// TIA Portal project "Project3" (V14)

(* hardware
DEVICE "S7-1200 station_1"  S7-1200 Station
   slot 0: "Rack_0"  S7-1200 Rack  Rack  V1.0
   slot 1: "PLC_1"  CPU 1215C DC/DC/DC  6ES7 215-1AG40-0XB0  V4.2
   slot 2: "DI 16/DQ 16x24VDC_1"  6ES7 223-1BL32-0XB0  V2.0
   slot 3: "DI 16/DQ 16x24VDC_2"  6ES7 223-1BL32-0XB0  V2.0
   slot 4: "AI 4x13BIT_1"  6ES7 231-4HD32-0XB0  V2.0
   slot 5: "AI 4xRTD_1"  SM 1231 AI4 x RTD  6ES7 231-5PD32-0XB0  V2.0
DEVICE "S7-1200 station_2"  S7-1200 Station
   slot 0: "Rack_0"  S7-1200 Rack  Rack  V1.0
   slot 1: "PLC_2"  CPU 1214C DC/DC/DC  6ES7 214-1AG40-0XB0  V4.2
   slot 2: "DI 16/DQ 16x24VDC_1"  6ES7 223-1BL32-0XB0  V2.0
   slot 3: "AQ 4x14BIT_1"  6ES7 232-4HD32-0XB0  V2.0
*)

// ===== PLC "PLC_1"  CPU 1215C DC/DC/DC =====

VAR_GLOBAL   // PLC tag table "Default tag table"
   "Rabota_M1.1" AT %I8.0 : Bool;
   "Rabota_X_M2" AT %I8.1 : Bool;
   "SL12.5.1" AT %I1.2 : Bool;
   "Gotovnost_M3" AT %I300.0 : Bool;
   "Rabota_M4" AT %I8.2 : Bool;
   "Rabota_M5" AT %I8.3 : Bool;
   "Gotovnost_X_M6.1" AT %I300.1 : Bool;
   "SL17.1" AT %I8.5 : Bool;
   "SL17.2" AT %I8.6 : Bool;
   "Gotovnost_M7.1" AT %I300.2 : Bool;
   "Gotovnost_M7" AT %I1.0 : Bool;
   "Rabota_X_12.1" AT %I300.5 : Bool;
   "Rabota_X_M6.1" AT %I300.6 : Bool;
   "Rabota_M8.3" AT %I300.7 : Bool;
   "Rabota_M9" AT %I301.0 : Bool;
   "Gotovnost_M10.1" AT %I300.3 : Bool;
   "Avaria_M10" AT %I1.4 : Bool;
   "Rabota_M11" AT %I301.1 : Bool;
   "Gotovnost_M12.1" AT %I300.4 : Bool;
   "Gotovnost_M12" AT %I1.1 : Bool;
   "Rabota_M13" AT %I301.2 : Bool;
   "Rabota_M14" AT %I301.3 : Bool;
   "Rabota_M15" AT %I301.4 : Bool;
   "Rabota_M16" AT %I301.5 : Bool;
   "Rabota_Vent" AT %I8.7 : Bool;
   "SB_Pusk_Cycle_Pererabotka" AT %I0.4 : Bool;
   "SB_Stop_Cycle_Pererabotka" AT %I0.5 : Bool;
   "Gribok_Shkaf_Pererabotka" AT %I0.2 : Bool;
   "Cycle_Filtration_Pusk" AT %I12.5 : Bool;
   "Cycle_Filtration_Stop" AT %I12.6 : Bool;
   "Filtration_Avary_Stop" AT %I12.7 : Bool;
   "Cepi_Upravlenia" AT %I0.0 : Bool;
   "Kontrol_Seti" AT %I0.1 : Bool;
   "Filtration_Avary_Stop_Post" AT %I13.1 : Bool;
   "Filtration_Blokirovka_Post" AT %I13.2 : Bool;
   "SL12.7.1.2_Zamok_Zakryt" AT %I13.4 : Bool;
   "SL12.7.3.2_Filtre_Zakryt" AT %I13.6 : Bool;
   "SL12.7.1.1_Zamok_Otkryt" AT %I13.3 : Bool;
   "SL12.7.3.1_Filtre_Otkryt" AT %I13.5 : Bool;
   "Baipas_UPP" AT %I12.0 : Bool;
   "SL1.2" AT %I12.1 : Bool;
   "SL1.1.1" AT %I16.4 : Bool;
   "SL1.1.2" AT %I16.5 : Bool;
   "SL5.1" AT %I12.3 : Bool;
   "None_4" AT %I16.6 : Bool;
   "None_5" AT %I16.7 : Bool;
   "None_6" AT %I17.0 : Bool;
   "SL7.5.3" AT %I17.1 : Bool;
   "SL9.1" AT %I302.0 : Bool;
   "OLD_SL11.1" AT %I302.1 : Bool;
   "None_0" AT %I16.0 : Bool;
   "None_1" AT %I16.1 : Bool;
   "SL13.1" AT %I302.2 : Bool;
   "None_2" AT %I16.2 : Bool;
   "None_3" AT %I16.3 : Bool;
   "Pererab_Ruchnoi_rezhim" AT %I0.7 : Bool;
   "Nachalo_Puska_M10" AT %I1.3 : Bool;
   "Pererabotka_stop" AT %I0.6 : Bool;
   "Avtomat_Kompress_On" AT %I8.4 : Bool;
   "Rabota_M1_Kotel" AT %I9.0 : Bool;
   "Rabota_M2_Kotel" AT %I9.1 : Bool;
   "Avtomat_Rabota_Osyshit" AT %I9.2 : Bool;
   "OLD_SL12.1" AT %I9.3 : Bool;
   "SL7.5.1" AT %I9.4 : Bool;
   "SL7.5.2" AT %I9.5 : Bool;
   "SB_vent_PUSK" AT %I9.6 : Bool;
   "SB_Vent_Stop" AT %I9.7 : Bool;
   "SL2.1" AT %I12.2 : Bool;
   "DatchikSP" AT %I12.4 : Bool;
   "Filtration_Manual" AT %I13.0 : Bool;
   "SL12.7.4" AT %I13.7 : Bool;
   "SB_Pusk_Ventilation" AT %I17.4 : Bool;
   "SB_Stop_Ventilation" AT %I17.5 : Bool;
   "Tok_M7_Int" AT %IW144 : Int;
   "Tok_M12_Int" AT %IW146 : Int;
   "Tok_M10_Int" AT %IW148 : Int;
   "Temper_T12.2" AT %IW160 : Int;
   "Temper_T1" AT %IW162 : Int;
   "Temper_T2" AT %IW164 : Int;
   "Temper_T3" AT %IW166 : Int;
   "Temper_T17.1" AT %IW168 : Int;
   "None_7" AT %I17.6 : Bool;
   "Pusk_M1.1" AT %Q8.0 : Bool;
   "Pusk_X_M2" AT %Q8.1 : Bool;
   "Pusk_M2" AT %Q0.5 : Bool;
   "Pusk_M3" AT %Q304.0 : Bool;
   "Pusk_M4" AT %Q8.2 : Bool;
   "Pusk_M5" AT %Q8.3 : Bool;
   "Pusk_X_M6.1" AT %Q304.1 : Bool;
   "Zamok_Open" AT %Q8.4 : Bool;
   "Zamok_Close" AT %Q8.5 : Bool;
   "Pusk_M7.1" AT %Q304.3 : Bool;
   "Pusk_M7" AT %Q0.1 : Bool;
   "Pusk_X_M12.1" AT %Q306.0 : Bool;
   "Pusk_X_6.1" AT %Q306.1 : Bool;
   "Pusk_M8.3" AT %Q306.2 : Bool;
   "Pusk_M9" AT %Q306.3 : Bool;
   "Pusk_M10.1" AT %Q304.5 : Bool;
   "Pusk_M10" AT %Q0.7 : Bool;
   "Pusk_M11" AT %Q306.4 : Bool;
   "Pusk_M12.1" AT %Q304.7 : Bool;
   "Pusk_M12" AT %Q0.3 : Bool;
   "Pusk_M13" AT %Q306.5 : Bool;
   "Pusk_M14" AT %Q306.6 : Bool;
   "Pusk_M15" AT %Q306.7 : Bool;
   "Pusk_M16" AT %Q307.0 : Bool;
   "Pusk_Vent" AT %Q8.6 : Bool;
   "Podogrev1_On" AT %Q0.0 : Bool;
   "Klapan_K1" AT %Q13.0 : Bool;
   "Klapan_K2" AT %Q13.1 : Bool;
   "Klapan_K3" AT %Q13.2 : Bool;
   "Klapan_K4" AT %Q13.3 : Bool;
   "Klapan_Kd" AT %Q13.4 : Bool;
   "Klapan_Kp6" AT %Q13.5 : Bool;
   "Klapan_Kp7" AT %Q13.6 : Bool;
   "Vibromotor" AT %Q13.7 : Bool;
   "NA1" AT %Q16.0 : Bool;
   "NA2" AT %Q16.1 : Bool;
   "NA3" AT %Q16.2 : Bool;
   "NA4" AT %Q16.3 : Bool;
   "Klapan_K12.5" AT %Q16.4 : Bool;
   "Klapan_K17" AT %Q16.5 : Bool;
   "Klapan_K2.1" AT %Q16.6 : Bool;
   "Klapan_P22.1" AT %Q16.7 : Bool;
   "Klapan_P22.2" AT %Q17.0 : Bool;
   "Avariyn_Stop_M10" AT %Q1.0 : Bool;
   "Sbros_Privodov1" AT %Q0.6 : Bool;
   "Pusk_Revers_M7" AT %Q0.2 : Bool;
   "Pusk_Revers_M12" AT %Q0.4 : Bool;
   "Pusk_Kotel1" AT %Q8.7 : Bool;
   "Pusk_Kotel2" AT %Q9.0 : Bool;
   "Gotovnost_Kontrollera" AT %Q12.0 : Bool;
   "ZadanieM7_Raw" AT %QW64 : Int;
   "ZadanieM12_Raw" AT %QW66 : Int;
   "Pusk_Revers_M6.1" AT %Q304.2 : Bool;
   "Pusk_Revers_M7.1" AT %Q304.4 : Bool;
   "Pusk_Revers_M10.1" AT %Q304.6 : Bool;
   "Pusk_Revers_M12.1" AT %Q305.0 : Bool;
   "Sbros_Privodov2" AT %Q305.1 : Bool;
   "ZadanieM6.1_Raw" AT %QW308 : Int;
   "ZadanieM7.1_Raw" AT %QW310 : Int;
   "ZadanieM10.1_Raw" AT %QW312 : Int;
   "ZadanieM12.1_Raw" AT %QW314 : Int;
   "Svetofor_Sirena" AT %Q9.3 : Bool;
   "Svetofor_Krasniy" AT %Q9.4 : Bool;
   "Svetofor_Zeleniy" AT %Q9.5 : Bool;
   "Lamp_Cepi_Upravlenia" AT %Q12.1 : Bool;
   "Lamp_Pererab_Cycle" AT %Q12.2 : Bool;
   "Lamp_Pererab_Avariya" AT %Q12.3 : Bool;
   "Lamp_Filtration_Cycle" AT %Q12.4 : Bool;
   "Lamp_Filtration_Avariya" AT %Q12.5 : Bool;
   "Lamp_Ventilation" AT %Q12.6 : Bool;
   "Tag_2" AT %Q307.3 : Bool;
   "System_Byte" AT %MB1 : Byte;
   "FirstScan" AT %M1.0 : Bool;
   "DiagStatusUpdate" AT %M1.1 : Bool;
   "AlwaysTRUE" AT %M1.2 : Bool;
   "AlwaysFALSE" AT %M1.3 : Bool;
   "Clock_Byte" AT %MB0 : Byte;
   "Clock_10Hz" AT %M0.0 : Bool;
   "Clock_5Hz" AT %M0.1 : Bool;
   "Clock_2.5Hz" AT %M0.2 : Bool;
   "Clock_2Hz" AT %M0.3 : Bool;
   "Clock_1.25Hz" AT %M0.4 : Bool;
   "Clock_1Hz" AT %M0.5 : Bool;
   "Clock_0.625Hz" AT %M0.6 : Bool;
   "Clock_0.5Hz" AT %M0.7 : Bool;
   "SB_Pusk_Cycle_Zargruzka" AT %M8.6 : Bool;
   "SB_Stop_Cycle_Zargruzka" AT %M8.7 : Bool;
   "Tag_1" AT %M1000.0 : Bool;
   "SL12.5.2" AT %I1.5 : Bool;
   "Filtre_Open" AT %Q9.6 : Bool;
   "Filtre_Close" AT %Q9.7 : Bool;
   "SL8.3" AT %I302.5 : Bool;
   "SL12.1" AT %I302.6 : Bool;
   "SL11.1" AT %I302.7 : Bool;
END_VAR

DATA_BLOCK "Local_Data"   // DB1
{ S7_Optimized_Access := 'TRUE' }
VERSION : 0.1
   VAR
      "Timer_Error_M1.1" : IEC_TIMER;
      Timer_Error_X_M2 : IEC_TIMER;
      Timer_Error_M2 : IEC_TIMER;
      Timer_Error_M3 : IEC_TIMER;
      Timer_Error_M4 : IEC_TIMER;
      Timer_Error_M5 : IEC_TIMER;
      "Timer_Error_M6.1" : IEC_TIMER;
      "Timer_Error_M6.2" : IEC_TIMER;
      "Timer_Error_M6.3" : IEC_TIMER;
      "Timer_Error_M7.1" : IEC_TIMER;
      Timer_Error_M7 : IEC_TIMER;
      "Timer_Error_X_M12.1" : IEC_TIMER;
      "Timer_Error_X_M6.1" : IEC_TIMER;
      "Timer_Error_M8.3" : IEC_TIMER;
      Timer_Error_M9 : IEC_TIMER;
      "Timer_Error_M10.1" : IEC_TIMER;
      Timer_Error_M10 : IEC_TIMER;
      Timer_Error_M11 : IEC_TIMER;
      "Timer_Error_M12.1" : IEC_TIMER;
      Timer_Error_M12 : IEC_TIMER;
      Timer_Error_M13 : IEC_TIMER;
      Timer_Error_M14 : IEC_TIMER;
      Timer_Error_M15 : IEC_TIMER;
      Timer_Error_M16 : IEC_TIMER;
      Timer_Error_Vent : IEC_TIMER;
      Timer_Error_Mkotel1 : IEC_TIMER;
      Timer_Error_Mkotel2 : IEC_TIMER;
   END_VAR
BEGIN
END_DATA_BLOCK

DATA_BLOCK "Unlock_Data"   // DB2
{ S7_Optimized_Access := 'FALSE' }
VERSION : 0.1
   VAR
      "Error_M1.1" : Bool;
      Error_X_M2 : Bool;
      Error_M2 : Bool;
      Error_M3 : Bool;
      Error_M4 : Bool;
      Error_M5 : Bool;
      "Error_M6.1" : Bool;
      "Error_M6.2" : Bool;
      "Error_M6.3" : Bool;
      "Error_M7.1" : Bool;
      Error_M7 : Bool;
      "Error_X_M12.1" : Bool;
      "Error_X_M6.1" : Bool;
      "Error_M8.3" : Bool;
      Error_M9 : Bool;
      "Error_M10.1" : Bool;
      Error_M10 : Bool;
      Error_M11 : Bool;
      "Error_M12.1" : Bool;
      Error_M12 : Bool;
      Error_M13 : Bool;
      Error_M14 : Bool;
      Error_M15 : Bool;
      Error_M16 : Bool;
      Error_Vent : Bool;
      "SB_Man_On_M1.1" : Bool;
      "SB_Man_Off_M1.1" : Bool;
      SB_Man_On_X_M2 : Bool;
      SB_Man_Off_X_M2 : Bool;
      SB_Man_On_M2 : Bool;
      SB_Man_Off_M2 : Bool;
      SB_Man_On_M3 : Bool;
      SB_Man_Off_M3 : Bool;
      SB_Man_On_M4 : Bool;
      SB_Man_Off_M4 : Bool;
      SB_Man_On_M5 : Bool;
      SB_Man_Off_M5 : Bool;
      "SB_Man_On_M6.1" : Bool;
      "SB_Man_Off_M6.1" : Bool;
      "SB_Man_On_M6.2" : Bool;
      "SB_Man_Off_M6.2" : Bool;
      "SB_Man_On_M6.3" : Bool;
      "SB_Man_Off_M6.3" : Bool;
      "SB_Man_On_M7.1" : Bool;
      "SB_Man_Off_M7.1" : Bool;
      SB_Man_On_M7 : Bool;
      SB_Man_Off_M7 : Bool;
      "SB_Man_On_X_M12.1" : Bool;
      "SB_Man_Off_X_M12.1" : Bool;
      "SB_Man_On_X_M6.1" : Bool;
      "SB_Man_Off_X_M6.1" : Bool;
      "SB_Man_On_M8.3" : Bool;
      "SB_Man_Off_M8.3" : Bool;
      SB_Man_On_M9 : Bool;
      SB_Man_Off_M9 : Bool;
      "SB_Man_On_M10.1" : Bool;
      "SB_Man_Off_M10.1" : Bool;
      SB_Man_On_M10 : Bool;
      SB_Man_Off_M10 : Bool;
      SB_Man_On_M11 : Bool;
      SB_Man_Off_M11 : Bool;
      "SB_Man_On_M12.1" : Bool;
      "SB_Man_Off_M12.1" : Bool;
      SB_Man_On_M12 : Bool;
      SB_Man_Off_M12 : Bool;
      SB_Man_On_M13 : Bool;
      SB_Man_Off_M13 : Bool;
      SB_Man_On_M14 : Bool;
      SB_Man_Off_M14 : Bool;
      SB_Man_On_M15 : Bool;
      SB_Man_Off_M15 : Bool;
      SB_Man_On_M16 : Bool;
      SB_Man_Off_M16 : Bool;
      SB_Man_On_Vent : Bool;
      SB_Man_Off_Vent : Bool;
      "Auto_On_M1.1" : Bool;
      Auto_On_X_M2 : Bool;
      Auto_On_M2 : Bool;
      Auto_On_M3 : Bool;
      Auto_On_M4 : Bool;
      Auto_On_M5 : Bool;
      "Auto_On_M6.1" : Bool;
      "Auto_On_M6.2" : Bool;
      "Auto_On_M6.3" : Bool;
      "Auto_On_M7.1" : Bool;
      Auto_On_M7 : Bool;
      "Auto_On_X_M12.1" : Bool;
      "Auto_On_X_M6.1" : Bool;
      "Auto_On_M8.3" : Bool;
      Auto_On_M9 : Bool;
      "Auto_On_M10.1" : Bool;
      Auto_On_M10 : Bool;
      Auto_On_M11 : Bool;
      "Auto_On_M12.1" : Bool;
      Auto_On_M12 : Bool;
      Auto_On_M13 : Bool;
      Auto_On_M14 : Bool;
      Auto_On_M15 : Bool;
      Auto_On_M16 : Bool;
      Auto_On_Vent : Bool;
      RESET_ERRORS_PANEL : Bool;
      Manual_Rezhim : Bool;
      Auto_Rezhim : Bool;
      Cycle_Pererab_Pusk : Bool;
      Cycle_Zagruzka_Pusk : Bool;
      SB_Man_On_Podogrev1 : Bool;
      SB_Man_Off_Podogrev1 : Bool;
      SB_Man_On_Podogrev2 : Bool;
      SB_Man_Off_Podogrev2 : Bool;
      Auto_On_Podogrev1 : Bool;
      Motors_Group1_Ok : Bool;
      Motors_Group2_Ok : Bool;
      Ready_Group1 : Bool;
      Ready_Group2 : Bool;
      "Vivod_iz_auto_M1.1" : Bool;
      Vivod_iz_auto_X_M2 : Bool;
      Vivod_iz_auto_M2 : Bool;
      Vivod_iz_auto_M3 : Bool;
      Vivod_iz_auto_M4 : Bool;
      Vivod_iz_auto_M5 : Bool;
      "Vivod_iz_auto_M6.1" : Bool;
      "Vivod_iz_auto_M6.2" : Bool;
      "Vivod_iz_auto_M6.3" : Bool;
      "Vivod_iz_auto_M7.1" : Bool;
      Vivod_iz_auto_M7 : Bool;
      "Vivod_iz_auto_X_M12.1" : Bool;
      "Vivod_iz_auto_X_M6.1" : Bool;
      "Vivod_iz_auto_M8.3" : Bool;
      Vivod_iz_auto_M9 : Bool;
      "Vivod_iz_auto_M10.1" : Bool;
      Vivod_iz_auto_M10 : Bool;
      Vivod_iz_auto_M11 : Bool;
      "Vivod_iz_auto_M12.1" : Bool;
      Vivod_iz_auto_M12 : Bool;
      Vivod_iz_auto_M13 : Bool;
      Vivod_iz_auto_M14 : Bool;
      Vivod_iz_auto_M15 : Bool;
      Vivod_iz_auto_M16 : Bool;
      "Vivesti_iz_auto_M1.1" : Bool;
      Vivesti_iz_auto_X_M2 : Bool;
      Vivesti_iz_auto_M2 : Bool;
      Vivesti_iz_auto_M3 : Bool;
      Vivesti_iz_auto_M4 : Bool;
      Vivesti_iz_auto_M5 : Bool;
      "Vivesti_iz_auto_M6.1" : Bool;
      "Vivesti_iz_auto_M6.2" : Bool;
      "Vivesti_iz_auto_M6.3" : Bool;
      "Vivesti_iz_auto_M7.1" : Bool;
      Vivesti_iz_auto_M7 : Bool;
      "Vivesti_iz_auto_X_M12.1" : Bool;
      "Vivesti_iz_auto_X_M6.1" : Bool;
      "Vivesti_iz_auto_M8.3" : Bool;
      Vivesti_iz_auto_M9 : Bool;
      "Vivesti_iz_auto_M10.1" : Bool;
      Vivesti_iz_auto_M10 : Bool;
      Vivesti_iz_auto_M11 : Bool;
      "Vivesti_iz_auto_M12.1" : Bool;
      Vivesti_iz_auto_M12 : Bool;
      Vivesti_iz_auto_M13 : Bool;
      Vivesti_iz_auto_M14 : Bool;
      Vivesti_iz_auto_M15 : Bool;
      Vivesti_iz_auto_M16 : Bool;
      BIT_AUTORIZATION : Bool;
      pulse_auto_F : Bool;
      System_Ok : Bool;
      Error_Mkotel1 : Bool;
      Error_Mkotel2 : Bool;
      SB_Man_On_M7_Rev : Bool;
      SB_Man_Off_M7_Rev : Bool;
      SB_Man_On_M12_Rev : Bool;
      SB_Man_Off_M12_Rev : Bool;
      "SB_Man_On_M6.1_Rev" : Bool;
      "SB_Man_Off_M6.1_Rev" : Bool;
      "SB_Man_On_M7.1_Rev" : Bool;
      "SB_Man_Off_M7.1_Rev" : Bool;
      "SB_Man_On_M10.1_Rev" : Bool;
      "SB_Man_Off_M10.1_Rev" : Bool;
      "SB_Man_On_M12.1_Rev" : Bool;
      "SB_Man_Off_M12.1_Rev" : Bool;
      Temperature_Real_T3 : Real;
      Ustavka_Ekstruder : Real;
      Temperature_Real_T2 : Real;
      Temperature_Real_T1 : Real;
      "Temperature_Real_T12.2" : Real;
      "Temperature_Real_T17.1" : Real;
      Tok_M7_Real : Real;
      Tok_M12_Real : Real;
      Tok_M10_Real : Real;
      Tok_M7_Real_Temp_Panel : Real;
      Tok_M12_Real_Temp_Panel : Real;
      Tok_M10_Real_Temp_Panel : Real;
      Tok_M7_Real_Temp1 : Real;
      Tok_M12_Real_Temp1 : Real;
      Tok_M10_Real_Temp1 : Real;
      "Ignore_SL17.1" : Bool;
      Cycle_Pererabotka_Stop : Bool;
      Timer_CPU_retVol : Int;
      Timer_CPU_statusRTM : Bool;
      Timer_CPU_output : DInt;
      Timer_M7_retVol : Int;
      Timer_M7_statusRTM : Bool;
      Timer_M7_output : DInt;
      Timer_M10_retVol : Int;
      Timer_M10_statusRTM : Bool;
      Timer_M10_output : DInt;
      Timer_M12_retVol : Int;
      Timer_M12_StatusRTM : Bool;
      Timer_M12_output : DInt;
   END_VAR
BEGIN
END_DATA_BLOCK

DATA_BLOCK "Retain_Data"   // DB3
{ S7_Optimized_Access := 'FALSE' }
VERSION : 0.1
   VAR
      "Timer_On_M1.1" : IEC_TIMER;
      Timer_On_X_M2 : IEC_TIMER;
      Timer_On_M2 : IEC_TIMER;
      Timer_On_M3 : IEC_TIMER;
      Timer_On_M4 : IEC_TIMER;
      Timer_On_M5 : IEC_TIMER;
      "Timer_On_X_M6.2" : IEC_TIMER;
      "Timer_On_M6.1_ex_M6.2" : IEC_TIMER;
      "Timer_On_M6.3" : IEC_TIMER;
      "Timer_On_M7.1" : IEC_TIMER;
      Timer_On_M7 : IEC_TIMER;
      "Timer_On_X_M12.1" : IEC_TIMER;
      "Timer_On_X_M6.1" : IEC_TIMER;
      "Timer_On_M8.3" : IEC_TIMER;
      Timer_On_M9 : IEC_TIMER;
      "Timer_On_M10.1" : IEC_TIMER;
      Timer_On_M10 : IEC_TIMER;
      Timer_On_M11 : IEC_TIMER;
      "Timer_On_M12.1" : IEC_TIMER;
      Timer_On_M12 : IEC_TIMER;
      Timer_On_M13 : IEC_TIMER;
      Timer_On_M14 : IEC_TIMER;
      Timer_On_M15 : IEC_TIMER;
      Timer_On_M16 : IEC_TIMER;
      "Timer_Off_M1.1" : IEC_TIMER;
      Timer_Off_X_M2 : IEC_TIMER;
      Timer_Off_M2 : IEC_TIMER;
      Timer_Off_M3 : IEC_TIMER;
      Timer_Off_M4 : IEC_TIMER;
      Timer_Off_M5 : IEC_TIMER;
      "Timer_Off_OLD_M6.1" : IEC_TIMER;
      "Timer_Off_M6.1_ex_M6.2" : IEC_TIMER;
      "Timer_Off_M6.3" : IEC_TIMER;
      "Timer_Off_M7.1" : IEC_TIMER;
      Timer_Off_M7 : IEC_TIMER;
      "Timer_Off_X_M12.1" : IEC_TIMER;
      "Timer_Off_X_M6.1" : IEC_TIMER;
      "Timer_Off_M8.3" : IEC_TIMER;
      Timer_Off_M9 : IEC_TIMER;
      "Timer_Off_M10.1" : IEC_TIMER;
      Timer_Off_M10 : IEC_TIMER;
      Timer_Off_M11 : IEC_TIMER;
      "Timer_Off_M12.1" : IEC_TIMER;
      Timer_Off_M12 : IEC_TIMER;
      Timer_Off_M13 : IEC_TIMER;
      Timer_Off_M14 : IEC_TIMER;
      Timer_Off_M15 : IEC_TIMER;
      Timer_Off_M16 : IEC_TIMER;
      Timer_K1 : IEC_TIMER;
      Timer_F_1 : IEC_TIMER;
      Timer_F_2 : IEC_TIMER;
      Timer_F_3 : IEC_TIMER;
      Timer_F_4 : IEC_TIMER;
      Timer_F_5 : IEC_TIMER;
      Timer_F_6 : IEC_TIMER;
      Timer_F_7 : IEC_TIMER;
      Timer_F_8 : IEC_TIMER;
      Timer_F_9 : IEC_TIMER;
      Timer_F_10 : IEC_TIMER;
      Timer_F_11 : IEC_TIMER;
      Timer_F_12 : IEC_TIMER;
      Timer_F_13 : IEC_TIMER;
      Timer_F_14 : IEC_TIMER;
      Timer_F_15 : IEC_TIMER;
      Tim_F_pusk : IEC_TIMER;
      Counter_F_1 : IEC_COUNTER;
      Counter_F_2 : IEC_COUNTER;
      Counter_F_3 : IEC_COUNTER;
      Counter_F_4 : IEC_COUNTER;
      Counter_F_5 : IEC_COUNTER;
      Counter_F_6 : IEC_COUNTER;
      "Timer_Delay_22.1" : IEC_TIMER;
      "Timer_Delay_22.2" : IEC_TIMER;
      "Vibor_M1.1" : Bool;
      "Vibor_M1.2" : Bool;
      "Timer_SL2.1" : IEC_TIMER;
      "Timer_SL5.1" : IEC_TIMER;
      "Timer_SL12.1" : IEC_TIMER;
      "Timer_SL7.5.3" : IEC_TIMER;
      "Timer_SL9.1" : IEC_TIMER;
      "Timer_SL11.1" : IEC_TIMER;
      "Timer_SL13.1" : IEC_TIMER;
      "tSL12.3" : IEC_TIMER;
      "Timer_SL12.5.2" : IEC_TIMER;
      "Timer_SL17.2" : IEC_TIMER;
      "Drebezg_SL17.2" : IEC_TIMER;
      "Timer_On_SL17.2" : IEC_TIMER;
      Timer_Ekst_Temper_On : IEC_TIMER;
      Timer_Ekst_Temper_Off : IEC_TIMER;
      Ustavka_Ekstruder : Real;
      "Zadanie_Real_M6.1" : Real;
      "Zadanie_Real_M7.1" : Real;
      Zadanie_Real_M7 : Real;
      "Zadanie_Real_M10.1" : Real;
      "Zadanie_Real_M12.1" : Real;
      Zadanie_Real_M12 : Real;
      Delitel_M7 : Real;
      Delitel_M12 : Real;
      Delitel_M10 : Real;
      "Timer_SL1.1" : IEC_TIMER;
      "Timer_SL1.2" : IEC_TIMER;
      "tSL1.1" : IEC_TIMER;
      Timer_Temp_M7 : IEC_TIMER;
      Ustavka_tok_M7 : Real;
      Ustavka_tok_M10 : Real;
      Ustavka_tok_M12 : Real;
      Timer_Temp_M7_OFF : IEC_TIMER;
      Timer_Tok_M10 : IEC_TIMER;
      Timer_Tok_M10_OFF : IEC_TIMER;
      Timer_Tok_M12 : IEC_TIMER;
      Timer_Tok_M12_OFF : IEC_TIMER;
      "Timer_SL8.3" : IEC_TIMER;
   END_VAR
BEGIN
END_DATA_BLOCK

DATA_BLOCK "Unlock_Filtration"   // DB4
{ S7_Optimized_Access := 'FALSE' }
VERSION : 0.1
   VAR
      Manual_Filtration : Bool;
      Auto_Filtration : Bool;
      SB_Man_K1_Open : Bool;
      SB_Man_K1_Close : Bool;
      SB_Man_K2_Open : Bool;
      SB_Man_K2_Close : Bool;
      "SB_Man_K2.1_Open" : Bool;
      "SB_Man_K2.1_Close" : Bool;
      SB_Man_K3_Open : Bool;
      SB_Man_K3_Close : Bool;
      SB_Man_K4_Open : Bool;
      SB_Man_K4_Close : Bool;
      SB_Man_Kd_Open : Bool;
      SB_Man_Kd_Close : Bool;
      SB_Man_Kp6_Open : Bool;
      SB_Man_Kp6_Close : Bool;
      SB_Man_Kp7_Open : Bool;
      SB_Man_Kp7_Close : Bool;
      SB_Man_Vibro_On : Bool;
      SB_Man_Vibro_Off : Bool;
      SB_Man_Zamok_Open : Bool;
      SB_Man_Zamok_Close : Bool;
      SB_Filtre_Open : Bool;
      SB_Filtre_Close : Bool;
      "SB_Man_K12.5_Open" : Bool;
      "SB_Man_K12.5_Close" : Bool;
      SB_Man_K17_Open : Bool;
      SB_Man_K17_Close : Bool;
      "SB_Man_P22.1_Open" : Bool;
      "SB_Man_P22.1_Close" : Bool;
      "SB_Man_P22.2_Open" : Bool;
      "SB_Man_P22.2_Close" : Bool;
   END_VAR
BEGIN
END_DATA_BLOCK

DATA_BLOCK "Zadanie_DB"   // DB5
{ S7_Optimized_Access := 'TRUE' }
VERSION : 0.1
// stored: InstanceOfName Zadanie
"Zadanie"
BEGIN
END_DATA_BLOCK

DATA_BLOCK "Errors_DB"   // DB6
{ S7_Optimized_Access := 'TRUE' }
VERSION : 0.1
// stored: InstanceOfName Errors
"Errors"
BEGIN
END_DATA_BLOCK

DATA_BLOCK "Filtration_Tags"   // DB7
{ S7_Optimized_Access := 'FALSE' }
VERSION : 0.1
   VAR
      MODE1 : Bool;
      MODE2 : Bool;
      MODE3 : Bool;
      MODE4 : Bool;
      ZC1 : Bool;
      ZC2 : Bool;
      ZC3 : Bool;
      ZC4 : Bool;
      SB_C1 : Bool;
      SB_C2 : Bool;
      SB_C3 : Bool;
      SB_C4 : Bool;
      KC1 : Bool;
      KC2 : Bool;
      KC3 : Bool;
      KC4 : Bool;
      KR1 : Bool;
      KR2 : Bool;
      KR3 : Bool;
      KR4 : Bool;
      Avto_F : Bool;
      Ready_F : Bool;
      ZC_F : Bool;
      Net_C : Bool;
      Error_F : Bool;
      Man_F : Bool;
      Cycle_F : Bool;
      C1 : Bool;
      C2 : Bool;
      C2_Stop : Bool;
      C3 : Bool;
      C4 : Bool;
      C4_E1 : Bool;
      C4_E2 : Bool;
      C4_E3 : Bool;
      pulse1 : Bool;
      C3_E1 : Bool;
      C3_E2 : Bool;
      C3_E3 : Bool;
      C3_E4 : Bool;
      pulse_KC1 : Bool;
      pulse_KC2 : Bool;
      pulse_KC3 : Bool;
      pulse_KC4 : Bool;
      pulse_SB_C1 : Bool;
      pulse_SB_C2 : Bool;
      pulse_SB_C3 : Bool;
      pulse_SB_C4 : Bool;
      pulse_SB_C1_1 : Bool;
      pulse_SB_C1_2 : Bool;
      pulse_SB_C1_3 : Bool;
      pulse_SB_C1_4 : Bool;
      pulse_F1 : Bool;
      pulse_F2 : Bool;
      pulse_F3 : Bool;
      pulse_F4 : Bool;
      pulse_F5 : Bool;
      PulseG_1 : Bool;
      PulseG_2 : Bool;
      PulseG_3 : Bool;
      "Vibor_12.5_xolodnoe" : Bool;
      Vibor_17_goryacheye : Bool;
      "Zabor_s_12.5" : Bool;
      Zabor_s_17 : Bool;
      pulse_KC5 : Bool;
      Sbros_Emkostei : Bool;
      Srabotal_KC2 : Bool;
      pulseKC_M19H : Bool;
      "pulse_T_SL18.1" : Bool;
      Word_Emkosti : Word;
      Pulse_W1_plus : Bool;
      Pulse_W2_plus : Bool;
      Sbros_Summ_W1 : Bool;
      Sbros_Summ_W2 : Bool;
      Pulse_sbros_W1 : Bool;
      Pulse_sbros_W2 : Bool;
      PLUS_W1_PANEL : Bool;
      PLUS_W2_PANEL : Bool;
      Pulse_W2_panel : Bool;
      Count_Etap1 : Int;
      Count_Etap2 : Int;
      Count_Etap3 : Int;
      Count_Etap4 : Int;
   END_VAR
BEGIN
END_DATA_BLOCK

DATA_BLOCK "Blokirovki_DB"   // DB8
{ S7_Optimized_Access := 'TRUE' }
VERSION : 0.1
// stored: InstanceOfName Blokirovki
"Blokirovki"
BEGIN
END_DATA_BLOCK

DATA_BLOCK "Filtration_DB"   // DB9
{ S7_Optimized_Access := 'TRUE' }
VERSION : 0.1
// stored: InstanceOfName Filtration
"Filtration"
BEGIN
END_DATA_BLOCK

DATA_BLOCK "Group1_Cycle_DB"   // DB10
{ S7_Optimized_Access := 'TRUE' }
VERSION : 0.1
// stored: InstanceOfName Group1_Cycle
"Group1_Cycle"
BEGIN
END_DATA_BLOCK

DATA_BLOCK "Lamp_Sound_DB"   // DB11
{ S7_Optimized_Access := 'TRUE' }
VERSION : 0.1
// stored: InstanceOfName Lamp_Sound
"Lamp_Sound"
BEGIN
END_DATA_BLOCK

DATA_BLOCK "Main_Cycle_DB"   // DB12
{ S7_Optimized_Access := 'TRUE' }
VERSION : 0.1
// stored: InstanceOfName Main_Cycle
"Main_Cycle"
BEGIN
END_DATA_BLOCK

DATA_BLOCK "Blokirovki_Data"   // DB13
{ S7_Optimized_Access := 'FALSE' }
VERSION : 0.1
   VAR
      "Srabotal_SL1.1.2" : Bool;
      "Srabotal_SL2.1" : Bool;
      "Srabotal_SL5.1" : Bool;
      "Srabotal_SL12.1" : Bool;
      "Srabotal_SL7.5.3" : Bool;
      "Srabotal_SL9.1" : Bool;
      "Srabotal_SL11.1" : Bool;
      "Srabotal_SL13.1" : Bool;
      "Srabotal_SL12.5.1" : Bool;
      "Srabotal_SL12.5.2" : Bool;
      "Srabotal_SL17.2" : Bool;
      Srabotal_T3 : Bool;
      "Srabotal_SL1.1" : Bool;
      "Srabotal_SL1.2" : Bool;
      "Srabotal_SL7.5.1" : Bool;
      "Ignore_SL17.2" : Bool;
      Srabotal_Tok_M7 : Bool;
      Srabotal_Tok_M10 : Bool;
      Srabotal_Tok_M12 : Bool;
      "Srabotal_SL8.3" : Bool;
   END_VAR
BEGIN
END_DATA_BLOCK

DATA_BLOCK "Motors_DB"   // DB14
{ S7_Optimized_Access := 'TRUE' }
VERSION : 0.1
// stored: InstanceOfName Motors
"Motors"
BEGIN
END_DATA_BLOCK

DATA_BLOCK "Motors_F_DB"   // DB15
{ S7_Optimized_Access := 'TRUE' }
VERSION : 0.1
// stored: InstanceOfName Motors_F
"Motors_F"
BEGIN
END_DATA_BLOCK

DATA_BLOCK "Temper_Tok_DB"   // DB16
{ S7_Optimized_Access := 'TRUE' }
VERSION : 0.1
// stored: InstanceOfName Temper_Tok
"Temper_Tok"
BEGIN
END_DATA_BLOCK

// folder: System blocks/Program resources

DATA_BLOCK "IEC_Timer_0_DB"   // DB17
{ S7_Optimized_Access := 'TRUE' }
AUTHOR : Simatic
FAMILY : IEC
NAME : IEC_TMR
VERSION : 1.0
// stored: InstanceOfName IEC_TIMER
"IEC_TIMER"
BEGIN
END_DATA_BLOCK

DATA_BLOCK "IEC_Timer_0_DB_1"   // DB18
{ S7_Optimized_Access := 'TRUE' }
AUTHOR : Simatic
FAMILY : IEC
NAME : IEC_TMR
VERSION : 1.0
// stored: InstanceOfName IEC_TIMER
"IEC_TIMER"
BEGIN
END_DATA_BLOCK

// folder: (top level)

FUNCTION_BLOCK "Errors"   // FB1, LAD
{ S7_Optimized_Access := 'TRUE' }
VERSION : 0.1
BEGIN

REGION Network 1
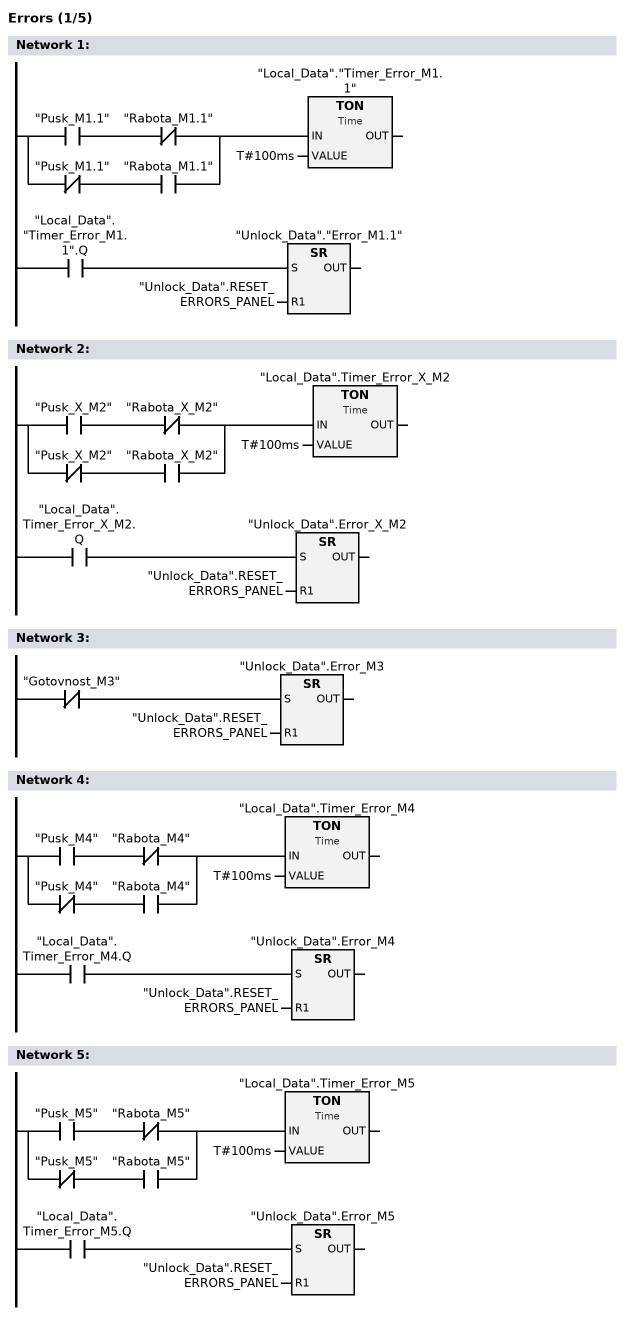
   "Local_Data"."Timer_Error_M1.1".TON(IN := ("Pusk_M1.1" AND NOT "Rabota_M1.1") OR (NOT "Pusk_M1.1" AND "Rabota_M1.1"), PT := T#100ms);   // TON coil
   IF "Local_Data"."Timer_Error_M1.1".Q THEN
       "Unlock_Data"."Error_M1.1" := TRUE;   // SR flip-flop
   END_IF;
   IF "Unlock_Data".RESET_ERRORS_PANEL THEN "Unlock_Data"."Error_M1.1" := FALSE; END_IF;
END_REGION

REGION Network 2
   "Local_Data".Timer_Error_X_M2.TON(IN := ("Pusk_X_M2" AND NOT "Rabota_X_M2") OR (NOT "Pusk_X_M2" AND "Rabota_X_M2"), PT := T#100ms);   // TON coil
   IF "Local_Data".Timer_Error_X_M2.Q THEN
       "Unlock_Data".Error_X_M2 := TRUE;   // SR flip-flop
   END_IF;
   IF "Unlock_Data".RESET_ERRORS_PANEL THEN "Unlock_Data".Error_X_M2 := FALSE; END_IF;
END_REGION

REGION Network 3
   RUNG wire#powerrail
      I_Contact( "Gotovnost_M3" )
      S_SR(operand := "Unlock_Data".Error_M3, r1 := "Unlock_Data".RESET_ERRORS_PANEL)
   END_RUNG
   // the same network as SCL:
   IF NOT "Gotovnost_M3" THEN
       "Unlock_Data".Error_M3 := TRUE;   // SR flip-flop
   END_IF;
   IF "Unlock_Data".RESET_ERRORS_PANEL THEN "Unlock_Data".Error_M3 := FALSE; END_IF;
END_REGION

REGION Network 4
   "Local_Data".Timer_Error_M4.TON(IN := ("Pusk_M4" AND NOT "Rabota_M4") OR (NOT "Pusk_M4" AND "Rabota_M4"), PT := T#100ms);   // TON coil
   IF "Local_Data".Timer_Error_M4.Q THEN
       "Unlock_Data".Error_M4 := TRUE;   // SR flip-flop
   END_IF;
   IF "Unlock_Data".RESET_ERRORS_PANEL THEN "Unlock_Data".Error_M4 := FALSE; END_IF;
END_REGION

REGION Network 5
   "Local_Data".Timer_Error_M5.TON(IN := ("Pusk_M5" AND NOT "Rabota_M5") OR (NOT "Pusk_M5" AND "Rabota_M5"), PT := T#100ms);   // TON coil
   IF "Local_Data".Timer_Error_M5.Q THEN
       "Unlock_Data".Error_M5 := TRUE;   // SR flip-flop
   END_IF;
   IF "Unlock_Data".RESET_ERRORS_PANEL THEN "Unlock_Data".Error_M5 := FALSE; END_IF;
END_REGION

REGION Network 8
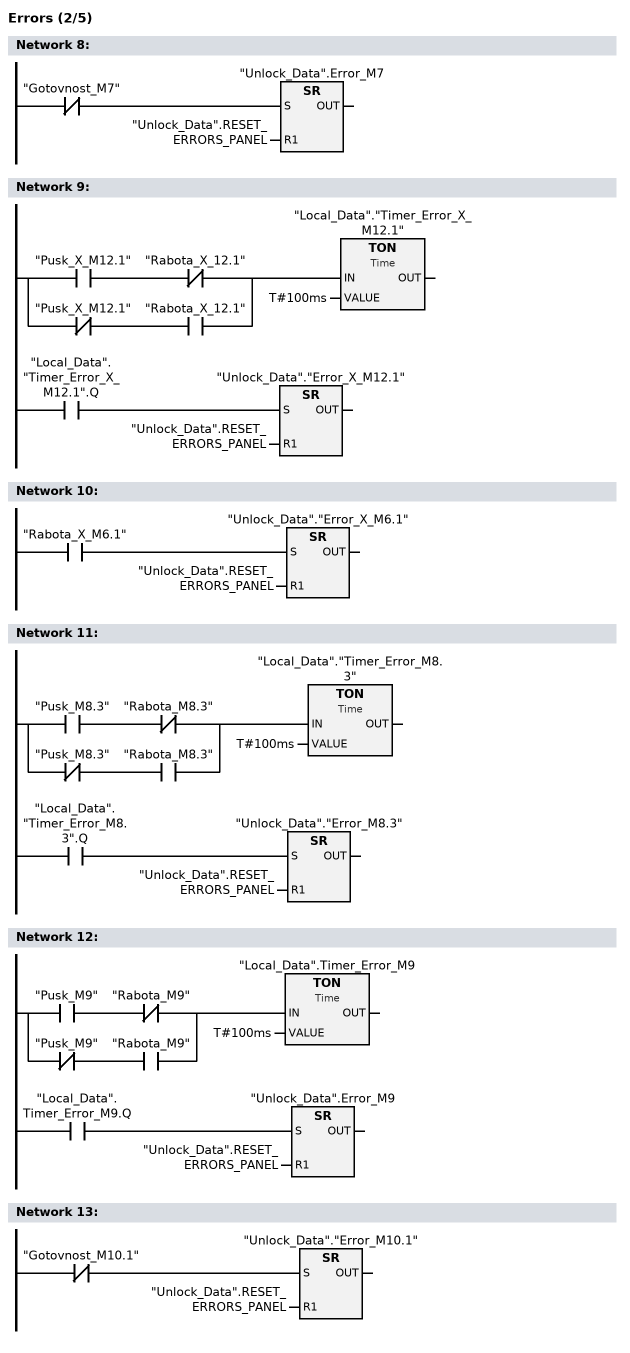
   RUNG wire#powerrail
      I_Contact( "Gotovnost_M7" )
      S_SR(operand := "Unlock_Data".Error_M7, r1 := "Unlock_Data".RESET_ERRORS_PANEL)
   END_RUNG
   // the same network as SCL:
   IF NOT "Gotovnost_M7" THEN
       "Unlock_Data".Error_M7 := TRUE;   // SR flip-flop
   END_IF;
   IF "Unlock_Data".RESET_ERRORS_PANEL THEN "Unlock_Data".Error_M7 := FALSE; END_IF;
END_REGION

REGION Network 9
   "Local_Data"."Timer_Error_X_M12.1".TON(IN := ("Pusk_X_M12.1" AND NOT "Rabota_X_12.1") OR (NOT "Pusk_X_M12.1" AND "Rabota_X_12.1"), PT := T#100ms);   // TON coil
   IF "Local_Data"."Timer_Error_X_M12.1".Q THEN
       "Unlock_Data"."Error_X_M12.1" := TRUE;   // SR flip-flop
   END_IF;
   IF "Unlock_Data".RESET_ERRORS_PANEL THEN "Unlock_Data"."Error_X_M12.1" := FALSE; END_IF;
END_REGION

REGION Network 10
   RUNG wire#powerrail
      Contact( "Rabota_X_M6.1" )
      S_SR(operand := "Unlock_Data"."Error_X_M6.1", r1 := "Unlock_Data".RESET_ERRORS_PANEL)
   END_RUNG
   // the same network as SCL:
   IF "Rabota_X_M6.1" THEN
       "Unlock_Data"."Error_X_M6.1" := TRUE;   // SR flip-flop
   END_IF;
   IF "Unlock_Data".RESET_ERRORS_PANEL THEN "Unlock_Data"."Error_X_M6.1" := FALSE; END_IF;
END_REGION

REGION Network 11
   "Local_Data"."Timer_Error_M8.3".TON(IN := ("Pusk_M8.3" AND NOT "Rabota_M8.3") OR (NOT "Pusk_M8.3" AND "Rabota_M8.3"), PT := T#100ms);   // TON coil
   IF "Local_Data"."Timer_Error_M8.3".Q THEN
       "Unlock_Data"."Error_M8.3" := TRUE;   // SR flip-flop
   END_IF;
   IF "Unlock_Data".RESET_ERRORS_PANEL THEN "Unlock_Data"."Error_M8.3" := FALSE; END_IF;
END_REGION

REGION Network 12
   "Local_Data".Timer_Error_M9.TON(IN := ("Pusk_M9" AND NOT "Rabota_M9") OR (NOT "Pusk_M9" AND "Rabota_M9"), PT := T#100ms);   // TON coil
   IF "Local_Data".Timer_Error_M9.Q THEN
       "Unlock_Data".Error_M9 := TRUE;   // SR flip-flop
   END_IF;
   IF "Unlock_Data".RESET_ERRORS_PANEL THEN "Unlock_Data".Error_M9 := FALSE; END_IF;
END_REGION

REGION Network 13
   RUNG wire#powerrail
      I_Contact( "Gotovnost_M10.1" )
      S_SR(operand := "Unlock_Data"."Error_M10.1", r1 := "Unlock_Data".RESET_ERRORS_PANEL)
   END_RUNG
   // the same network as SCL:
   IF NOT "Gotovnost_M10.1" THEN
       "Unlock_Data"."Error_M10.1" := TRUE;   // SR flip-flop
   END_IF;
   IF "Unlock_Data".RESET_ERRORS_PANEL THEN "Unlock_Data"."Error_M10.1" := FALSE; END_IF;
END_REGION

REGION Network 14
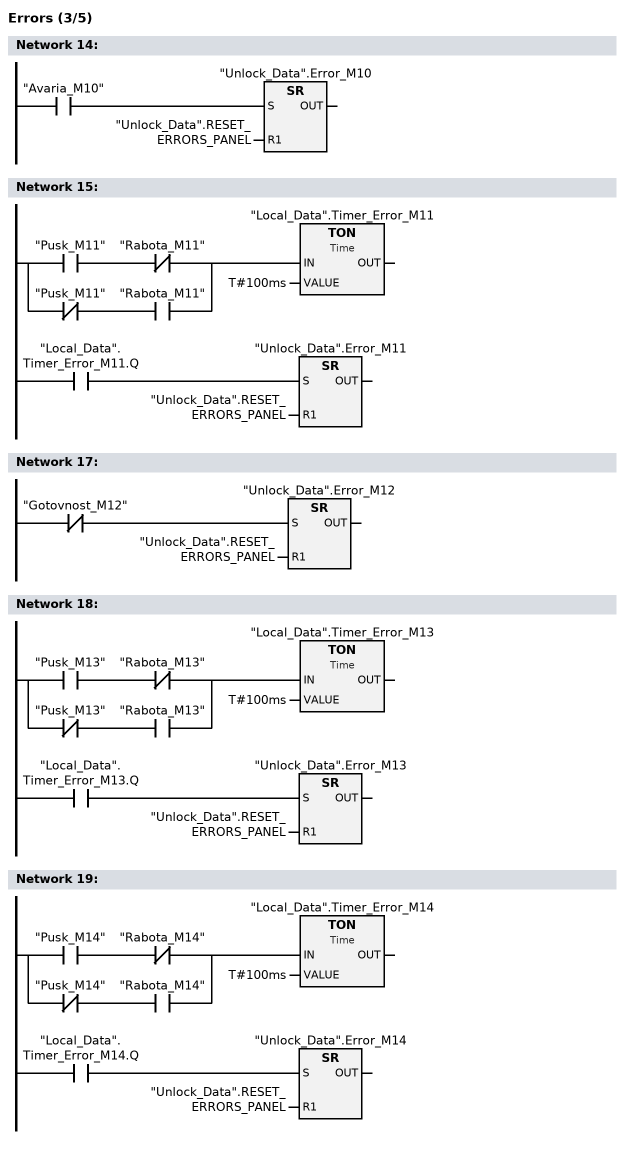
   RUNG wire#powerrail
      Contact( "Avaria_M10" )
      S_SR(operand := "Unlock_Data".Error_M10, r1 := "Unlock_Data".RESET_ERRORS_PANEL)
   END_RUNG
   // the same network as SCL:
   IF "Avaria_M10" THEN
       "Unlock_Data".Error_M10 := TRUE;   // SR flip-flop
   END_IF;
   IF "Unlock_Data".RESET_ERRORS_PANEL THEN "Unlock_Data".Error_M10 := FALSE; END_IF;
END_REGION

REGION Network 15
   "Local_Data".Timer_Error_M11.TON(IN := ("Pusk_M11" AND NOT "Rabota_M11") OR (NOT "Pusk_M11" AND "Rabota_M11"), PT := T#100ms);   // TON coil
   IF "Local_Data".Timer_Error_M11.Q THEN
       "Unlock_Data".Error_M11 := TRUE;   // SR flip-flop
   END_IF;
   IF "Unlock_Data".RESET_ERRORS_PANEL THEN "Unlock_Data".Error_M11 := FALSE; END_IF;
END_REGION

REGION Network 17
   RUNG wire#powerrail
      I_Contact( "Gotovnost_M12" )
      S_SR(operand := "Unlock_Data".Error_M12, r1 := "Unlock_Data".RESET_ERRORS_PANEL)
   END_RUNG
   // the same network as SCL:
   IF NOT "Gotovnost_M12" THEN
       "Unlock_Data".Error_M12 := TRUE;   // SR flip-flop
   END_IF;
   IF "Unlock_Data".RESET_ERRORS_PANEL THEN "Unlock_Data".Error_M12 := FALSE; END_IF;
END_REGION

REGION Network 18
   "Local_Data".Timer_Error_M13.TON(IN := ("Pusk_M13" AND NOT "Rabota_M13") OR (NOT "Pusk_M13" AND "Rabota_M13"), PT := T#100ms);   // TON coil
   IF "Local_Data".Timer_Error_M13.Q THEN
       "Unlock_Data".Error_M13 := TRUE;   // SR flip-flop
   END_IF;
   IF "Unlock_Data".RESET_ERRORS_PANEL THEN "Unlock_Data".Error_M13 := FALSE; END_IF;
END_REGION

REGION Network 19
   "Local_Data".Timer_Error_M14.TON(IN := ("Pusk_M14" AND NOT "Rabota_M14") OR (NOT "Pusk_M14" AND "Rabota_M14"), PT := T#100ms);   // TON coil
   IF "Local_Data".Timer_Error_M14.Q THEN
       "Unlock_Data".Error_M14 := TRUE;   // SR flip-flop
   END_IF;
   IF "Unlock_Data".RESET_ERRORS_PANEL THEN "Unlock_Data".Error_M14 := FALSE; END_IF;
END_REGION

REGION Network 20
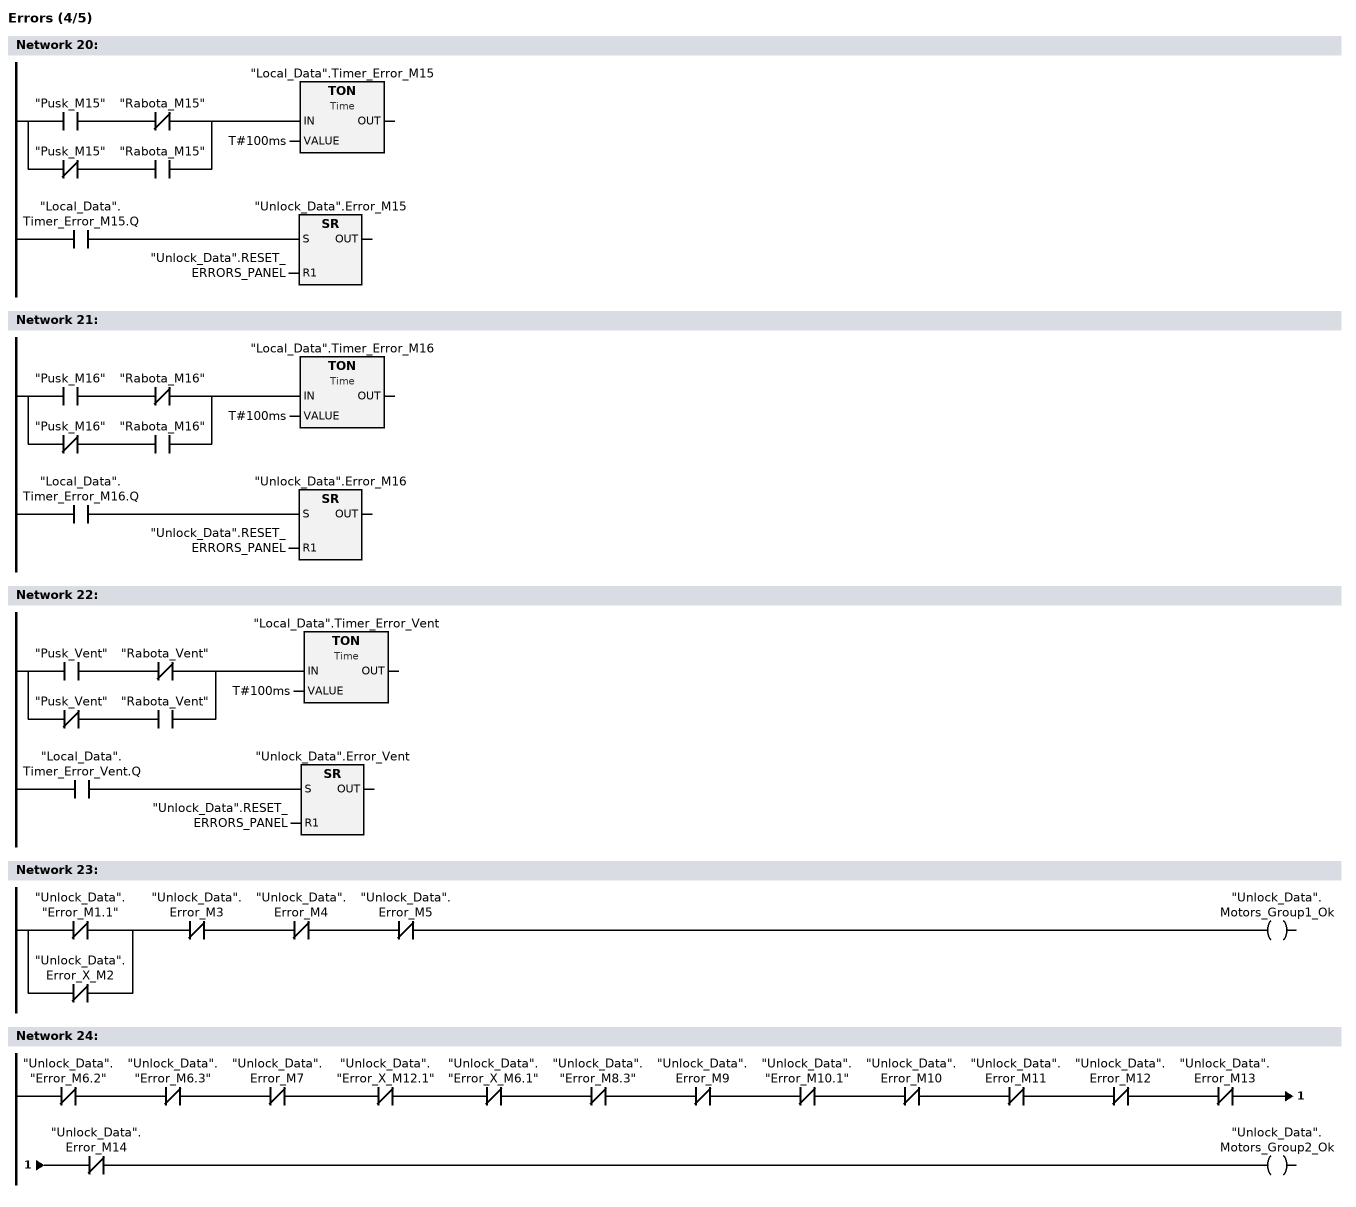
   "Local_Data".Timer_Error_M15.TON(IN := ("Pusk_M15" AND NOT "Rabota_M15") OR (NOT "Pusk_M15" AND "Rabota_M15"), PT := T#100ms);   // TON coil
   IF "Local_Data".Timer_Error_M15.Q THEN
       "Unlock_Data".Error_M15 := TRUE;   // SR flip-flop
   END_IF;
   IF "Unlock_Data".RESET_ERRORS_PANEL THEN "Unlock_Data".Error_M15 := FALSE; END_IF;
END_REGION

REGION Network 21
   "Local_Data".Timer_Error_M16.TON(IN := ("Pusk_M16" AND NOT "Rabota_M16") OR (NOT "Pusk_M16" AND "Rabota_M16"), PT := T#100ms);   // TON coil
   IF "Local_Data".Timer_Error_M16.Q THEN
       "Unlock_Data".Error_M16 := TRUE;   // SR flip-flop
   END_IF;
   IF "Unlock_Data".RESET_ERRORS_PANEL THEN "Unlock_Data".Error_M16 := FALSE; END_IF;
END_REGION

REGION Network 22
   "Local_Data".Timer_Error_Vent.TON(IN := ("Pusk_Vent" AND NOT "Rabota_Vent") OR (NOT "Pusk_Vent" AND "Rabota_Vent"), PT := T#100ms);   // TON coil
   IF "Local_Data".Timer_Error_Vent.Q THEN
       "Unlock_Data".Error_Vent := TRUE;   // SR flip-flop
   END_IF;
   IF "Unlock_Data".RESET_ERRORS_PANEL THEN "Unlock_Data".Error_Vent := FALSE; END_IF;
END_REGION

REGION Network 23
   RUNG wire#powerrail
      I_Contact( "Unlock_Data"."Error_M1.1" )
      wire#w1
      I_Contact( "Unlock_Data".Error_M3 )
      I_Contact( "Unlock_Data".Error_M4 )
      I_Contact( "Unlock_Data".Error_M5 )
      Coil( "Unlock_Data".Motors_Group1_Ok )
   END_RUNG
   RUNG wire#powerrail
      I_Contact( "Unlock_Data".Error_X_M2 )
   END_RUNG wire#w1
   // the same network as SCL:
   "Unlock_Data".Motors_Group1_Ok := (NOT "Unlock_Data"."Error_M1.1" OR NOT "Unlock_Data".Error_X_M2) AND NOT "Unlock_Data".Error_M3 AND NOT "Unlock_Data".Error_M4 AND NOT "Unlock_Data".Error_M5;
END_REGION

REGION Network 24
   RUNG wire#powerrail
      I_Contact( "Unlock_Data"."Error_M6.2" )
      I_Contact( "Unlock_Data"."Error_M6.3" )
      I_Contact( "Unlock_Data".Error_M7 )
      I_Contact( "Unlock_Data"."Error_X_M12.1" )
      I_Contact( "Unlock_Data"."Error_X_M6.1" )
      I_Contact( "Unlock_Data"."Error_M8.3" )
      I_Contact( "Unlock_Data".Error_M9 )
      I_Contact( "Unlock_Data"."Error_M10.1" )
      I_Contact( "Unlock_Data".Error_M10 )
      I_Contact( "Unlock_Data".Error_M11 )
      I_Contact( "Unlock_Data".Error_M12 )
      I_Contact( "Unlock_Data".Error_M13 )
      I_Contact( "Unlock_Data".Error_M14 )
      Coil( "Unlock_Data".Motors_Group2_Ok )
   END_RUNG
   // the same network as SCL:
   "Unlock_Data".Motors_Group2_Ok := NOT "Unlock_Data"."Error_M6.2" AND NOT "Unlock_Data"."Error_M6.3" AND NOT "Unlock_Data".Error_M7 AND NOT "Unlock_Data"."Error_X_M12.1" AND NOT "Unlock_Data"."Error_X_M6.1" AND NOT "Unlock_Data"."Error_M8.3" AND NOT "Unlock_Data".Error_M9 AND NOT "Unlock_Data"."Error_M10.1" AND NOT "Unlock_Data".Error_M10 AND NOT "Unlock_Data".Error_M11 AND NOT "Unlock_Data".Error_M12 AND NOT "Unlock_Data".Error_M13 AND NOT "Unlock_Data".Error_M14;
END_REGION

REGION Network 25
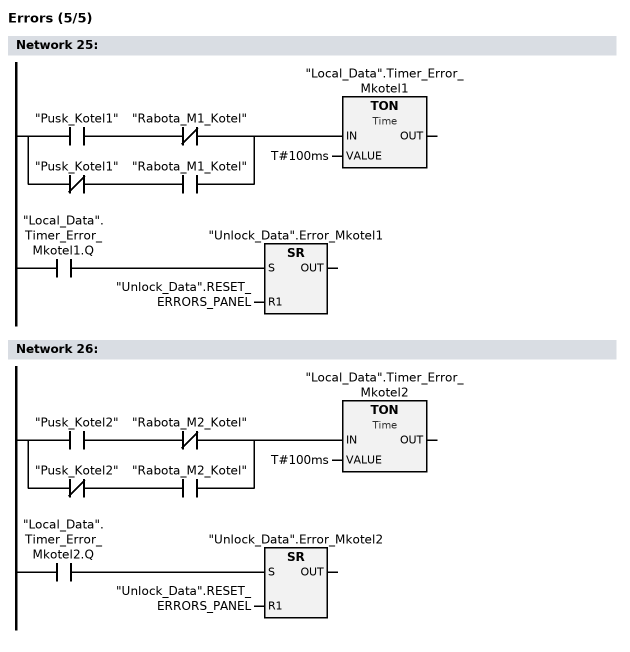
   "Local_Data".Timer_Error_Mkotel1.TON(IN := ("Pusk_Kotel1" AND NOT "Rabota_M1_Kotel") OR (NOT "Pusk_Kotel1" AND "Rabota_M1_Kotel"), PT := T#100ms);   // TON coil
   IF "Local_Data".Timer_Error_Mkotel1.Q THEN
       "Unlock_Data".Error_Mkotel1 := TRUE;   // SR flip-flop
   END_IF;
   IF "Unlock_Data".RESET_ERRORS_PANEL THEN "Unlock_Data".Error_Mkotel1 := FALSE; END_IF;
END_REGION

REGION Network 26
   "Local_Data".Timer_Error_Mkotel2.TON(IN := ("Pusk_Kotel2" AND NOT "Rabota_M2_Kotel") OR (NOT "Pusk_Kotel2" AND "Rabota_M2_Kotel"), PT := T#100ms);   // TON coil
   IF "Local_Data".Timer_Error_Mkotel2.Q THEN
       "Unlock_Data".Error_Mkotel2 := TRUE;   // SR flip-flop
   END_IF;
   IF "Unlock_Data".RESET_ERRORS_PANEL THEN "Unlock_Data".Error_Mkotel2 := FALSE; END_IF;
END_REGION
END_FUNCTION_BLOCK

FUNCTION_BLOCK "Motors"   // FB2, LAD
{ S7_Optimized_Access := 'TRUE' }
VERSION : 0.1
   VAR_TEMP   // added for the SCL form of the ladder/FBD networks
      _w1 : Bool;
   END_VAR
BEGIN

REGION Network 1: Насос М1.1
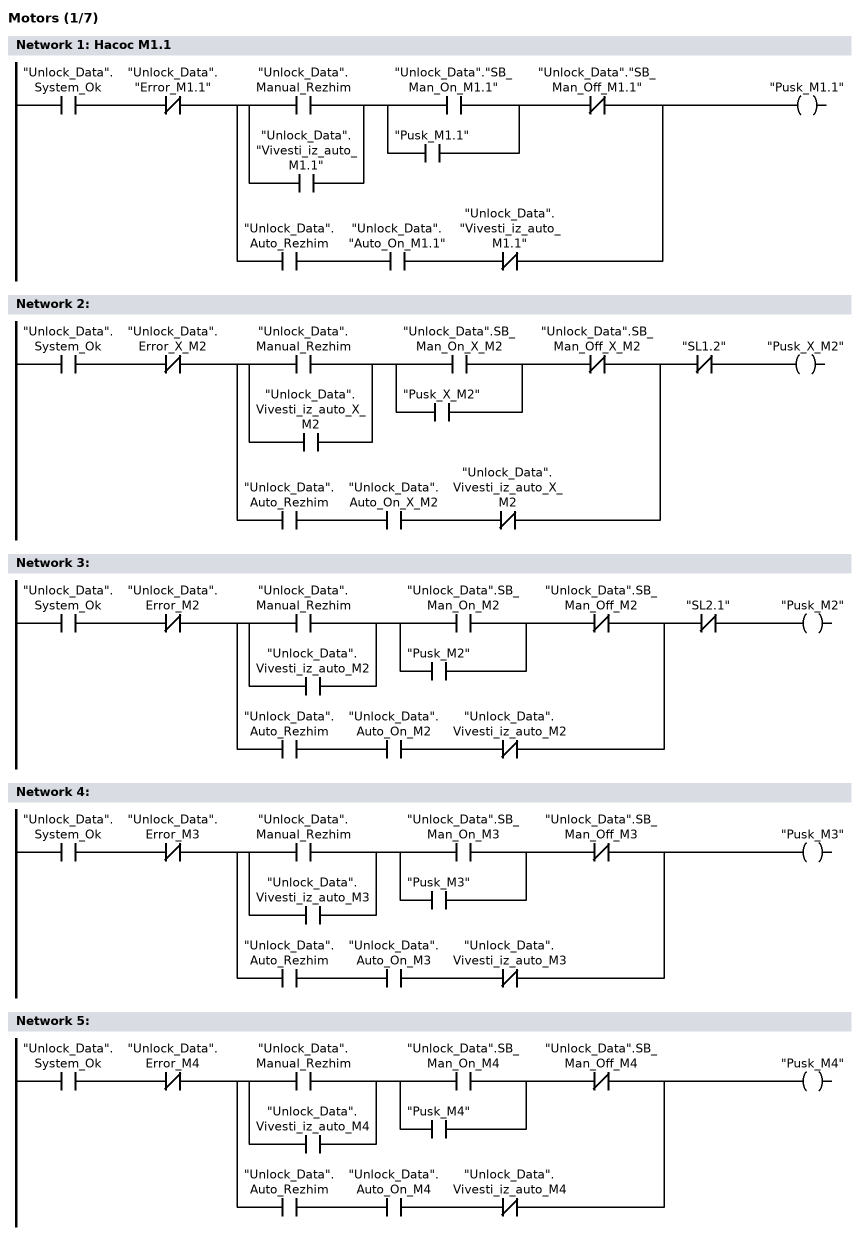
   RUNG wire#powerrail
      Contact( "Unlock_Data".System_Ok )
      I_Contact( "Unlock_Data"."Error_M1.1" )
      wire#w1
      Contact( "Unlock_Data".Manual_Rezhim )
      wire#w2
      Contact( "Unlock_Data"."SB_Man_On_M1.1" )
      wire#w3
      I_Contact( "Unlock_Data"."SB_Man_Off_M1.1" )
      wire#w4
      Coil( "Pusk_M1.1" )
   END_RUNG
   RUNG wire#w1
      Contact( "Unlock_Data"."Vivesti_iz_auto_M1.1" )
   END_RUNG wire#w2
   RUNG wire#w2
      Contact( "Pusk_M1.1" )
   END_RUNG wire#w3
   RUNG wire#w1
      Contact( "Unlock_Data".Auto_Rezhim )
      Contact( "Unlock_Data"."Auto_On_M1.1" )
      I_Contact( "Unlock_Data"."Vivesti_iz_auto_M1.1" )
   END_RUNG wire#w4
   // the same network as SCL:
   "Pusk_M1.1" := "Unlock_Data".System_Ok AND NOT "Unlock_Data"."Error_M1.1" AND ((("Unlock_Data".Manual_Rezhim OR "Unlock_Data"."Vivesti_iz_auto_M1.1") AND ("Unlock_Data"."SB_Man_On_M1.1" OR "Pusk_M1.1") AND NOT "Unlock_Data"."SB_Man_Off_M1.1") OR ("Unlock_Data".Auto_Rezhim AND "Unlock_Data"."Auto_On_M1.1" AND NOT "Unlock_Data"."Vivesti_iz_auto_M1.1"));
END_REGION

REGION Network 2
   RUNG wire#powerrail
      Contact( "Unlock_Data".System_Ok )
      I_Contact( "Unlock_Data".Error_X_M2 )
      wire#w1
      Contact( "Unlock_Data".Manual_Rezhim )
      wire#w2
      Contact( "Unlock_Data".SB_Man_On_X_M2 )
      wire#w3
      I_Contact( "Unlock_Data".SB_Man_Off_X_M2 )
      wire#w4
      I_Contact( "SL1.2" )
      Coil( "Pusk_X_M2" )
   END_RUNG
   RUNG wire#w1
      Contact( "Unlock_Data".Vivesti_iz_auto_X_M2 )
   END_RUNG wire#w2
   RUNG wire#w2
      Contact( "Pusk_X_M2" )
   END_RUNG wire#w3
   RUNG wire#w1
      Contact( "Unlock_Data".Auto_Rezhim )
      Contact( "Unlock_Data".Auto_On_X_M2 )
      I_Contact( "Unlock_Data".Vivesti_iz_auto_X_M2 )
   END_RUNG wire#w4
   // the same network as SCL:
   "Pusk_X_M2" := "Unlock_Data".System_Ok AND NOT "Unlock_Data".Error_X_M2 AND ((("Unlock_Data".Manual_Rezhim OR "Unlock_Data".Vivesti_iz_auto_X_M2) AND ("Unlock_Data".SB_Man_On_X_M2 OR "Pusk_X_M2") AND NOT "Unlock_Data".SB_Man_Off_X_M2) OR ("Unlock_Data".Auto_Rezhim AND "Unlock_Data".Auto_On_X_M2 AND NOT "Unlock_Data".Vivesti_iz_auto_X_M2)) AND NOT "SL1.2";
END_REGION

REGION Network 3
   RUNG wire#powerrail
      Contact( "Unlock_Data".System_Ok )
      I_Contact( "Unlock_Data".Error_M2 )
      wire#w1
      Contact( "Unlock_Data".Manual_Rezhim )
      wire#w2
      Contact( "Unlock_Data".SB_Man_On_M2 )
      wire#w3
      I_Contact( "Unlock_Data".SB_Man_Off_M2 )
      wire#w4
      I_Contact( "SL2.1" )
      Coil( "Pusk_M2" )
   END_RUNG
   RUNG wire#w1
      Contact( "Unlock_Data".Vivesti_iz_auto_M2 )
   END_RUNG wire#w2
   RUNG wire#w2
      Contact( "Pusk_M2" )
   END_RUNG wire#w3
   RUNG wire#w1
      Contact( "Unlock_Data".Auto_Rezhim )
      Contact( "Unlock_Data".Auto_On_M2 )
      I_Contact( "Unlock_Data".Vivesti_iz_auto_M2 )
   END_RUNG wire#w4
   // the same network as SCL:
   "Pusk_M2" := "Unlock_Data".System_Ok AND NOT "Unlock_Data".Error_M2 AND ((("Unlock_Data".Manual_Rezhim OR "Unlock_Data".Vivesti_iz_auto_M2) AND ("Unlock_Data".SB_Man_On_M2 OR "Pusk_M2") AND NOT "Unlock_Data".SB_Man_Off_M2) OR ("Unlock_Data".Auto_Rezhim AND "Unlock_Data".Auto_On_M2 AND NOT "Unlock_Data".Vivesti_iz_auto_M2)) AND NOT "SL2.1";
END_REGION

REGION Network 4
   RUNG wire#powerrail
      Contact( "Unlock_Data".System_Ok )
      I_Contact( "Unlock_Data".Error_M3 )
      wire#w1
      Contact( "Unlock_Data".Manual_Rezhim )
      wire#w2
      Contact( "Unlock_Data".SB_Man_On_M3 )
      wire#w3
      I_Contact( "Unlock_Data".SB_Man_Off_M3 )
      wire#w4
      Coil( "Pusk_M3" )
   END_RUNG
   RUNG wire#w1
      Contact( "Unlock_Data".Vivesti_iz_auto_M3 )
   END_RUNG wire#w2
   RUNG wire#w2
      Contact( "Pusk_M3" )
   END_RUNG wire#w3
   RUNG wire#w1
      Contact( "Unlock_Data".Auto_Rezhim )
      Contact( "Unlock_Data".Auto_On_M3 )
      I_Contact( "Unlock_Data".Vivesti_iz_auto_M3 )
   END_RUNG wire#w4
   // the same network as SCL:
   "Pusk_M3" := "Unlock_Data".System_Ok AND NOT "Unlock_Data".Error_M3 AND ((("Unlock_Data".Manual_Rezhim OR "Unlock_Data".Vivesti_iz_auto_M3) AND ("Unlock_Data".SB_Man_On_M3 OR "Pusk_M3") AND NOT "Unlock_Data".SB_Man_Off_M3) OR ("Unlock_Data".Auto_Rezhim AND "Unlock_Data".Auto_On_M3 AND NOT "Unlock_Data".Vivesti_iz_auto_M3));
END_REGION

REGION Network 5
   RUNG wire#powerrail
      Contact( "Unlock_Data".System_Ok )
      I_Contact( "Unlock_Data".Error_M4 )
      wire#w1
      Contact( "Unlock_Data".Manual_Rezhim )
      wire#w2
      Contact( "Unlock_Data".SB_Man_On_M4 )
      wire#w3
      I_Contact( "Unlock_Data".SB_Man_Off_M4 )
      wire#w4
      Coil( "Pusk_M4" )
   END_RUNG
   RUNG wire#w1
      Contact( "Unlock_Data".Vivesti_iz_auto_M4 )
   END_RUNG wire#w2
   RUNG wire#w2
      Contact( "Pusk_M4" )
   END_RUNG wire#w3
   RUNG wire#w1
      Contact( "Unlock_Data".Auto_Rezhim )
      Contact( "Unlock_Data".Auto_On_M4 )
      I_Contact( "Unlock_Data".Vivesti_iz_auto_M4 )
   END_RUNG wire#w4
   // the same network as SCL:
   "Pusk_M4" := "Unlock_Data".System_Ok AND NOT "Unlock_Data".Error_M4 AND ((("Unlock_Data".Manual_Rezhim OR "Unlock_Data".Vivesti_iz_auto_M4) AND ("Unlock_Data".SB_Man_On_M4 OR "Pusk_M4") AND NOT "Unlock_Data".SB_Man_Off_M4) OR ("Unlock_Data".Auto_Rezhim AND "Unlock_Data".Auto_On_M4 AND NOT "Unlock_Data".Vivesti_iz_auto_M4));
END_REGION

REGION Network 6
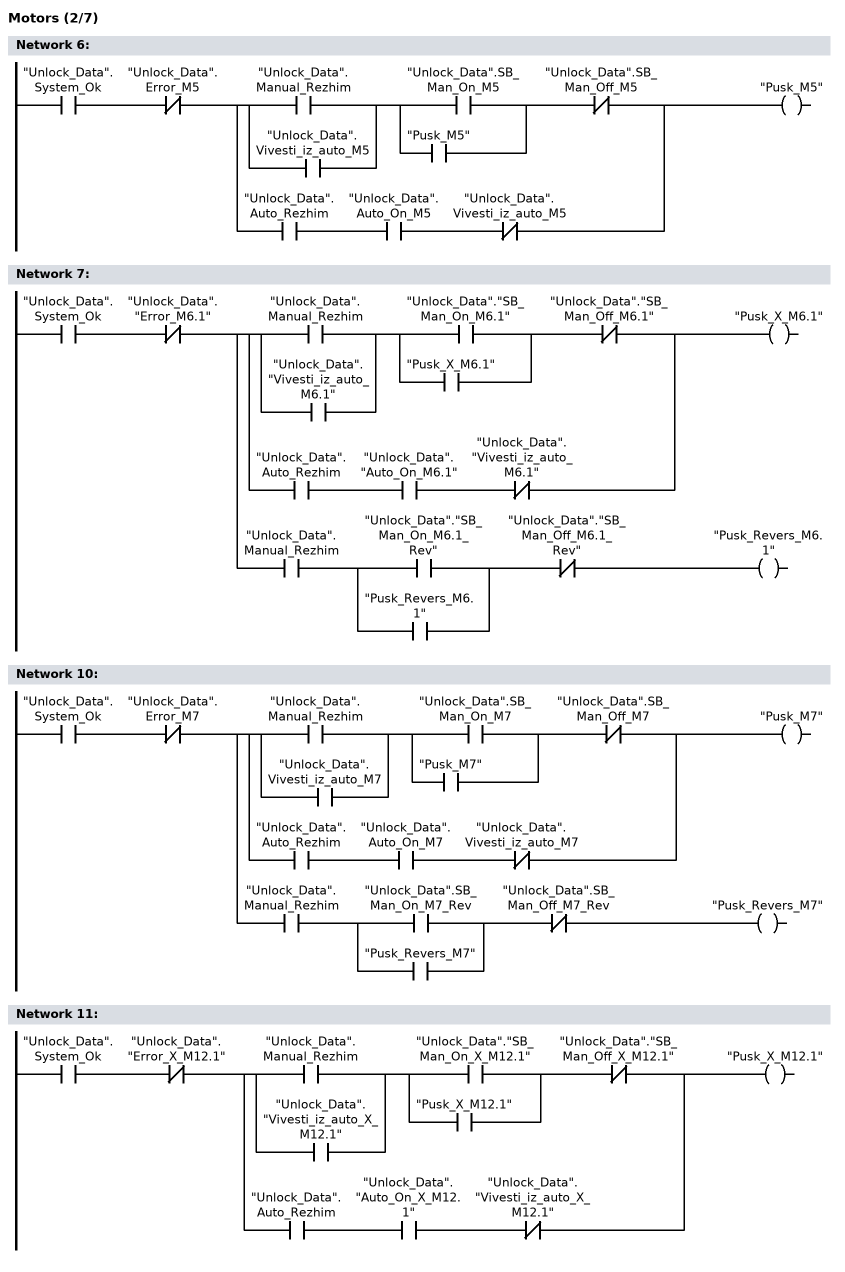
   RUNG wire#powerrail
      Contact( "Unlock_Data".System_Ok )
      I_Contact( "Unlock_Data".Error_M5 )
      wire#w1
      Contact( "Unlock_Data".Manual_Rezhim )
      wire#w2
      Contact( "Unlock_Data".SB_Man_On_M5 )
      wire#w3
      I_Contact( "Unlock_Data".SB_Man_Off_M5 )
      wire#w4
      Coil( "Pusk_M5" )
   END_RUNG
   RUNG wire#w1
      Contact( "Unlock_Data".Vivesti_iz_auto_M5 )
   END_RUNG wire#w2
   RUNG wire#w2
      Contact( "Pusk_M5" )
   END_RUNG wire#w3
   RUNG wire#w1
      Contact( "Unlock_Data".Auto_Rezhim )
      Contact( "Unlock_Data".Auto_On_M5 )
      I_Contact( "Unlock_Data".Vivesti_iz_auto_M5 )
   END_RUNG wire#w4
   // the same network as SCL:
   "Pusk_M5" := "Unlock_Data".System_Ok AND NOT "Unlock_Data".Error_M5 AND ((("Unlock_Data".Manual_Rezhim OR "Unlock_Data".Vivesti_iz_auto_M5) AND ("Unlock_Data".SB_Man_On_M5 OR "Pusk_M5") AND NOT "Unlock_Data".SB_Man_Off_M5) OR ("Unlock_Data".Auto_Rezhim AND "Unlock_Data".Auto_On_M5 AND NOT "Unlock_Data".Vivesti_iz_auto_M5));
END_REGION

REGION Network 7
   RUNG wire#powerrail
      Contact( "Unlock_Data".System_Ok )
      I_Contact( "Unlock_Data"."Error_M6.1" )
      wire#w1
      Contact( "Unlock_Data".Manual_Rezhim )
      wire#w2
      Contact( "Unlock_Data"."SB_Man_On_M6.1" )
      wire#w3
      I_Contact( "Unlock_Data"."SB_Man_Off_M6.1" )
      wire#w4
      Coil( "Pusk_X_M6.1" )
   END_RUNG
   RUNG wire#w1
      Contact( "Unlock_Data"."Vivesti_iz_auto_M6.1" )
   END_RUNG wire#w2
   RUNG wire#w2
      Contact( "Pusk_X_M6.1" )
   END_RUNG wire#w3
   RUNG wire#w1
      Contact( "Unlock_Data".Auto_Rezhim )
      Contact( "Unlock_Data"."Auto_On_M6.1" )
      I_Contact( "Unlock_Data"."Vivesti_iz_auto_M6.1" )
   END_RUNG wire#w4
   RUNG wire#w1
      Contact( "Unlock_Data".Manual_Rezhim )
      wire#w5
      Contact( "Unlock_Data"."SB_Man_On_M6.1_Rev" )
      wire#w6
      I_Contact( "Unlock_Data"."SB_Man_Off_M6.1_Rev" )
      Coil( "Pusk_Revers_M6.1" )
   END_RUNG
   RUNG wire#w5
      Contact( "Pusk_Revers_M6.1" )
   END_RUNG wire#w6
   // the same network as SCL:
   #_w1 := "Unlock_Data".System_Ok AND NOT "Unlock_Data"."Error_M6.1";
   "Pusk_X_M6.1" := #_w1 AND ((("Unlock_Data".Manual_Rezhim OR "Unlock_Data"."Vivesti_iz_auto_M6.1") AND ("Unlock_Data"."SB_Man_On_M6.1" OR "Pusk_X_M6.1") AND NOT "Unlock_Data"."SB_Man_Off_M6.1") OR ("Unlock_Data".Auto_Rezhim AND "Unlock_Data"."Auto_On_M6.1" AND NOT "Unlock_Data"."Vivesti_iz_auto_M6.1"));
   "Pusk_Revers_M6.1" := #_w1 AND "Unlock_Data".Manual_Rezhim AND ("Unlock_Data"."SB_Man_On_M6.1_Rev" OR "Pusk_Revers_M6.1") AND NOT "Unlock_Data"."SB_Man_Off_M6.1_Rev";
END_REGION

REGION Network 10
   RUNG wire#powerrail
      Contact( "Unlock_Data".System_Ok )
      I_Contact( "Unlock_Data".Error_M7 )
      wire#w1
      Contact( "Unlock_Data".Manual_Rezhim )
      wire#w2
      Contact( "Unlock_Data".SB_Man_On_M7 )
      wire#w3
      I_Contact( "Unlock_Data".SB_Man_Off_M7 )
      wire#w4
      Coil( "Pusk_M7" )
   END_RUNG
   RUNG wire#w1
      Contact( "Unlock_Data".Vivesti_iz_auto_M7 )
   END_RUNG wire#w2
   RUNG wire#w2
      Contact( "Pusk_M7" )
   END_RUNG wire#w3
   RUNG wire#w1
      Contact( "Unlock_Data".Auto_Rezhim )
      Contact( "Unlock_Data".Auto_On_M7 )
      I_Contact( "Unlock_Data".Vivesti_iz_auto_M7 )
   END_RUNG wire#w4
   RUNG wire#w1
      Contact( "Unlock_Data".Manual_Rezhim )
      wire#w5
      Contact( "Unlock_Data".SB_Man_On_M7_Rev )
      wire#w6
      I_Contact( "Unlock_Data".SB_Man_Off_M7_Rev )
      Coil( "Pusk_Revers_M7" )
   END_RUNG
   RUNG wire#w5
      Contact( "Pusk_Revers_M7" )
   END_RUNG wire#w6
   // the same network as SCL:
   #_w1 := "Unlock_Data".System_Ok AND NOT "Unlock_Data".Error_M7;
   "Pusk_M7" := #_w1 AND ((("Unlock_Data".Manual_Rezhim OR "Unlock_Data".Vivesti_iz_auto_M7) AND ("Unlock_Data".SB_Man_On_M7 OR "Pusk_M7") AND NOT "Unlock_Data".SB_Man_Off_M7) OR ("Unlock_Data".Auto_Rezhim AND "Unlock_Data".Auto_On_M7 AND NOT "Unlock_Data".Vivesti_iz_auto_M7));
   "Pusk_Revers_M7" := #_w1 AND "Unlock_Data".Manual_Rezhim AND ("Unlock_Data".SB_Man_On_M7_Rev OR "Pusk_Revers_M7") AND NOT "Unlock_Data".SB_Man_Off_M7_Rev;
END_REGION

REGION Network 11
   RUNG wire#powerrail
      Contact( "Unlock_Data".System_Ok )
      I_Contact( "Unlock_Data"."Error_X_M12.1" )
      wire#w1
      Contact( "Unlock_Data".Manual_Rezhim )
      wire#w2
      Contact( "Unlock_Data"."SB_Man_On_X_M12.1" )
      wire#w3
      I_Contact( "Unlock_Data"."SB_Man_Off_X_M12.1" )
      wire#w4
      Coil( "Pusk_X_M12.1" )
   END_RUNG
   RUNG wire#w1
      Contact( "Unlock_Data"."Vivesti_iz_auto_X_M12.1" )
   END_RUNG wire#w2
   RUNG wire#w2
      Contact( "Pusk_X_M12.1" )
   END_RUNG wire#w3
   RUNG wire#w1
      Contact( "Unlock_Data".Auto_Rezhim )
      Contact( "Unlock_Data"."Auto_On_X_M12.1" )
      I_Contact( "Unlock_Data"."Vivesti_iz_auto_X_M12.1" )
   END_RUNG wire#w4
   // the same network as SCL:
   "Pusk_X_M12.1" := "Unlock_Data".System_Ok AND NOT "Unlock_Data"."Error_X_M12.1" AND ((("Unlock_Data".Manual_Rezhim OR "Unlock_Data"."Vivesti_iz_auto_X_M12.1") AND ("Unlock_Data"."SB_Man_On_X_M12.1" OR "Pusk_X_M12.1") AND NOT "Unlock_Data"."SB_Man_Off_X_M12.1") OR ("Unlock_Data".Auto_Rezhim AND "Unlock_Data"."Auto_On_X_M12.1" AND NOT "Unlock_Data"."Vivesti_iz_auto_X_M12.1"));
END_REGION

REGION Network 12
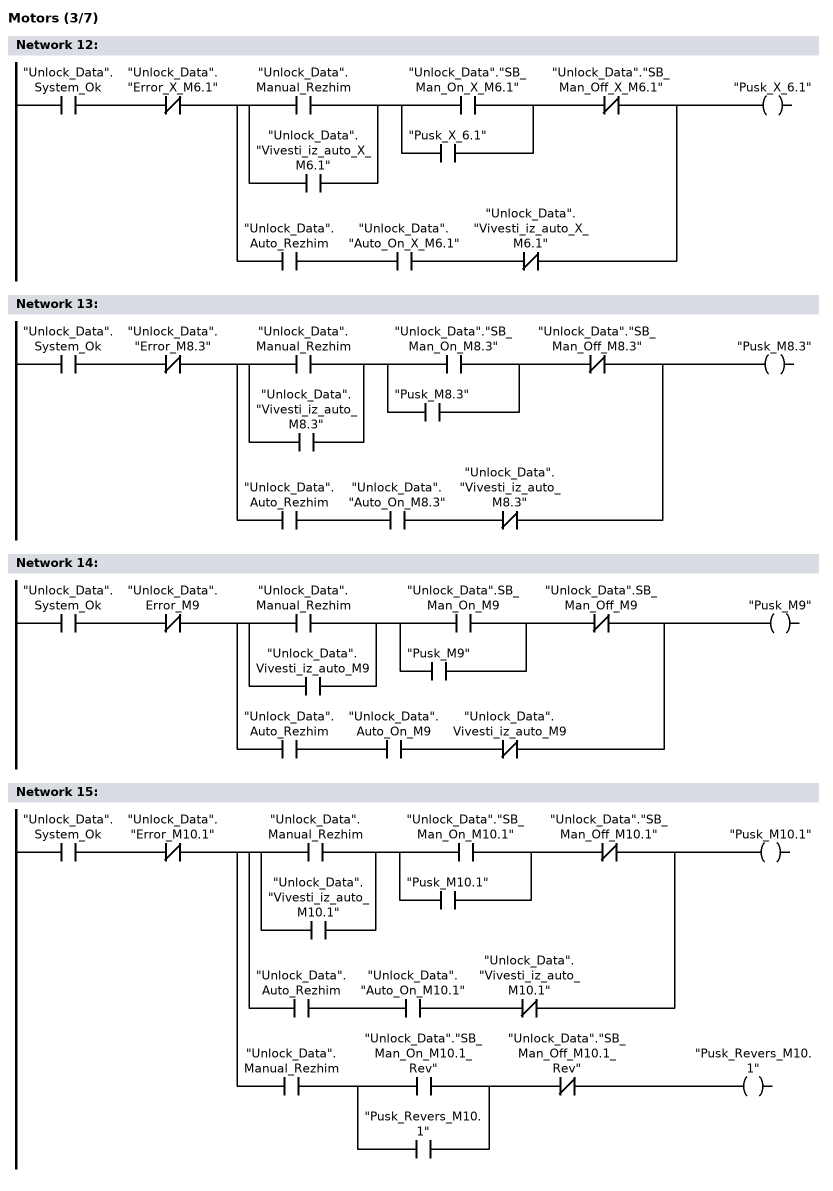
   RUNG wire#powerrail
      Contact( "Unlock_Data".System_Ok )
      I_Contact( "Unlock_Data"."Error_X_M6.1" )
      wire#w1
      Contact( "Unlock_Data".Manual_Rezhim )
      wire#w2
      Contact( "Unlock_Data"."SB_Man_On_X_M6.1" )
      wire#w3
      I_Contact( "Unlock_Data"."SB_Man_Off_X_M6.1" )
      wire#w4
      Coil( "Pusk_X_6.1" )
   END_RUNG
   RUNG wire#w1
      Contact( "Unlock_Data"."Vivesti_iz_auto_X_M6.1" )
   END_RUNG wire#w2
   RUNG wire#w2
      Contact( "Pusk_X_6.1" )
   END_RUNG wire#w3
   RUNG wire#w1
      Contact( "Unlock_Data".Auto_Rezhim )
      Contact( "Unlock_Data"."Auto_On_X_M6.1" )
      I_Contact( "Unlock_Data"."Vivesti_iz_auto_X_M6.1" )
   END_RUNG wire#w4
   // the same network as SCL:
   "Pusk_X_6.1" := "Unlock_Data".System_Ok AND NOT "Unlock_Data"."Error_X_M6.1" AND ((("Unlock_Data".Manual_Rezhim OR "Unlock_Data"."Vivesti_iz_auto_X_M6.1") AND ("Unlock_Data"."SB_Man_On_X_M6.1" OR "Pusk_X_6.1") AND NOT "Unlock_Data"."SB_Man_Off_X_M6.1") OR ("Unlock_Data".Auto_Rezhim AND "Unlock_Data"."Auto_On_X_M6.1" AND NOT "Unlock_Data"."Vivesti_iz_auto_X_M6.1"));
END_REGION

REGION Network 13
   RUNG wire#powerrail
      Contact( "Unlock_Data".System_Ok )
      I_Contact( "Unlock_Data"."Error_M8.3" )
      wire#w1
      Contact( "Unlock_Data".Manual_Rezhim )
      wire#w2
      Contact( "Unlock_Data"."SB_Man_On_M8.3" )
      wire#w3
      I_Contact( "Unlock_Data"."SB_Man_Off_M8.3" )
      wire#w4
      Coil( "Pusk_M8.3" )
   END_RUNG
   RUNG wire#w1
      Contact( "Unlock_Data"."Vivesti_iz_auto_M8.3" )
   END_RUNG wire#w2
   RUNG wire#w2
      Contact( "Pusk_M8.3" )
   END_RUNG wire#w3
   RUNG wire#w1
      Contact( "Unlock_Data".Auto_Rezhim )
      Contact( "Unlock_Data"."Auto_On_M8.3" )
      I_Contact( "Unlock_Data"."Vivesti_iz_auto_M8.3" )
   END_RUNG wire#w4
   // the same network as SCL:
   "Pusk_M8.3" := "Unlock_Data".System_Ok AND NOT "Unlock_Data"."Error_M8.3" AND ((("Unlock_Data".Manual_Rezhim OR "Unlock_Data"."Vivesti_iz_auto_M8.3") AND ("Unlock_Data"."SB_Man_On_M8.3" OR "Pusk_M8.3") AND NOT "Unlock_Data"."SB_Man_Off_M8.3") OR ("Unlock_Data".Auto_Rezhim AND "Unlock_Data"."Auto_On_M8.3" AND NOT "Unlock_Data"."Vivesti_iz_auto_M8.3"));
END_REGION

REGION Network 14
   RUNG wire#powerrail
      Contact( "Unlock_Data".System_Ok )
      I_Contact( "Unlock_Data".Error_M9 )
      wire#w1
      Contact( "Unlock_Data".Manual_Rezhim )
      wire#w2
      Contact( "Unlock_Data".SB_Man_On_M9 )
      wire#w3
      I_Contact( "Unlock_Data".SB_Man_Off_M9 )
      wire#w4
      Coil( "Pusk_M9" )
   END_RUNG
   RUNG wire#w1
      Contact( "Unlock_Data".Vivesti_iz_auto_M9 )
   END_RUNG wire#w2
   RUNG wire#w2
      Contact( "Pusk_M9" )
   END_RUNG wire#w3
   RUNG wire#w1
      Contact( "Unlock_Data".Auto_Rezhim )
      Contact( "Unlock_Data".Auto_On_M9 )
      I_Contact( "Unlock_Data".Vivesti_iz_auto_M9 )
   END_RUNG wire#w4
   // the same network as SCL:
   "Pusk_M9" := "Unlock_Data".System_Ok AND NOT "Unlock_Data".Error_M9 AND ((("Unlock_Data".Manual_Rezhim OR "Unlock_Data".Vivesti_iz_auto_M9) AND ("Unlock_Data".SB_Man_On_M9 OR "Pusk_M9") AND NOT "Unlock_Data".SB_Man_Off_M9) OR ("Unlock_Data".Auto_Rezhim AND "Unlock_Data".Auto_On_M9 AND NOT "Unlock_Data".Vivesti_iz_auto_M9));
END_REGION

REGION Network 15
   RUNG wire#powerrail
      Contact( "Unlock_Data".System_Ok )
      I_Contact( "Unlock_Data"."Error_M10.1" )
      wire#w1
      Contact( "Unlock_Data".Manual_Rezhim )
      wire#w2
      Contact( "Unlock_Data"."SB_Man_On_M10.1" )
      wire#w3
      I_Contact( "Unlock_Data"."SB_Man_Off_M10.1" )
      wire#w4
      Coil( "Pusk_M10.1" )
   END_RUNG
   RUNG wire#w1
      Contact( "Unlock_Data"."Vivesti_iz_auto_M10.1" )
   END_RUNG wire#w2
   RUNG wire#w2
      Contact( "Pusk_M10.1" )
   END_RUNG wire#w3
   RUNG wire#w1
      Contact( "Unlock_Data".Auto_Rezhim )
      Contact( "Unlock_Data"."Auto_On_M10.1" )
      I_Contact( "Unlock_Data"."Vivesti_iz_auto_M10.1" )
   END_RUNG wire#w4
   RUNG wire#w1
      Contact( "Unlock_Data".Manual_Rezhim )
      wire#w5
      Contact( "Unlock_Data"."SB_Man_On_M10.1_Rev" )
      wire#w6
      I_Contact( "Unlock_Data"."SB_Man_Off_M10.1_Rev" )
      Coil( "Pusk_Revers_M10.1" )
   END_RUNG
   RUNG wire#w5
      Contact( "Pusk_Revers_M10.1" )
   END_RUNG wire#w6
   // the same network as SCL:
   #_w1 := "Unlock_Data".System_Ok AND NOT "Unlock_Data"."Error_M10.1";
   "Pusk_M10.1" := #_w1 AND ((("Unlock_Data".Manual_Rezhim OR "Unlock_Data"."Vivesti_iz_auto_M10.1") AND ("Unlock_Data"."SB_Man_On_M10.1" OR "Pusk_M10.1") AND NOT "Unlock_Data"."SB_Man_Off_M10.1") OR ("Unlock_Data".Auto_Rezhim AND "Unlock_Data"."Auto_On_M10.1" AND NOT "Unlock_Data"."Vivesti_iz_auto_M10.1"));
   "Pusk_Revers_M10.1" := #_w1 AND "Unlock_Data".Manual_Rezhim AND ("Unlock_Data"."SB_Man_On_M10.1_Rev" OR "Pusk_Revers_M10.1") AND NOT "Unlock_Data"."SB_Man_Off_M10.1_Rev";
END_REGION

REGION Network 16
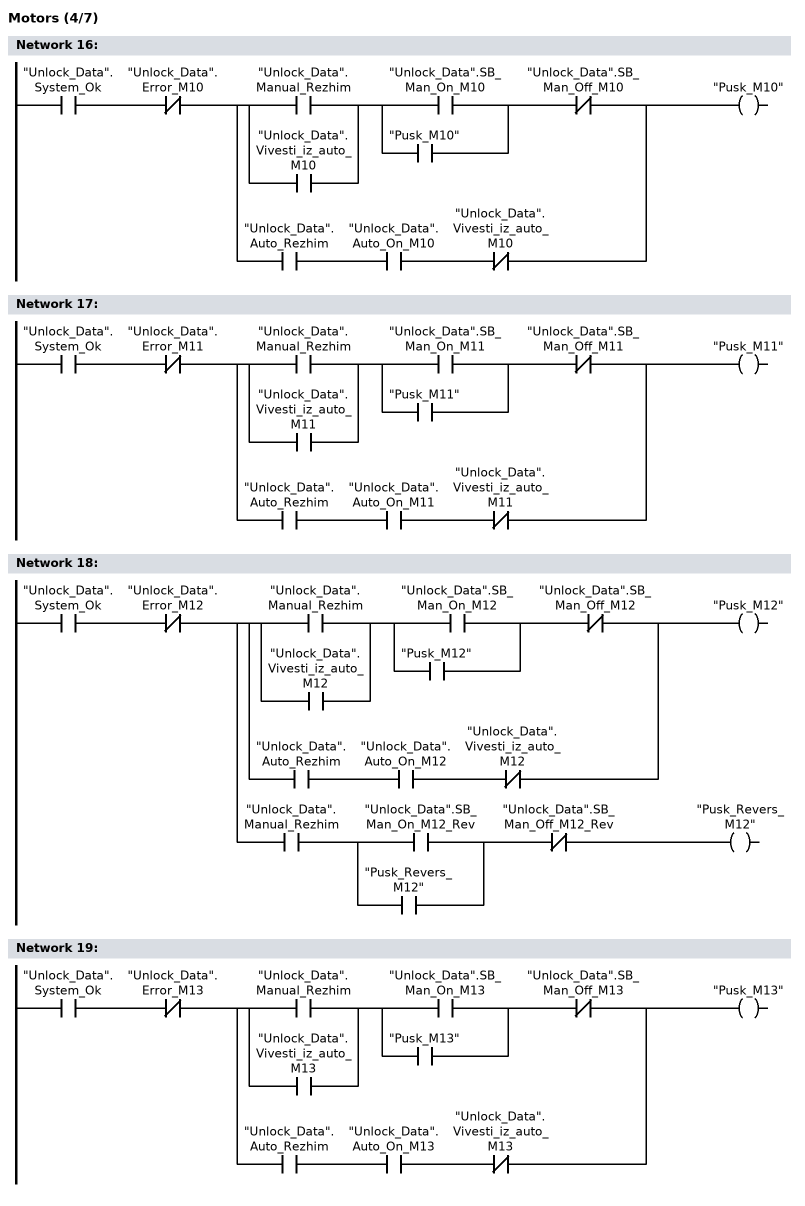
   RUNG wire#powerrail
      Contact( "Unlock_Data".System_Ok )
      I_Contact( "Unlock_Data".Error_M10 )
      wire#w1
      Contact( "Unlock_Data".Manual_Rezhim )
      wire#w2
      Contact( "Unlock_Data".SB_Man_On_M10 )
      wire#w3
      I_Contact( "Unlock_Data".SB_Man_Off_M10 )
      wire#w4
      Coil( "Pusk_M10" )
   END_RUNG
   RUNG wire#w1
      Contact( "Unlock_Data".Vivesti_iz_auto_M10 )
   END_RUNG wire#w2
   RUNG wire#w2
      Contact( "Pusk_M10" )
   END_RUNG wire#w3
   RUNG wire#w1
      Contact( "Unlock_Data".Auto_Rezhim )
      Contact( "Unlock_Data".Auto_On_M10 )
      I_Contact( "Unlock_Data".Vivesti_iz_auto_M10 )
   END_RUNG wire#w4
   // the same network as SCL:
   "Pusk_M10" := "Unlock_Data".System_Ok AND NOT "Unlock_Data".Error_M10 AND ((("Unlock_Data".Manual_Rezhim OR "Unlock_Data".Vivesti_iz_auto_M10) AND ("Unlock_Data".SB_Man_On_M10 OR "Pusk_M10") AND NOT "Unlock_Data".SB_Man_Off_M10) OR ("Unlock_Data".Auto_Rezhim AND "Unlock_Data".Auto_On_M10 AND NOT "Unlock_Data".Vivesti_iz_auto_M10));
END_REGION

REGION Network 17
   RUNG wire#powerrail
      Contact( "Unlock_Data".System_Ok )
      I_Contact( "Unlock_Data".Error_M11 )
      wire#w1
      Contact( "Unlock_Data".Manual_Rezhim )
      wire#w2
      Contact( "Unlock_Data".SB_Man_On_M11 )
      wire#w3
      I_Contact( "Unlock_Data".SB_Man_Off_M11 )
      wire#w4
      Coil( "Pusk_M11" )
   END_RUNG
   RUNG wire#w1
      Contact( "Unlock_Data".Vivesti_iz_auto_M11 )
   END_RUNG wire#w2
   RUNG wire#w2
      Contact( "Pusk_M11" )
   END_RUNG wire#w3
   RUNG wire#w1
      Contact( "Unlock_Data".Auto_Rezhim )
      Contact( "Unlock_Data".Auto_On_M11 )
      I_Contact( "Unlock_Data".Vivesti_iz_auto_M11 )
   END_RUNG wire#w4
   // the same network as SCL:
   "Pusk_M11" := "Unlock_Data".System_Ok AND NOT "Unlock_Data".Error_M11 AND ((("Unlock_Data".Manual_Rezhim OR "Unlock_Data".Vivesti_iz_auto_M11) AND ("Unlock_Data".SB_Man_On_M11 OR "Pusk_M11") AND NOT "Unlock_Data".SB_Man_Off_M11) OR ("Unlock_Data".Auto_Rezhim AND "Unlock_Data".Auto_On_M11 AND NOT "Unlock_Data".Vivesti_iz_auto_M11));
END_REGION

REGION Network 18
   RUNG wire#powerrail
      Contact( "Unlock_Data".System_Ok )
      I_Contact( "Unlock_Data".Error_M12 )
      wire#w1
      Contact( "Unlock_Data".Manual_Rezhim )
      wire#w2
      Contact( "Unlock_Data".SB_Man_On_M12 )
      wire#w3
      I_Contact( "Unlock_Data".SB_Man_Off_M12 )
      wire#w4
      Coil( "Pusk_M12" )
   END_RUNG
   RUNG wire#w1
      Contact( "Unlock_Data".Vivesti_iz_auto_M12 )
   END_RUNG wire#w2
   RUNG wire#w2
      Contact( "Pusk_M12" )
   END_RUNG wire#w3
   RUNG wire#w1
      Contact( "Unlock_Data".Auto_Rezhim )
      Contact( "Unlock_Data".Auto_On_M12 )
      I_Contact( "Unlock_Data".Vivesti_iz_auto_M12 )
   END_RUNG wire#w4
   RUNG wire#w1
      Contact( "Unlock_Data".Manual_Rezhim )
      wire#w5
      Contact( "Unlock_Data".SB_Man_On_M12_Rev )
      wire#w6
      I_Contact( "Unlock_Data".SB_Man_Off_M12_Rev )
      Coil( "Pusk_Revers_M12" )
   END_RUNG
   RUNG wire#w5
      Contact( "Pusk_Revers_M12" )
   END_RUNG wire#w6
   // the same network as SCL:
   #_w1 := "Unlock_Data".System_Ok AND NOT "Unlock_Data".Error_M12;
   "Pusk_M12" := #_w1 AND ((("Unlock_Data".Manual_Rezhim OR "Unlock_Data".Vivesti_iz_auto_M12) AND ("Unlock_Data".SB_Man_On_M12 OR "Pusk_M12") AND NOT "Unlock_Data".SB_Man_Off_M12) OR ("Unlock_Data".Auto_Rezhim AND "Unlock_Data".Auto_On_M12 AND NOT "Unlock_Data".Vivesti_iz_auto_M12));
   "Pusk_Revers_M12" := #_w1 AND "Unlock_Data".Manual_Rezhim AND ("Unlock_Data".SB_Man_On_M12_Rev OR "Pusk_Revers_M12") AND NOT "Unlock_Data".SB_Man_Off_M12_Rev;
END_REGION

REGION Network 19
   RUNG wire#powerrail
      Contact( "Unlock_Data".System_Ok )
      I_Contact( "Unlock_Data".Error_M13 )
      wire#w1
      Contact( "Unlock_Data".Manual_Rezhim )
      wire#w2
      Contact( "Unlock_Data".SB_Man_On_M13 )
      wire#w3
      I_Contact( "Unlock_Data".SB_Man_Off_M13 )
      wire#w4
      Coil( "Pusk_M13" )
   END_RUNG
   RUNG wire#w1
      Contact( "Unlock_Data".Vivesti_iz_auto_M13 )
   END_RUNG wire#w2
   RUNG wire#w2
      Contact( "Pusk_M13" )
   END_RUNG wire#w3
   RUNG wire#w1
      Contact( "Unlock_Data".Auto_Rezhim )
      Contact( "Unlock_Data".Auto_On_M13 )
      I_Contact( "Unlock_Data".Vivesti_iz_auto_M13 )
   END_RUNG wire#w4
   // the same network as SCL:
   "Pusk_M13" := "Unlock_Data".System_Ok AND NOT "Unlock_Data".Error_M13 AND ((("Unlock_Data".Manual_Rezhim OR "Unlock_Data".Vivesti_iz_auto_M13) AND ("Unlock_Data".SB_Man_On_M13 OR "Pusk_M13") AND NOT "Unlock_Data".SB_Man_Off_M13) OR ("Unlock_Data".Auto_Rezhim AND "Unlock_Data".Auto_On_M13 AND NOT "Unlock_Data".Vivesti_iz_auto_M13));
END_REGION

REGION Network 20
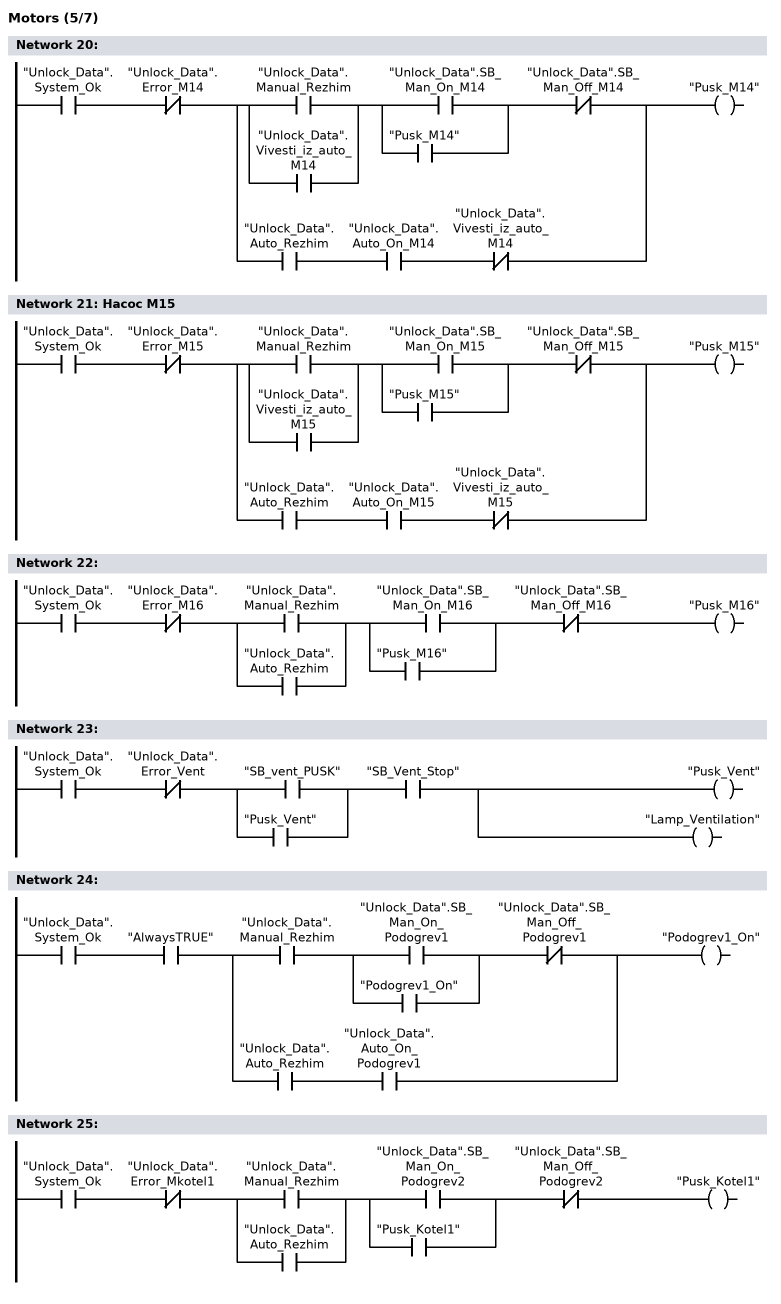
   RUNG wire#powerrail
      Contact( "Unlock_Data".System_Ok )
      I_Contact( "Unlock_Data".Error_M14 )
      wire#w1
      Contact( "Unlock_Data".Manual_Rezhim )
      wire#w2
      Contact( "Unlock_Data".SB_Man_On_M14 )
      wire#w3
      I_Contact( "Unlock_Data".SB_Man_Off_M14 )
      wire#w4
      Coil( "Pusk_M14" )
   END_RUNG
   RUNG wire#w1
      Contact( "Unlock_Data".Vivesti_iz_auto_M14 )
   END_RUNG wire#w2
   RUNG wire#w2
      Contact( "Pusk_M14" )
   END_RUNG wire#w3
   RUNG wire#w1
      Contact( "Unlock_Data".Auto_Rezhim )
      Contact( "Unlock_Data".Auto_On_M14 )
      I_Contact( "Unlock_Data".Vivesti_iz_auto_M14 )
   END_RUNG wire#w4
   // the same network as SCL:
   "Pusk_M14" := "Unlock_Data".System_Ok AND NOT "Unlock_Data".Error_M14 AND ((("Unlock_Data".Manual_Rezhim OR "Unlock_Data".Vivesti_iz_auto_M14) AND ("Unlock_Data".SB_Man_On_M14 OR "Pusk_M14") AND NOT "Unlock_Data".SB_Man_Off_M14) OR ("Unlock_Data".Auto_Rezhim AND "Unlock_Data".Auto_On_M14 AND NOT "Unlock_Data".Vivesti_iz_auto_M14));
END_REGION

REGION Network 21: Насос М15
   RUNG wire#powerrail
      Contact( "Unlock_Data".System_Ok )
      I_Contact( "Unlock_Data".Error_M15 )
      wire#w1
      Contact( "Unlock_Data".Manual_Rezhim )
      wire#w2
      Contact( "Unlock_Data".SB_Man_On_M15 )
      wire#w3
      I_Contact( "Unlock_Data".SB_Man_Off_M15 )
      wire#w4
      Coil( "Pusk_M15" )
   END_RUNG
   RUNG wire#w1
      Contact( "Unlock_Data".Vivesti_iz_auto_M15 )
   END_RUNG wire#w2
   RUNG wire#w2
      Contact( "Pusk_M15" )
   END_RUNG wire#w3
   RUNG wire#w1
      Contact( "Unlock_Data".Auto_Rezhim )
      Contact( "Unlock_Data".Auto_On_M15 )
      I_Contact( "Unlock_Data".Vivesti_iz_auto_M15 )
   END_RUNG wire#w4
   // the same network as SCL:
   "Pusk_M15" := "Unlock_Data".System_Ok AND NOT "Unlock_Data".Error_M15 AND ((("Unlock_Data".Manual_Rezhim OR "Unlock_Data".Vivesti_iz_auto_M15) AND ("Unlock_Data".SB_Man_On_M15 OR "Pusk_M15") AND NOT "Unlock_Data".SB_Man_Off_M15) OR ("Unlock_Data".Auto_Rezhim AND "Unlock_Data".Auto_On_M15 AND NOT "Unlock_Data".Vivesti_iz_auto_M15));
END_REGION

REGION Network 22
   RUNG wire#powerrail
      Contact( "Unlock_Data".System_Ok )
      I_Contact( "Unlock_Data".Error_M16 )
      wire#w1
      Contact( "Unlock_Data".Manual_Rezhim )
      wire#w2
      Contact( "Unlock_Data".SB_Man_On_M16 )
      wire#w3
      I_Contact( "Unlock_Data".SB_Man_Off_M16 )
      Coil( "Pusk_M16" )
   END_RUNG
   RUNG wire#w1
      Contact( "Unlock_Data".Auto_Rezhim )
   END_RUNG wire#w2
   RUNG wire#w2
      Contact( "Pusk_M16" )
   END_RUNG wire#w3
   // the same network as SCL:
   "Pusk_M16" := "Unlock_Data".System_Ok AND NOT "Unlock_Data".Error_M16 AND ("Unlock_Data".Manual_Rezhim OR "Unlock_Data".Auto_Rezhim) AND ("Unlock_Data".SB_Man_On_M16 OR "Pusk_M16") AND NOT "Unlock_Data".SB_Man_Off_M16;
END_REGION

REGION Network 23
   RUNG wire#powerrail
      Contact( "Unlock_Data".System_Ok )
      I_Contact( "Unlock_Data".Error_Vent )
      wire#w1
      Contact( "SB_vent_PUSK" )
      wire#w2
      Contact( "SB_Vent_Stop" )
      wire#w3
      Coil( "Pusk_Vent" )
   END_RUNG
   RUNG wire#w1
      Contact( "Pusk_Vent" )
   END_RUNG wire#w2
   RUNG wire#w3
      Coil( "Lamp_Ventilation" )
   END_RUNG
   // the same network as SCL:
   "Pusk_Vent" := "Unlock_Data".System_Ok AND NOT "Unlock_Data".Error_Vent AND ("SB_vent_PUSK" OR "Pusk_Vent") AND "SB_Vent_Stop";
   "Lamp_Ventilation" := "Pusk_Vent";
END_REGION

REGION Network 24
   RUNG wire#powerrail
      Contact( "Unlock_Data".System_Ok )
      Contact( "AlwaysTRUE" )
      wire#w1
      Contact( "Unlock_Data".Manual_Rezhim )
      wire#w2
      Contact( "Unlock_Data".SB_Man_On_Podogrev1 )
      wire#w3
      I_Contact( "Unlock_Data".SB_Man_Off_Podogrev1 )
      wire#w4
      Coil( "Podogrev1_On" )
   END_RUNG
   RUNG wire#w2
      Contact( "Podogrev1_On" )
   END_RUNG wire#w3
   RUNG wire#w1
      Contact( "Unlock_Data".Auto_Rezhim )
      Contact( "Unlock_Data".Auto_On_Podogrev1 )
   END_RUNG wire#w4
   // the same network as SCL:
   "Podogrev1_On" := "Unlock_Data".System_Ok AND "AlwaysTRUE" AND (("Unlock_Data".Manual_Rezhim AND ("Unlock_Data".SB_Man_On_Podogrev1 OR "Podogrev1_On") AND NOT "Unlock_Data".SB_Man_Off_Podogrev1) OR ("Unlock_Data".Auto_Rezhim AND "Unlock_Data".Auto_On_Podogrev1));
END_REGION

REGION Network 25
   RUNG wire#powerrail
      Contact( "Unlock_Data".System_Ok )
      I_Contact( "Unlock_Data".Error_Mkotel1 )
      wire#w1
      Contact( "Unlock_Data".Manual_Rezhim )
      wire#w2
      Contact( "Unlock_Data".SB_Man_On_Podogrev2 )
      wire#w3
      I_Contact( "Unlock_Data".SB_Man_Off_Podogrev2 )
      Coil( "Pusk_Kotel1" )
   END_RUNG
   RUNG wire#w1
      Contact( "Unlock_Data".Auto_Rezhim )
   END_RUNG wire#w2
   RUNG wire#w2
      Contact( "Pusk_Kotel1" )
   END_RUNG wire#w3
   // the same network as SCL:
   "Pusk_Kotel1" := "Unlock_Data".System_Ok AND NOT "Unlock_Data".Error_Mkotel1 AND ("Unlock_Data".Manual_Rezhim OR "Unlock_Data".Auto_Rezhim) AND ("Unlock_Data".SB_Man_On_Podogrev2 OR "Pusk_Kotel1") AND NOT "Unlock_Data".SB_Man_Off_Podogrev2;
END_REGION

REGION Network 26
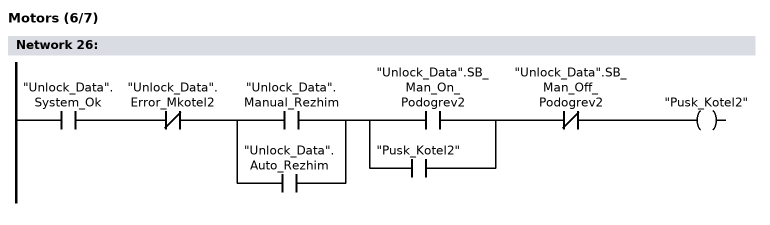
   RUNG wire#powerrail
      Contact( "Unlock_Data".System_Ok )
      I_Contact( "Unlock_Data".Error_Mkotel2 )
      wire#w1
      Contact( "Unlock_Data".Manual_Rezhim )
      wire#w2
      Contact( "Unlock_Data".SB_Man_On_Podogrev2 )
      wire#w3
      I_Contact( "Unlock_Data".SB_Man_Off_Podogrev2 )
      Coil( "Pusk_Kotel2" )
   END_RUNG
   RUNG wire#w1
      Contact( "Unlock_Data".Auto_Rezhim )
   END_RUNG wire#w2
   RUNG wire#w2
      Contact( "Pusk_Kotel2" )
   END_RUNG wire#w3
   // the same network as SCL:
   "Pusk_Kotel2" := "Unlock_Data".System_Ok AND NOT "Unlock_Data".Error_Mkotel2 AND ("Unlock_Data".Manual_Rezhim OR "Unlock_Data".Auto_Rezhim) AND ("Unlock_Data".SB_Man_On_Podogrev2 OR "Pusk_Kotel2") AND NOT "Unlock_Data".SB_Man_Off_Podogrev2;
END_REGION

REGION Network 27
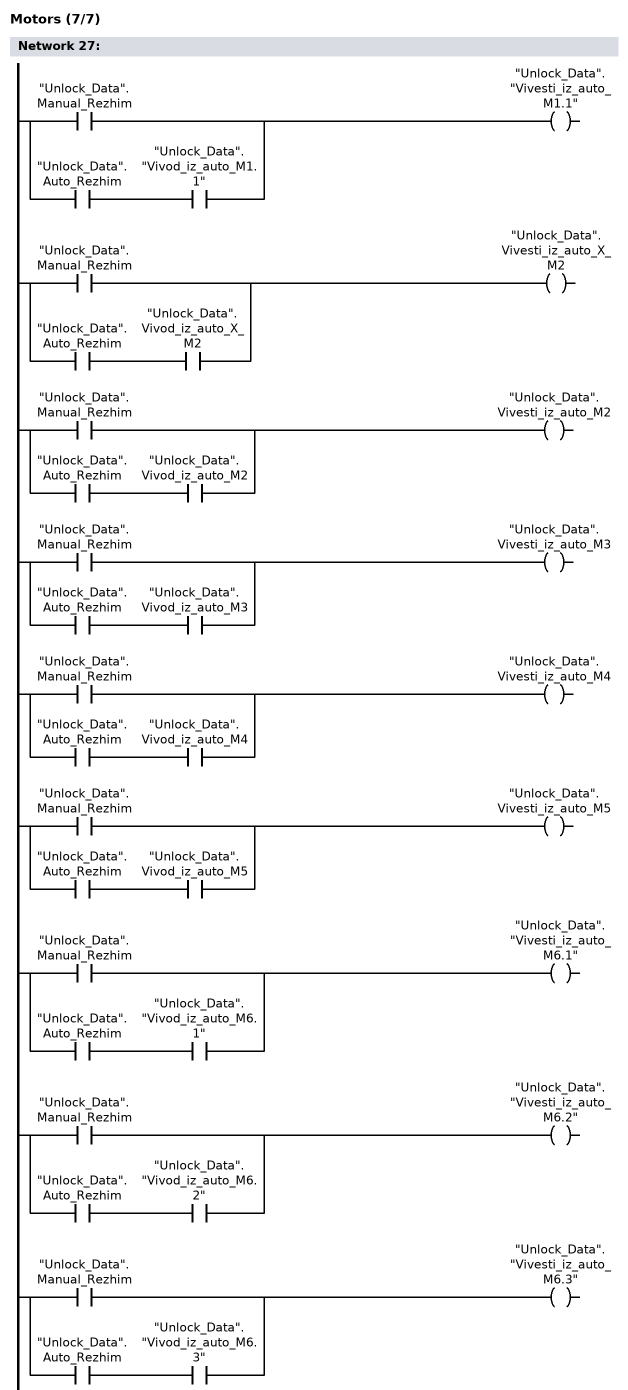
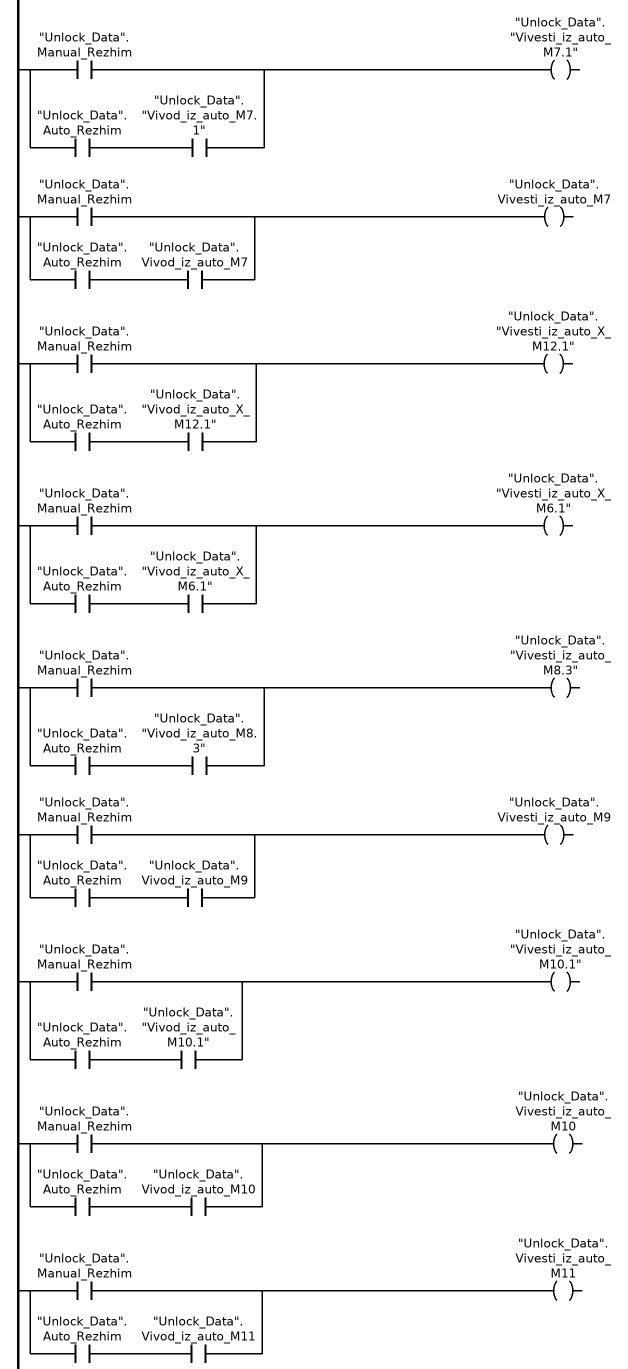
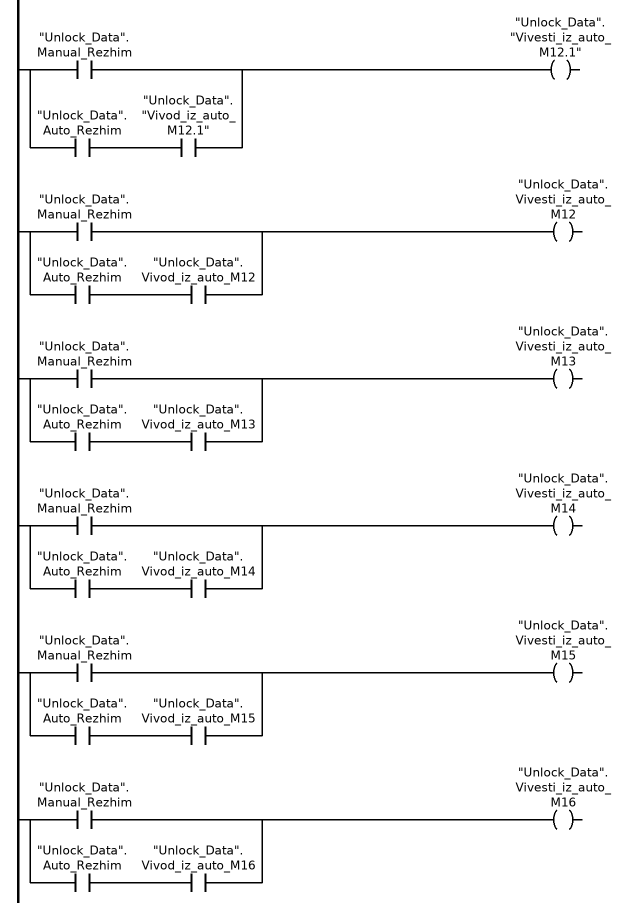
   RUNG wire#powerrail
      Contact( "Unlock_Data".Manual_Rezhim )
      wire#w1
      Coil( "Unlock_Data"."Vivesti_iz_auto_M1.1" )
   END_RUNG
   RUNG wire#powerrail
      Contact( "Unlock_Data".Auto_Rezhim )
      Contact( "Unlock_Data"."Vivod_iz_auto_M1.1" )
   END_RUNG wire#w1
   RUNG wire#powerrail
      Contact( "Unlock_Data".Manual_Rezhim )
      wire#w2
      Coil( "Unlock_Data".Vivesti_iz_auto_X_M2 )
   END_RUNG
   RUNG wire#powerrail
      Contact( "Unlock_Data".Auto_Rezhim )
      Contact( "Unlock_Data".Vivod_iz_auto_X_M2 )
   END_RUNG wire#w2
   RUNG wire#powerrail
      Contact( "Unlock_Data".Manual_Rezhim )
      wire#w3
      Coil( "Unlock_Data".Vivesti_iz_auto_M2 )
   END_RUNG
   RUNG wire#powerrail
      Contact( "Unlock_Data".Auto_Rezhim )
      Contact( "Unlock_Data".Vivod_iz_auto_M2 )
   END_RUNG wire#w3
   RUNG wire#powerrail
      Contact( "Unlock_Data".Manual_Rezhim )
      wire#w4
      Coil( "Unlock_Data".Vivesti_iz_auto_M3 )
   END_RUNG
   RUNG wire#powerrail
      Contact( "Unlock_Data".Auto_Rezhim )
      Contact( "Unlock_Data".Vivod_iz_auto_M3 )
   END_RUNG wire#w4
   RUNG wire#powerrail
      Contact( "Unlock_Data".Manual_Rezhim )
      wire#w5
      Coil( "Unlock_Data".Vivesti_iz_auto_M4 )
   END_RUNG
   RUNG wire#powerrail
      Contact( "Unlock_Data".Auto_Rezhim )
      Contact( "Unlock_Data".Vivod_iz_auto_M4 )
   END_RUNG wire#w5
   RUNG wire#powerrail
      Contact( "Unlock_Data".Manual_Rezhim )
      wire#w6
      Coil( "Unlock_Data".Vivesti_iz_auto_M5 )
   END_RUNG
   RUNG wire#powerrail
      Contact( "Unlock_Data".Auto_Rezhim )
      Contact( "Unlock_Data".Vivod_iz_auto_M5 )
   END_RUNG wire#w6
   RUNG wire#powerrail
      Contact( "Unlock_Data".Manual_Rezhim )
      wire#w7
      Coil( "Unlock_Data"."Vivesti_iz_auto_M6.1" )
   END_RUNG
   RUNG wire#powerrail
      Contact( "Unlock_Data".Auto_Rezhim )
      Contact( "Unlock_Data"."Vivod_iz_auto_M6.1" )
   END_RUNG wire#w7
   RUNG wire#powerrail
      Contact( "Unlock_Data".Manual_Rezhim )
      wire#w8
      Coil( "Unlock_Data"."Vivesti_iz_auto_M6.2" )
   END_RUNG
   RUNG wire#powerrail
      Contact( "Unlock_Data".Auto_Rezhim )
      Contact( "Unlock_Data"."Vivod_iz_auto_M6.2" )
   END_RUNG wire#w8
   RUNG wire#powerrail
      Contact( "Unlock_Data".Manual_Rezhim )
      wire#w9
      Coil( "Unlock_Data"."Vivesti_iz_auto_M6.3" )
   END_RUNG
   RUNG wire#powerrail
      Contact( "Unlock_Data".Auto_Rezhim )
      Contact( "Unlock_Data"."Vivod_iz_auto_M6.3" )
   END_RUNG wire#w9
   RUNG wire#powerrail
      Contact( "Unlock_Data".Manual_Rezhim )
      wire#w10
      Coil( "Unlock_Data"."Vivesti_iz_auto_M7.1" )
   END_RUNG
   RUNG wire#powerrail
      Contact( "Unlock_Data".Auto_Rezhim )
      Contact( "Unlock_Data"."Vivod_iz_auto_M7.1" )
   END_RUNG wire#w10
   RUNG wire#powerrail
      Contact( "Unlock_Data".Manual_Rezhim )
      wire#w11
      Coil( "Unlock_Data".Vivesti_iz_auto_M7 )
   END_RUNG
   RUNG wire#powerrail
      Contact( "Unlock_Data".Auto_Rezhim )
      Contact( "Unlock_Data".Vivod_iz_auto_M7 )
   END_RUNG wire#w11
   RUNG wire#powerrail
      Contact( "Unlock_Data".Manual_Rezhim )
      wire#w12
      Coil( "Unlock_Data"."Vivesti_iz_auto_X_M12.1" )
   END_RUNG
   RUNG wire#powerrail
      Contact( "Unlock_Data".Auto_Rezhim )
      Contact( "Unlock_Data"."Vivod_iz_auto_X_M12.1" )
   END_RUNG wire#w12
   RUNG wire#powerrail
      Contact( "Unlock_Data".Manual_Rezhim )
      wire#w13
      Coil( "Unlock_Data"."Vivesti_iz_auto_X_M6.1" )
   END_RUNG
   RUNG wire#powerrail
      Contact( "Unlock_Data".Auto_Rezhim )
      Contact( "Unlock_Data"."Vivod_iz_auto_X_M6.1" )
   END_RUNG wire#w13
   RUNG wire#powerrail
      Contact( "Unlock_Data".Manual_Rezhim )
      wire#w14
      Coil( "Unlock_Data"."Vivesti_iz_auto_M8.3" )
   END_RUNG
   RUNG wire#powerrail
      Contact( "Unlock_Data".Auto_Rezhim )
      Contact( "Unlock_Data"."Vivod_iz_auto_M8.3" )
   END_RUNG wire#w14
   RUNG wire#powerrail
      Contact( "Unlock_Data".Manual_Rezhim )
      wire#w15
      Coil( "Unlock_Data".Vivesti_iz_auto_M9 )
   END_RUNG
   RUNG wire#powerrail
      Contact( "Unlock_Data".Auto_Rezhim )
      Contact( "Unlock_Data".Vivod_iz_auto_M9 )
   END_RUNG wire#w15
   RUNG wire#powerrail
      Contact( "Unlock_Data".Manual_Rezhim )
      wire#w16
      Coil( "Unlock_Data"."Vivesti_iz_auto_M10.1" )
   END_RUNG
   RUNG wire#powerrail
      Contact( "Unlock_Data".Auto_Rezhim )
      Contact( "Unlock_Data"."Vivod_iz_auto_M10.1" )
   END_RUNG wire#w16
   RUNG wire#powerrail
      Contact( "Unlock_Data".Manual_Rezhim )
      wire#w17
      Coil( "Unlock_Data".Vivesti_iz_auto_M10 )
   END_RUNG
   RUNG wire#powerrail
      Contact( "Unlock_Data".Auto_Rezhim )
      Contact( "Unlock_Data".Vivod_iz_auto_M10 )
   END_RUNG wire#w17
   RUNG wire#powerrail
      Contact( "Unlock_Data".Manual_Rezhim )
      wire#w18
      Coil( "Unlock_Data".Vivesti_iz_auto_M11 )
   END_RUNG
   RUNG wire#powerrail
      Contact( "Unlock_Data".Auto_Rezhim )
      Contact( "Unlock_Data".Vivod_iz_auto_M11 )
   END_RUNG wire#w18
   RUNG wire#powerrail
      Contact( "Unlock_Data".Manual_Rezhim )
      wire#w19
      Coil( "Unlock_Data"."Vivesti_iz_auto_M12.1" )
   END_RUNG
   RUNG wire#powerrail
      Contact( "Unlock_Data".Auto_Rezhim )
      Contact( "Unlock_Data"."Vivod_iz_auto_M12.1" )
   END_RUNG wire#w19
   RUNG wire#powerrail
      Contact( "Unlock_Data".Manual_Rezhim )
      wire#w20
      Coil( "Unlock_Data".Vivesti_iz_auto_M12 )
   END_RUNG
   RUNG wire#powerrail
      Contact( "Unlock_Data".Auto_Rezhim )
      Contact( "Unlock_Data".Vivod_iz_auto_M12 )
   END_RUNG wire#w20
   RUNG wire#powerrail
      Contact( "Unlock_Data".Manual_Rezhim )
      wire#w21
      Coil( "Unlock_Data".Vivesti_iz_auto_M13 )
   END_RUNG
   RUNG wire#powerrail
      Contact( "Unlock_Data".Auto_Rezhim )
      Contact( "Unlock_Data".Vivod_iz_auto_M13 )
   END_RUNG wire#w21
   RUNG wire#powerrail
      Contact( "Unlock_Data".Manual_Rezhim )
      wire#w22
      Coil( "Unlock_Data".Vivesti_iz_auto_M14 )
   END_RUNG
   RUNG wire#powerrail
      Contact( "Unlock_Data".Auto_Rezhim )
      Contact( "Unlock_Data".Vivod_iz_auto_M14 )
   END_RUNG wire#w22
   RUNG wire#powerrail
      Contact( "Unlock_Data".Manual_Rezhim )
      wire#w23
      Coil( "Unlock_Data".Vivesti_iz_auto_M15 )
   END_RUNG
   RUNG wire#powerrail
      Contact( "Unlock_Data".Auto_Rezhim )
      Contact( "Unlock_Data".Vivod_iz_auto_M15 )
   END_RUNG wire#w23
   RUNG wire#powerrail
      Contact( "Unlock_Data".Manual_Rezhim )
      wire#w24
      Coil( "Unlock_Data".Vivesti_iz_auto_M16 )
   END_RUNG
   RUNG wire#powerrail
      Contact( "Unlock_Data".Auto_Rezhim )
      Contact( "Unlock_Data".Vivod_iz_auto_M16 )
   END_RUNG wire#w24
   // the same network as SCL:
   "Unlock_Data"."Vivesti_iz_auto_M1.1" := "Unlock_Data".Manual_Rezhim OR ("Unlock_Data".Auto_Rezhim AND "Unlock_Data"."Vivod_iz_auto_M1.1");
   "Unlock_Data".Vivesti_iz_auto_X_M2 := "Unlock_Data".Manual_Rezhim OR ("Unlock_Data".Auto_Rezhim AND "Unlock_Data".Vivod_iz_auto_X_M2);
   "Unlock_Data".Vivesti_iz_auto_M2 := "Unlock_Data".Manual_Rezhim OR ("Unlock_Data".Auto_Rezhim AND "Unlock_Data".Vivod_iz_auto_M2);
   "Unlock_Data".Vivesti_iz_auto_M3 := "Unlock_Data".Manual_Rezhim OR ("Unlock_Data".Auto_Rezhim AND "Unlock_Data".Vivod_iz_auto_M3);
   "Unlock_Data".Vivesti_iz_auto_M4 := "Unlock_Data".Manual_Rezhim OR ("Unlock_Data".Auto_Rezhim AND "Unlock_Data".Vivod_iz_auto_M4);
   "Unlock_Data".Vivesti_iz_auto_M5 := "Unlock_Data".Manual_Rezhim OR ("Unlock_Data".Auto_Rezhim AND "Unlock_Data".Vivod_iz_auto_M5);
   "Unlock_Data"."Vivesti_iz_auto_M6.1" := "Unlock_Data".Manual_Rezhim OR ("Unlock_Data".Auto_Rezhim AND "Unlock_Data"."Vivod_iz_auto_M6.1");
   "Unlock_Data"."Vivesti_iz_auto_M6.2" := "Unlock_Data".Manual_Rezhim OR ("Unlock_Data".Auto_Rezhim AND "Unlock_Data"."Vivod_iz_auto_M6.2");
   "Unlock_Data"."Vivesti_iz_auto_M6.3" := "Unlock_Data".Manual_Rezhim OR ("Unlock_Data".Auto_Rezhim AND "Unlock_Data"."Vivod_iz_auto_M6.3");
   "Unlock_Data"."Vivesti_iz_auto_M7.1" := "Unlock_Data".Manual_Rezhim OR ("Unlock_Data".Auto_Rezhim AND "Unlock_Data"."Vivod_iz_auto_M7.1");
   "Unlock_Data".Vivesti_iz_auto_M7 := "Unlock_Data".Manual_Rezhim OR ("Unlock_Data".Auto_Rezhim AND "Unlock_Data".Vivod_iz_auto_M7);
   "Unlock_Data"."Vivesti_iz_auto_X_M12.1" := "Unlock_Data".Manual_Rezhim OR ("Unlock_Data".Auto_Rezhim AND "Unlock_Data"."Vivod_iz_auto_X_M12.1");
   "Unlock_Data"."Vivesti_iz_auto_X_M6.1" := "Unlock_Data".Manual_Rezhim OR ("Unlock_Data".Auto_Rezhim AND "Unlock_Data"."Vivod_iz_auto_X_M6.1");
   "Unlock_Data"."Vivesti_iz_auto_M8.3" := "Unlock_Data".Manual_Rezhim OR ("Unlock_Data".Auto_Rezhim AND "Unlock_Data"."Vivod_iz_auto_M8.3");
   "Unlock_Data".Vivesti_iz_auto_M9 := "Unlock_Data".Manual_Rezhim OR ("Unlock_Data".Auto_Rezhim AND "Unlock_Data".Vivod_iz_auto_M9);
   "Unlock_Data"."Vivesti_iz_auto_M10.1" := "Unlock_Data".Manual_Rezhim OR ("Unlock_Data".Auto_Rezhim AND "Unlock_Data"."Vivod_iz_auto_M10.1");
   "Unlock_Data".Vivesti_iz_auto_M10 := "Unlock_Data".Manual_Rezhim OR ("Unlock_Data".Auto_Rezhim AND "Unlock_Data".Vivod_iz_auto_M10);
   "Unlock_Data".Vivesti_iz_auto_M11 := "Unlock_Data".Manual_Rezhim OR ("Unlock_Data".Auto_Rezhim AND "Unlock_Data".Vivod_iz_auto_M11);
   "Unlock_Data"."Vivesti_iz_auto_M12.1" := "Unlock_Data".Manual_Rezhim OR ("Unlock_Data".Auto_Rezhim AND "Unlock_Data"."Vivod_iz_auto_M12.1");
   "Unlock_Data".Vivesti_iz_auto_M12 := "Unlock_Data".Manual_Rezhim OR ("Unlock_Data".Auto_Rezhim AND "Unlock_Data".Vivod_iz_auto_M12);
   "Unlock_Data".Vivesti_iz_auto_M13 := "Unlock_Data".Manual_Rezhim OR ("Unlock_Data".Auto_Rezhim AND "Unlock_Data".Vivod_iz_auto_M13);
   "Unlock_Data".Vivesti_iz_auto_M14 := "Unlock_Data".Manual_Rezhim OR ("Unlock_Data".Auto_Rezhim AND "Unlock_Data".Vivod_iz_auto_M14);
   "Unlock_Data".Vivesti_iz_auto_M15 := "Unlock_Data".Manual_Rezhim OR ("Unlock_Data".Auto_Rezhim AND "Unlock_Data".Vivod_iz_auto_M15);
   "Unlock_Data".Vivesti_iz_auto_M16 := "Unlock_Data".Manual_Rezhim OR ("Unlock_Data".Auto_Rezhim AND "Unlock_Data".Vivod_iz_auto_M16);
END_REGION
END_FUNCTION_BLOCK

FUNCTION_BLOCK "Main_Cycle"   // FB3, LAD
{ S7_Optimized_Access := 'TRUE' }
VERSION : 0.1
   VAR_TEMP   // added for the SCL form of the ladder/FBD networks
      _w1 : Bool;
      _w2 : Bool;
      _w3 : Bool;
      _w4 : Bool;
      _w5 : Bool;
      _w6 : Bool;
      _w7 : Bool;
      _w8 : Bool;
      _w9 : Bool;
      _w10 : Bool;
      _w11 : Bool;
      _w12 : Bool;
   END_VAR
BEGIN

REGION Network 1
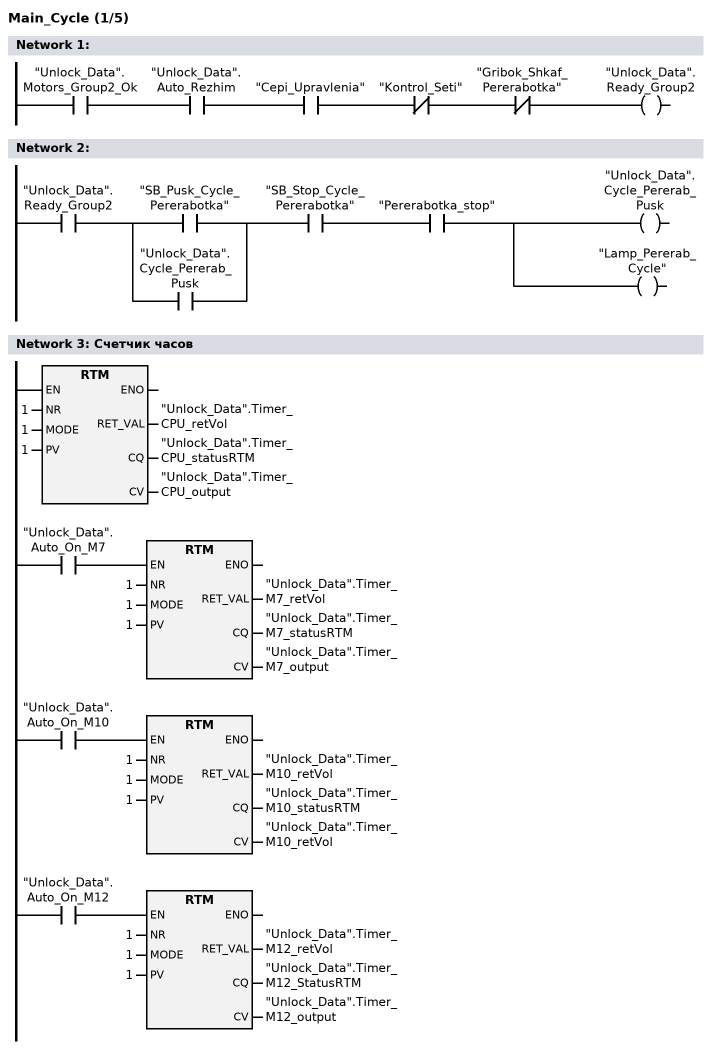
   RUNG wire#powerrail
      Contact( "Unlock_Data".Motors_Group2_Ok )
      Contact( "Unlock_Data".Auto_Rezhim )
      Contact( "Cepi_Upravlenia" )
      I_Contact( "Kontrol_Seti" )
      I_Contact( "Gribok_Shkaf_Pererabotka" )
      Coil( "Unlock_Data".Ready_Group2 )
   END_RUNG
   // the same network as SCL:
   "Unlock_Data".Ready_Group2 := "Unlock_Data".Motors_Group2_Ok AND "Unlock_Data".Auto_Rezhim AND "Cepi_Upravlenia" AND NOT "Kontrol_Seti" AND NOT "Gribok_Shkaf_Pererabotka";
END_REGION

REGION Network 2
   RUNG wire#powerrail
      Contact( "Unlock_Data".Ready_Group2 )
      wire#w1
      Contact( "SB_Pusk_Cycle_Pererabotka" )
      wire#w2
      Contact( "SB_Stop_Cycle_Pererabotka" )
      Contact( "Pererabotka_stop" )
      wire#w3
      Coil( "Unlock_Data".Cycle_Pererab_Pusk )
   END_RUNG
   RUNG wire#w1
      Contact( "Unlock_Data".Cycle_Pererab_Pusk )
   END_RUNG wire#w2
   RUNG wire#w3
      Coil( "Lamp_Pererab_Cycle" )
   END_RUNG
   // the same network as SCL:
   "Unlock_Data".Cycle_Pererab_Pusk := "Unlock_Data".Ready_Group2 AND ("SB_Pusk_Cycle_Pererabotka" OR "Unlock_Data".Cycle_Pererab_Pusk) AND "SB_Stop_Cycle_Pererabotka" AND "Pererabotka_stop";
   "Lamp_Pererab_Cycle" := "Unlock_Data".Cycle_Pererab_Pusk;
END_REGION

REGION Network 3: Счетчик часов
   // no checked SCL form for this network; see the picture
END_REGION

REGION Network 4: Переработка ПУСК
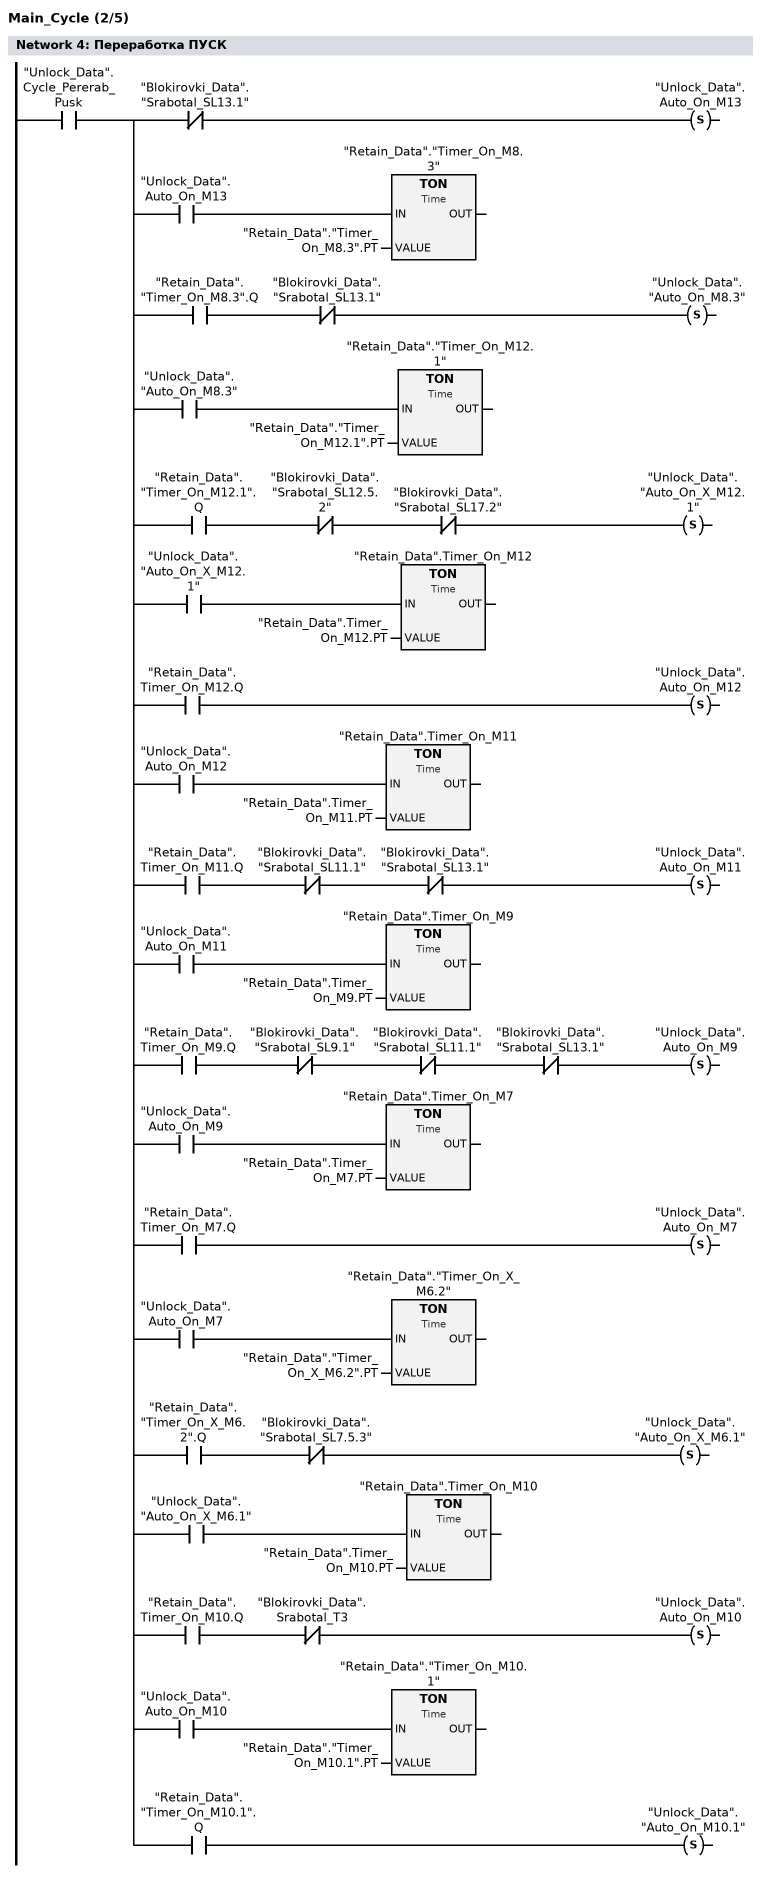
   IF "Unlock_Data".Cycle_Pererab_Pusk AND NOT "Blokirovki_Data"."Srabotal_SL13.1" THEN
       "Unlock_Data".Auto_On_M13 := TRUE;
   END_IF;
   "Retain_Data"."Timer_On_M8.3".TON(IN := "Unlock_Data".Cycle_Pererab_Pusk AND "Unlock_Data".Auto_On_M13, PT := "Retain_Data"."Timer_On_M8.3".PT);   // TON coil
   IF "Unlock_Data".Cycle_Pererab_Pusk AND "Retain_Data"."Timer_On_M8.3".Q AND NOT "Blokirovki_Data"."Srabotal_SL13.1" THEN
       "Unlock_Data"."Auto_On_M8.3" := TRUE;
   END_IF;
   "Retain_Data"."Timer_On_M12.1".TON(IN := "Unlock_Data".Cycle_Pererab_Pusk AND "Unlock_Data"."Auto_On_M8.3", PT := "Retain_Data"."Timer_On_M12.1".PT);   // TON coil
   IF "Unlock_Data".Cycle_Pererab_Pusk AND "Retain_Data"."Timer_On_M12.1".Q AND NOT "Blokirovki_Data"."Srabotal_SL12.5.2" AND NOT "Blokirovki_Data"."Srabotal_SL17.2" THEN
       "Unlock_Data"."Auto_On_X_M12.1" := TRUE;
   END_IF;
   "Retain_Data".Timer_On_M12.TON(IN := "Unlock_Data".Cycle_Pererab_Pusk AND "Unlock_Data"."Auto_On_X_M12.1", PT := "Retain_Data".Timer_On_M12.PT);   // TON coil
   IF "Unlock_Data".Cycle_Pererab_Pusk AND "Retain_Data".Timer_On_M12.Q THEN
       "Unlock_Data".Auto_On_M12 := TRUE;
   END_IF;
   "Retain_Data".Timer_On_M11.TON(IN := "Unlock_Data".Cycle_Pererab_Pusk AND "Unlock_Data".Auto_On_M12, PT := "Retain_Data".Timer_On_M11.PT);   // TON coil
   IF "Unlock_Data".Cycle_Pererab_Pusk AND "Retain_Data".Timer_On_M11.Q AND NOT "Blokirovki_Data"."Srabotal_SL11.1" AND NOT "Blokirovki_Data"."Srabotal_SL13.1" THEN
       "Unlock_Data".Auto_On_M11 := TRUE;
   END_IF;
   "Retain_Data".Timer_On_M9.TON(IN := "Unlock_Data".Cycle_Pererab_Pusk AND "Unlock_Data".Auto_On_M11, PT := "Retain_Data".Timer_On_M9.PT);   // TON coil
   IF "Unlock_Data".Cycle_Pererab_Pusk AND "Retain_Data".Timer_On_M9.Q AND NOT "Blokirovki_Data"."Srabotal_SL9.1" AND NOT "Blokirovki_Data"."Srabotal_SL11.1" AND NOT "Blokirovki_Data"."Srabotal_SL13.1" THEN
       "Unlock_Data".Auto_On_M9 := TRUE;
   END_IF;
   "Retain_Data".Timer_On_M7.TON(IN := "Unlock_Data".Cycle_Pererab_Pusk AND "Unlock_Data".Auto_On_M9, PT := "Retain_Data".Timer_On_M7.PT);   // TON coil
   IF "Unlock_Data".Cycle_Pererab_Pusk AND "Retain_Data".Timer_On_M7.Q THEN
       "Unlock_Data".Auto_On_M7 := TRUE;
   END_IF;
   "Retain_Data"."Timer_On_X_M6.2".TON(IN := "Unlock_Data".Cycle_Pererab_Pusk AND "Unlock_Data".Auto_On_M7, PT := "Retain_Data"."Timer_On_X_M6.2".PT);   // TON coil
   IF "Unlock_Data".Cycle_Pererab_Pusk AND "Retain_Data"."Timer_On_X_M6.2".Q AND NOT "Blokirovki_Data"."Srabotal_SL7.5.3" THEN
       "Unlock_Data"."Auto_On_X_M6.1" := TRUE;
   END_IF;
   "Retain_Data".Timer_On_M10.TON(IN := "Unlock_Data".Cycle_Pererab_Pusk AND "Unlock_Data"."Auto_On_X_M6.1", PT := "Retain_Data".Timer_On_M10.PT);   // TON coil
   IF "Unlock_Data".Cycle_Pererab_Pusk AND "Retain_Data".Timer_On_M10.Q AND NOT "Blokirovki_Data".Srabotal_T3 THEN
       "Unlock_Data".Auto_On_M10 := TRUE;
   END_IF;
   "Retain_Data"."Timer_On_M10.1".TON(IN := "Unlock_Data".Cycle_Pererab_Pusk AND "Unlock_Data".Auto_On_M10, PT := "Retain_Data"."Timer_On_M10.1".PT);   // TON coil
   IF "Unlock_Data".Cycle_Pererab_Pusk AND "Retain_Data"."Timer_On_M10.1".Q THEN
       "Unlock_Data"."Auto_On_M10.1" := TRUE;
   END_IF;
END_REGION

REGION Network 5
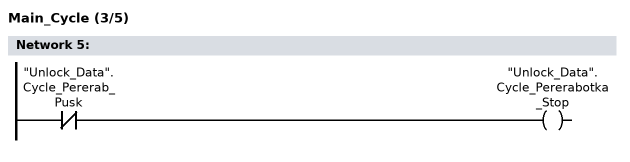
   RUNG wire#powerrail
      I_Contact( "Unlock_Data".Cycle_Pererab_Pusk )
      Coil( "Unlock_Data".Cycle_Pererabotka_Stop )
   END_RUNG
   // the same network as SCL:
   "Unlock_Data".Cycle_Pererabotka_Stop := NOT "Unlock_Data".Cycle_Pererab_Pusk;
END_REGION

REGION Network 6
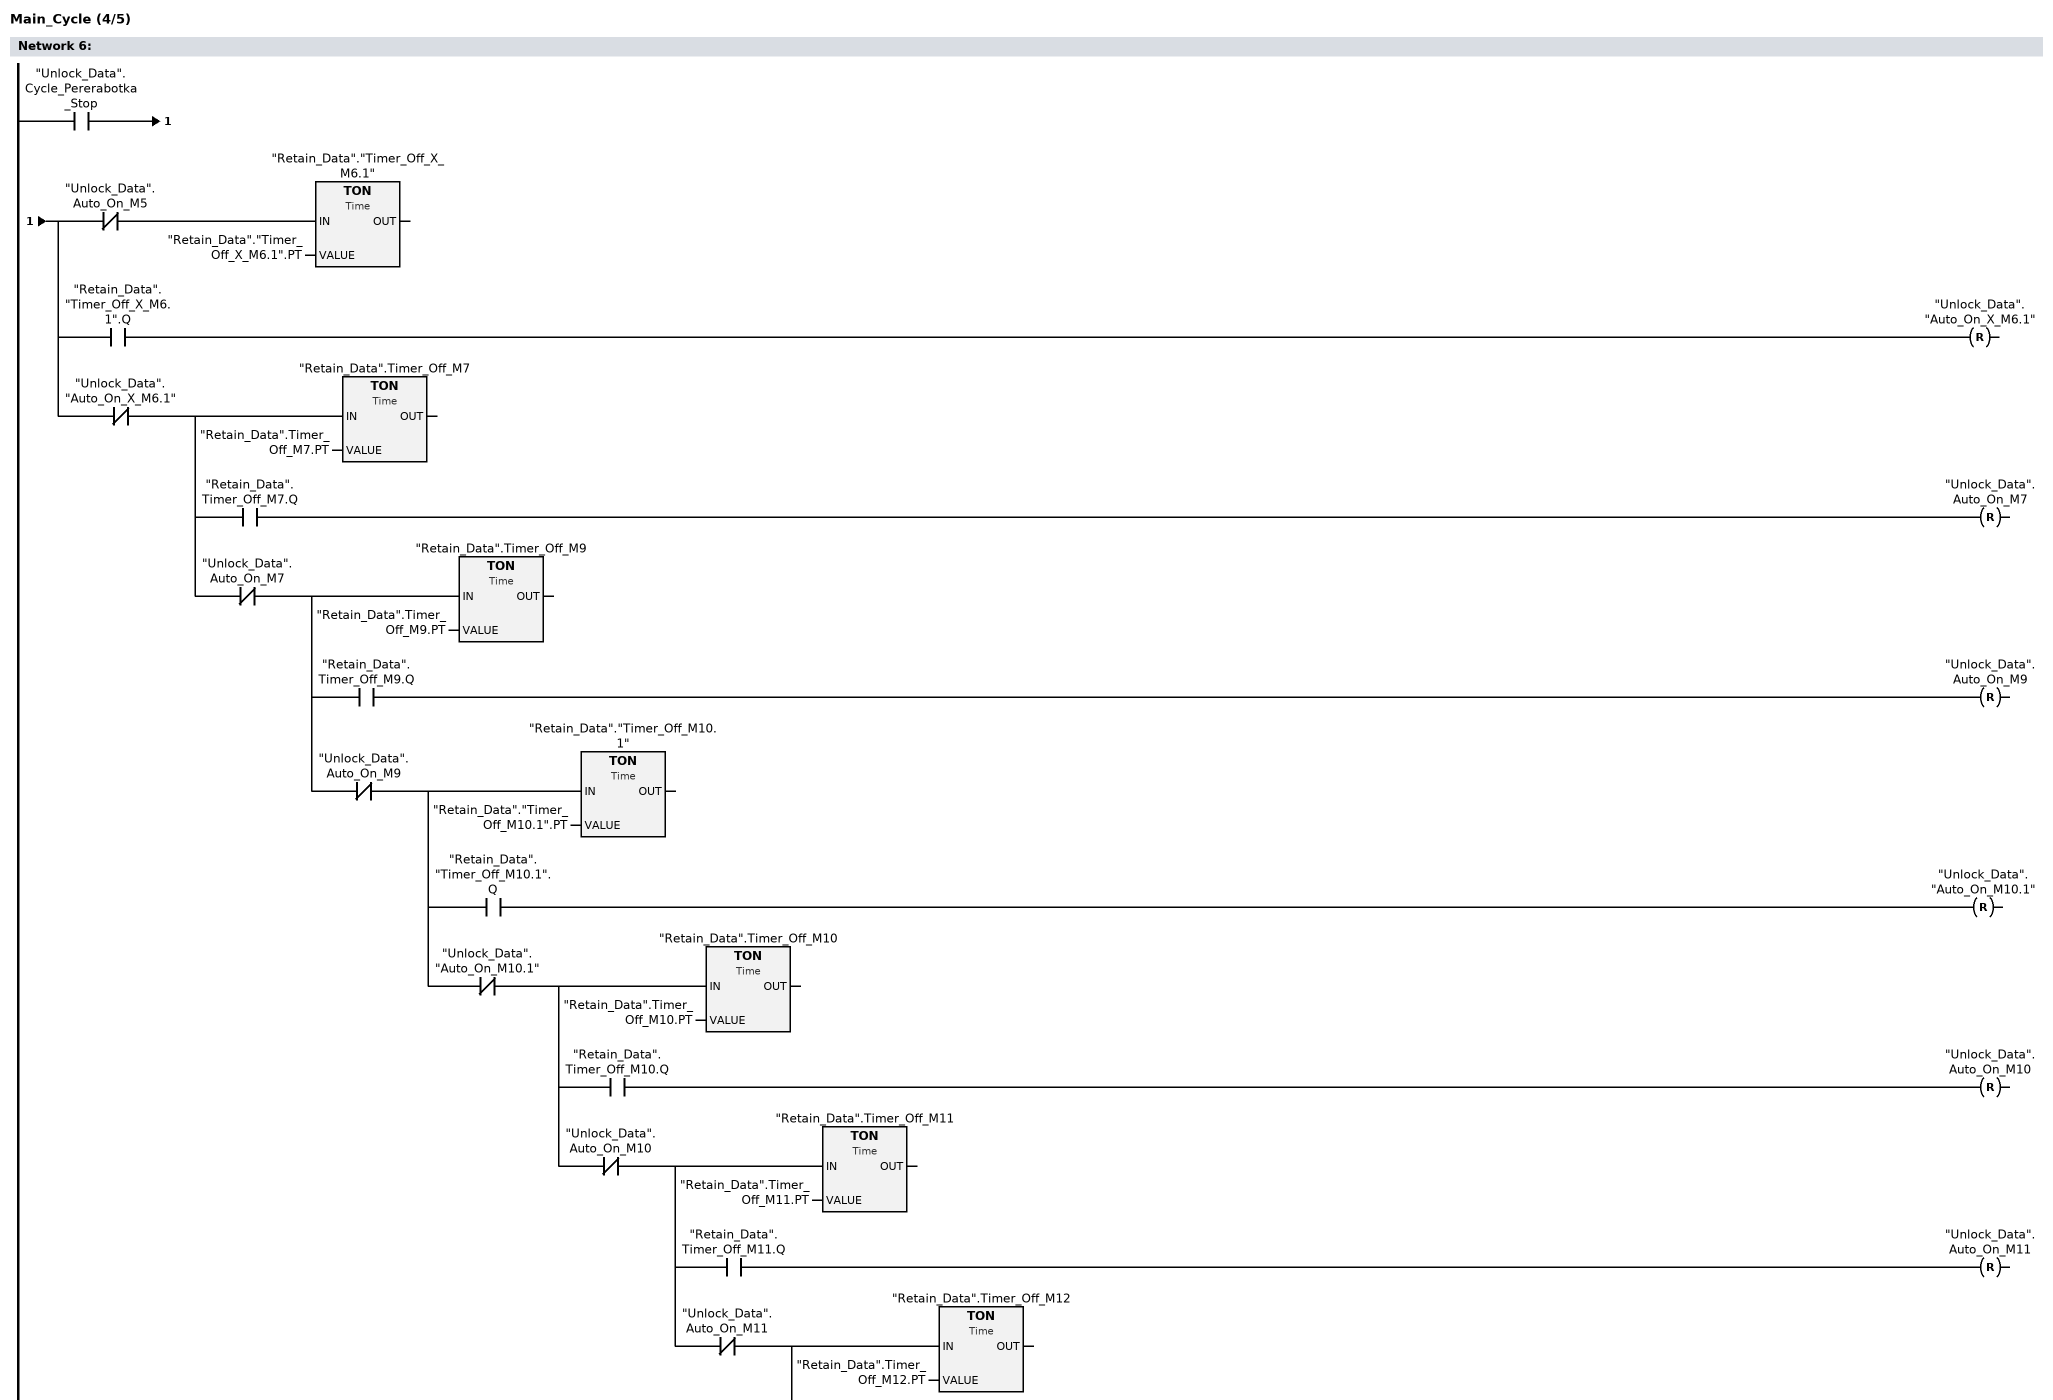
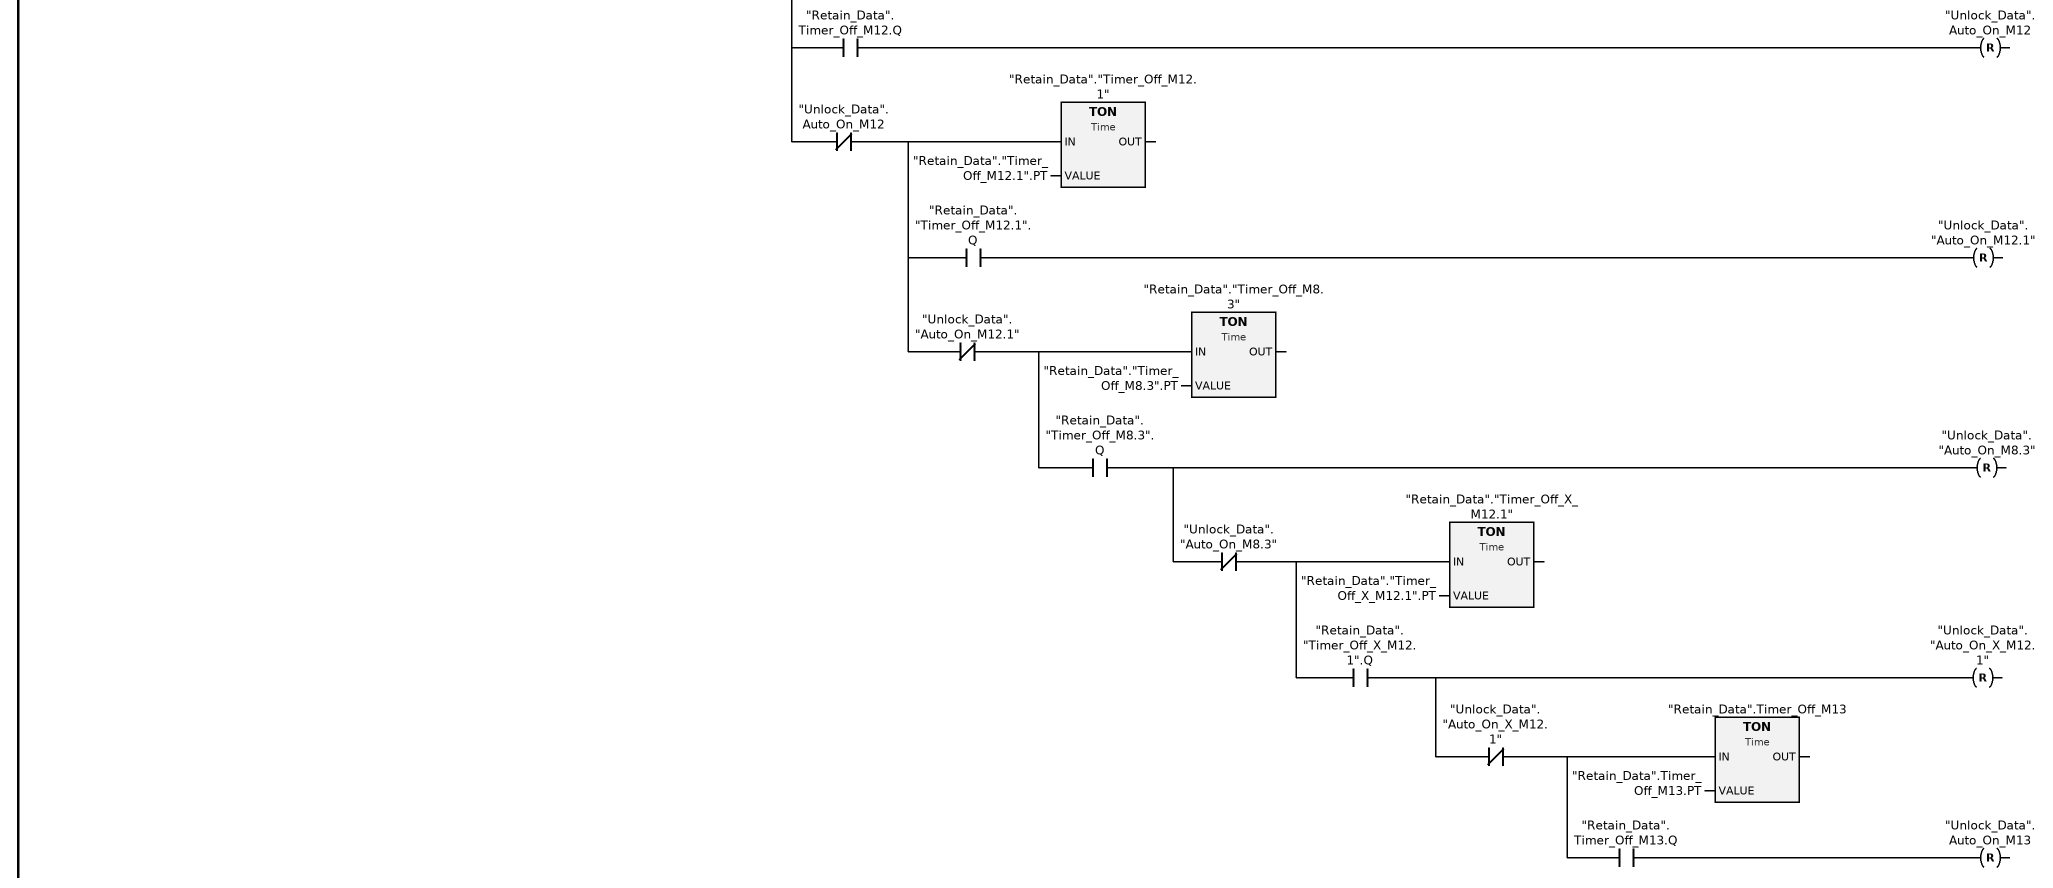
   "Retain_Data"."Timer_Off_X_M6.1".TON(IN := "Unlock_Data".Cycle_Pererabotka_Stop AND NOT "Unlock_Data".Auto_On_M5, PT := "Retain_Data"."Timer_Off_X_M6.1".PT);   // TON coil
   IF "Unlock_Data".Cycle_Pererabotka_Stop AND "Retain_Data"."Timer_Off_X_M6.1".Q THEN
       "Unlock_Data"."Auto_On_X_M6.1" := FALSE;
   END_IF;
   #_w1 := "Unlock_Data".Cycle_Pererabotka_Stop AND NOT "Unlock_Data"."Auto_On_X_M6.1";
   "Retain_Data".Timer_Off_M7.TON(IN := #_w1, PT := "Retain_Data".Timer_Off_M7.PT);   // TON coil
   IF #_w1 AND "Retain_Data".Timer_Off_M7.Q THEN "Unlock_Data".Auto_On_M7 := FALSE; END_IF;
   #_w2 := #_w1 AND NOT "Unlock_Data".Auto_On_M7;
   "Retain_Data".Timer_Off_M9.TON(IN := #_w2, PT := "Retain_Data".Timer_Off_M9.PT);   // TON coil
   IF #_w2 AND "Retain_Data".Timer_Off_M9.Q THEN "Unlock_Data".Auto_On_M9 := FALSE; END_IF;
   #_w3 := #_w2 AND NOT "Unlock_Data".Auto_On_M9;
   "Retain_Data"."Timer_Off_M10.1".TON(IN := #_w3, PT := "Retain_Data"."Timer_Off_M10.1".PT);   // TON coil
   IF #_w3 AND "Retain_Data"."Timer_Off_M10.1".Q THEN "Unlock_Data"."Auto_On_M10.1" := FALSE; END_IF;
   #_w4 := #_w3 AND NOT "Unlock_Data"."Auto_On_M10.1";
   "Retain_Data".Timer_Off_M10.TON(IN := #_w4, PT := "Retain_Data".Timer_Off_M10.PT);   // TON coil
   IF #_w4 AND "Retain_Data".Timer_Off_M10.Q THEN "Unlock_Data".Auto_On_M10 := FALSE; END_IF;
   #_w5 := #_w4 AND NOT "Unlock_Data".Auto_On_M10;
   "Retain_Data".Timer_Off_M11.TON(IN := #_w5, PT := "Retain_Data".Timer_Off_M11.PT);   // TON coil
   IF #_w5 AND "Retain_Data".Timer_Off_M11.Q THEN "Unlock_Data".Auto_On_M11 := FALSE; END_IF;
   #_w6 := #_w5 AND NOT "Unlock_Data".Auto_On_M11;
   "Retain_Data".Timer_Off_M12.TON(IN := #_w6, PT := "Retain_Data".Timer_Off_M12.PT);   // TON coil
   IF #_w6 AND "Retain_Data".Timer_Off_M12.Q THEN "Unlock_Data".Auto_On_M12 := FALSE; END_IF;
   #_w7 := #_w6 AND NOT "Unlock_Data".Auto_On_M12;
   "Retain_Data"."Timer_Off_M12.1".TON(IN := #_w7, PT := "Retain_Data"."Timer_Off_M12.1".PT);   // TON coil
   IF #_w7 AND "Retain_Data"."Timer_Off_M12.1".Q THEN "Unlock_Data"."Auto_On_M12.1" := FALSE; END_IF;
   #_w8 := #_w7 AND NOT "Unlock_Data"."Auto_On_M12.1";
   "Retain_Data"."Timer_Off_M8.3".TON(IN := #_w8, PT := "Retain_Data"."Timer_Off_M8.3".PT);   // TON coil
   #_w9 := #_w8 AND "Retain_Data"."Timer_Off_M8.3".Q;
   IF #_w9 THEN "Unlock_Data"."Auto_On_M8.3" := FALSE; END_IF;
   #_w10 := #_w9 AND NOT "Unlock_Data"."Auto_On_M8.3";
   "Retain_Data"."Timer_Off_X_M12.1".TON(IN := #_w10, PT := "Retain_Data"."Timer_Off_X_M12.1".PT);   // TON coil
   #_w11 := #_w10 AND "Retain_Data"."Timer_Off_X_M12.1".Q;
   IF #_w11 THEN "Unlock_Data"."Auto_On_X_M12.1" := FALSE; END_IF;
   #_w12 := #_w11 AND NOT "Unlock_Data"."Auto_On_X_M12.1";
   "Retain_Data".Timer_Off_M13.TON(IN := #_w12, PT := "Retain_Data".Timer_Off_M13.PT);   // TON coil
   IF #_w12 AND "Retain_Data".Timer_Off_M13.Q THEN "Unlock_Data".Auto_On_M13 := FALSE; END_IF;
END_REGION

REGION Network 8
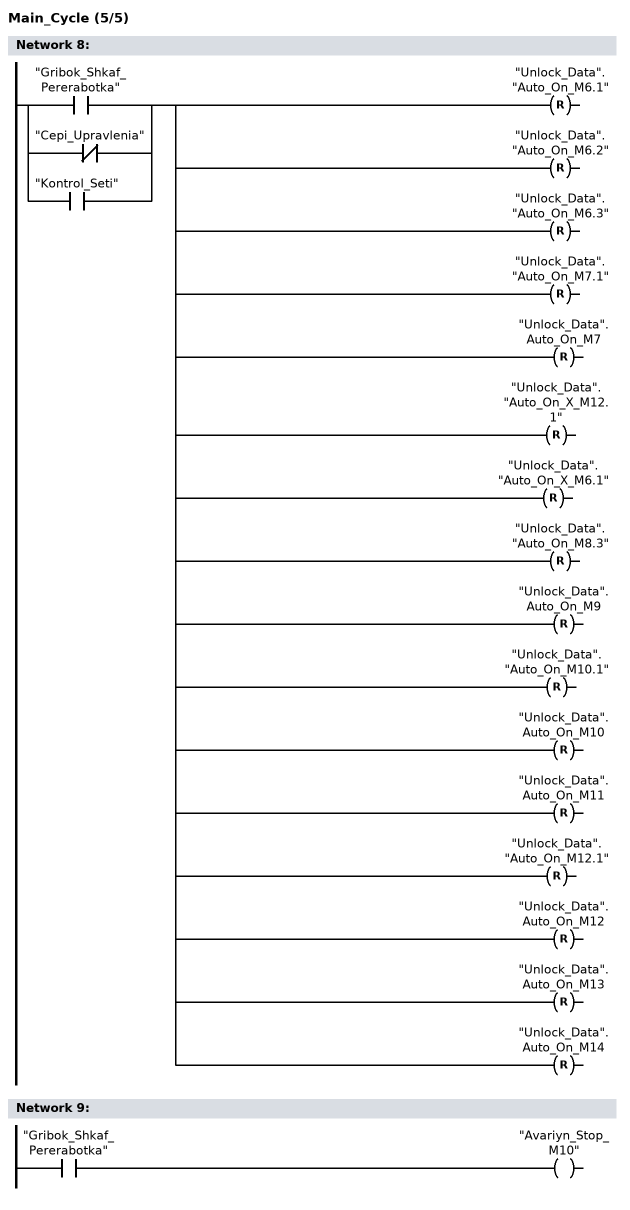
   RUNG wire#powerrail
      Contact( "Gribok_Shkaf_Pererabotka" )
      wire#w1
      R_Coil( "Unlock_Data"."Auto_On_M6.1" )
   END_RUNG
   RUNG wire#powerrail
      I_Contact( "Cepi_Upravlenia" )
   END_RUNG wire#w1
   RUNG wire#powerrail
      Contact( "Kontrol_Seti" )
   END_RUNG wire#w1
   RUNG wire#w1
      R_Coil( "Unlock_Data"."Auto_On_M6.2" )
   END_RUNG
   RUNG wire#w1
      R_Coil( "Unlock_Data"."Auto_On_M6.3" )
   END_RUNG
   RUNG wire#w1
      R_Coil( "Unlock_Data"."Auto_On_M7.1" )
   END_RUNG
   RUNG wire#w1
      R_Coil( "Unlock_Data".Auto_On_M7 )
   END_RUNG
   RUNG wire#w1
      R_Coil( "Unlock_Data"."Auto_On_X_M12.1" )
   END_RUNG
   RUNG wire#w1
      R_Coil( "Unlock_Data"."Auto_On_X_M6.1" )
   END_RUNG
   RUNG wire#w1
      R_Coil( "Unlock_Data"."Auto_On_M8.3" )
   END_RUNG
   RUNG wire#w1
      R_Coil( "Unlock_Data".Auto_On_M9 )
   END_RUNG
   RUNG wire#w1
      R_Coil( "Unlock_Data"."Auto_On_M10.1" )
   END_RUNG
   RUNG wire#w1
      R_Coil( "Unlock_Data".Auto_On_M10 )
   END_RUNG
   RUNG wire#w1
      R_Coil( "Unlock_Data".Auto_On_M11 )
   END_RUNG
   RUNG wire#w1
      R_Coil( "Unlock_Data"."Auto_On_M12.1" )
   END_RUNG
   RUNG wire#w1
      R_Coil( "Unlock_Data".Auto_On_M12 )
   END_RUNG
   RUNG wire#w1
      R_Coil( "Unlock_Data".Auto_On_M13 )
   END_RUNG
   RUNG wire#w1
      R_Coil( "Unlock_Data".Auto_On_M14 )
   END_RUNG
   // the same network as SCL:
   IF "Gribok_Shkaf_Pererabotka" OR NOT "Cepi_Upravlenia" OR "Kontrol_Seti" THEN
       "Unlock_Data"."Auto_On_M6.1" := FALSE;
       "Unlock_Data"."Auto_On_M6.2" := FALSE;
       "Unlock_Data"."Auto_On_M6.3" := FALSE;
       "Unlock_Data"."Auto_On_M7.1" := FALSE;
       "Unlock_Data".Auto_On_M7 := FALSE;
       "Unlock_Data"."Auto_On_X_M12.1" := FALSE;
       "Unlock_Data"."Auto_On_X_M6.1" := FALSE;
       "Unlock_Data"."Auto_On_M8.3" := FALSE;
       "Unlock_Data".Auto_On_M9 := FALSE;
       "Unlock_Data"."Auto_On_M10.1" := FALSE;
       "Unlock_Data".Auto_On_M10 := FALSE;
       "Unlock_Data".Auto_On_M11 := FALSE;
       "Unlock_Data"."Auto_On_M12.1" := FALSE;
       "Unlock_Data".Auto_On_M12 := FALSE;
       "Unlock_Data".Auto_On_M13 := FALSE;
       "Unlock_Data".Auto_On_M14 := FALSE;
   END_IF;
END_REGION

REGION Network 9
   RUNG wire#powerrail
      Contact( "Gribok_Shkaf_Pererabotka" )
      Coil( "Avariyn_Stop_M10" )
   END_RUNG
   // the same network as SCL:
   "Avariyn_Stop_M10" := "Gribok_Shkaf_Pererabotka";
END_REGION
END_FUNCTION_BLOCK

FUNCTION_BLOCK "Group1_Cycle"   // FB4, LAD
{ S7_Optimized_Access := 'TRUE' }
VERSION : 0.1
   VAR_TEMP   // added for the SCL form of the ladder/FBD networks
      _w1 : Bool;
      _w2 : Bool;
      _w3 : Bool;
      _w4 : Bool;
   END_VAR
BEGIN

REGION Network 1
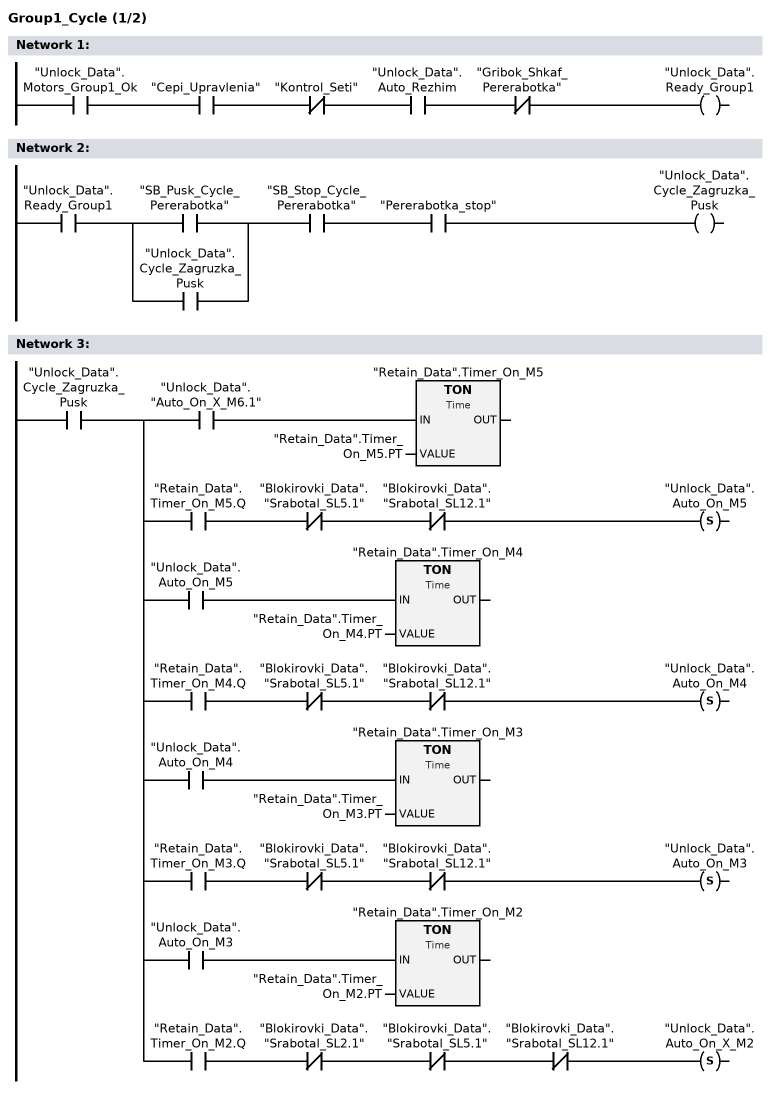
   RUNG wire#powerrail
      Contact( "Unlock_Data".Motors_Group1_Ok )
      Contact( "Cepi_Upravlenia" )
      I_Contact( "Kontrol_Seti" )
      Contact( "Unlock_Data".Auto_Rezhim )
      I_Contact( "Gribok_Shkaf_Pererabotka" )
      Coil( "Unlock_Data".Ready_Group1 )
   END_RUNG
   // the same network as SCL:
   "Unlock_Data".Ready_Group1 := "Unlock_Data".Motors_Group1_Ok AND "Cepi_Upravlenia" AND NOT "Kontrol_Seti" AND "Unlock_Data".Auto_Rezhim AND NOT "Gribok_Shkaf_Pererabotka";
END_REGION

REGION Network 2
   RUNG wire#powerrail
      Contact( "Unlock_Data".Ready_Group1 )
      wire#w1
      Contact( "SB_Pusk_Cycle_Pererabotka" )
      wire#w2
      Contact( "SB_Stop_Cycle_Pererabotka" )
      Contact( "Pererabotka_stop" )
      Coil( "Unlock_Data".Cycle_Zagruzka_Pusk )
   END_RUNG
   RUNG wire#w1
      Contact( "Unlock_Data".Cycle_Zagruzka_Pusk )
   END_RUNG wire#w2
   // the same network as SCL:
   "Unlock_Data".Cycle_Zagruzka_Pusk := "Unlock_Data".Ready_Group1 AND ("SB_Pusk_Cycle_Pererabotka" OR "Unlock_Data".Cycle_Zagruzka_Pusk) AND "SB_Stop_Cycle_Pererabotka" AND "Pererabotka_stop";
END_REGION

REGION Network 3
   "Retain_Data".Timer_On_M5.TON(IN := "Unlock_Data".Cycle_Zagruzka_Pusk AND "Unlock_Data"."Auto_On_X_M6.1", PT := "Retain_Data".Timer_On_M5.PT);   // TON coil
   IF "Unlock_Data".Cycle_Zagruzka_Pusk AND "Retain_Data".Timer_On_M5.Q AND NOT "Blokirovki_Data"."Srabotal_SL5.1" AND NOT "Blokirovki_Data"."Srabotal_SL12.1" THEN
       "Unlock_Data".Auto_On_M5 := TRUE;
   END_IF;
   "Retain_Data".Timer_On_M4.TON(IN := "Unlock_Data".Cycle_Zagruzka_Pusk AND "Unlock_Data".Auto_On_M5, PT := "Retain_Data".Timer_On_M4.PT);   // TON coil
   IF "Unlock_Data".Cycle_Zagruzka_Pusk AND "Retain_Data".Timer_On_M4.Q AND NOT "Blokirovki_Data"."Srabotal_SL5.1" AND NOT "Blokirovki_Data"."Srabotal_SL12.1" THEN
       "Unlock_Data".Auto_On_M4 := TRUE;
   END_IF;
   "Retain_Data".Timer_On_M3.TON(IN := "Unlock_Data".Cycle_Zagruzka_Pusk AND "Unlock_Data".Auto_On_M4, PT := "Retain_Data".Timer_On_M3.PT);   // TON coil
   IF "Unlock_Data".Cycle_Zagruzka_Pusk AND "Retain_Data".Timer_On_M3.Q AND NOT "Blokirovki_Data"."Srabotal_SL5.1" AND NOT "Blokirovki_Data"."Srabotal_SL12.1" THEN
       "Unlock_Data".Auto_On_M3 := TRUE;
   END_IF;
   "Retain_Data".Timer_On_M2.TON(IN := "Unlock_Data".Cycle_Zagruzka_Pusk AND "Unlock_Data".Auto_On_M3, PT := "Retain_Data".Timer_On_M2.PT);   // TON coil
   IF "Unlock_Data".Cycle_Zagruzka_Pusk AND "Retain_Data".Timer_On_M2.Q AND NOT "Blokirovki_Data"."Srabotal_SL2.1" AND NOT "Blokirovki_Data"."Srabotal_SL5.1" AND NOT "Blokirovki_Data"."Srabotal_SL12.1" THEN
       "Unlock_Data".Auto_On_X_M2 := TRUE;
   END_IF;
END_REGION

REGION Network 4
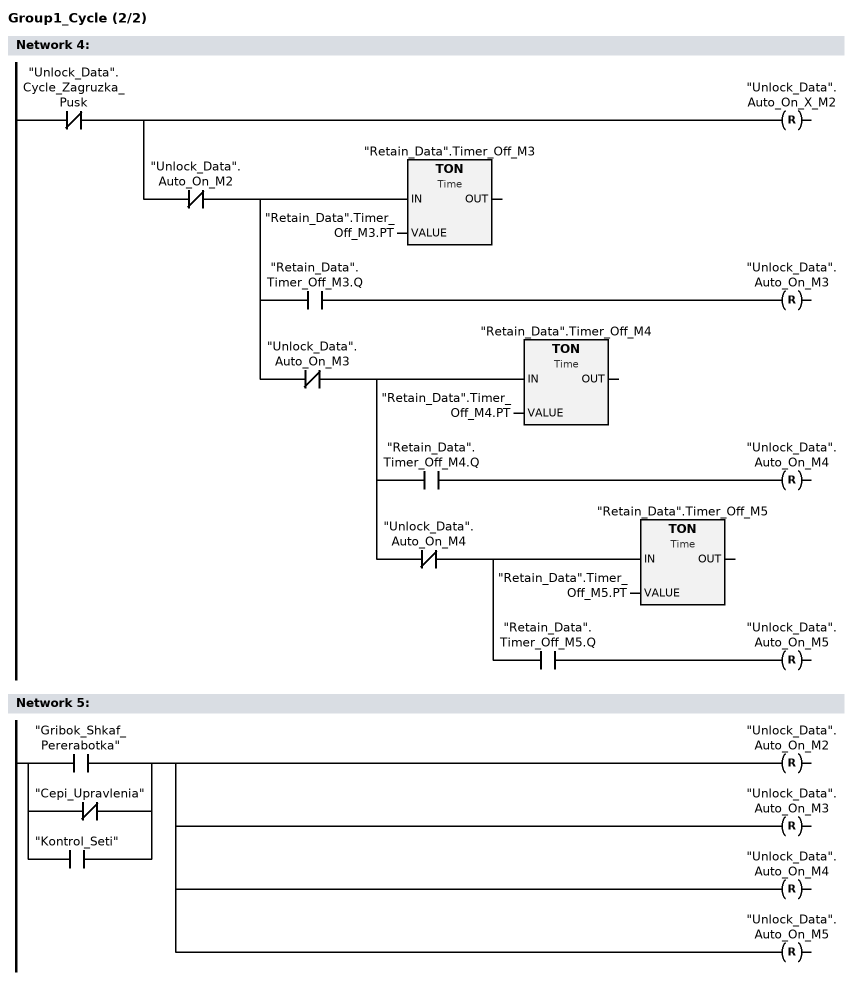
   #_w1 := NOT "Unlock_Data".Cycle_Zagruzka_Pusk;
   IF #_w1 THEN "Unlock_Data".Auto_On_X_M2 := FALSE; END_IF;
   #_w2 := #_w1 AND NOT "Unlock_Data".Auto_On_M2;
   "Retain_Data".Timer_Off_M3.TON(IN := #_w2, PT := "Retain_Data".Timer_Off_M3.PT);   // TON coil
   IF #_w2 AND "Retain_Data".Timer_Off_M3.Q THEN "Unlock_Data".Auto_On_M3 := FALSE; END_IF;
   #_w3 := #_w2 AND NOT "Unlock_Data".Auto_On_M3;
   "Retain_Data".Timer_Off_M4.TON(IN := #_w3, PT := "Retain_Data".Timer_Off_M4.PT);   // TON coil
   IF #_w3 AND "Retain_Data".Timer_Off_M4.Q THEN "Unlock_Data".Auto_On_M4 := FALSE; END_IF;
   #_w4 := #_w3 AND NOT "Unlock_Data".Auto_On_M4;
   "Retain_Data".Timer_Off_M5.TON(IN := #_w4, PT := "Retain_Data".Timer_Off_M5.PT);   // TON coil
   IF #_w4 AND "Retain_Data".Timer_Off_M5.Q THEN "Unlock_Data".Auto_On_M5 := FALSE; END_IF;
END_REGION

REGION Network 5
   RUNG wire#powerrail
      Contact( "Gribok_Shkaf_Pererabotka" )
      wire#w1
      R_Coil( "Unlock_Data".Auto_On_M2 )
   END_RUNG
   RUNG wire#powerrail
      I_Contact( "Cepi_Upravlenia" )
   END_RUNG wire#w1
   RUNG wire#powerrail
      Contact( "Kontrol_Seti" )
   END_RUNG wire#w1
   RUNG wire#w1
      R_Coil( "Unlock_Data".Auto_On_M3 )
   END_RUNG
   RUNG wire#w1
      R_Coil( "Unlock_Data".Auto_On_M4 )
   END_RUNG
   RUNG wire#w1
      R_Coil( "Unlock_Data".Auto_On_M5 )
   END_RUNG
   // the same network as SCL:
   IF "Gribok_Shkaf_Pererabotka" OR NOT "Cepi_Upravlenia" OR "Kontrol_Seti" THEN
       "Unlock_Data".Auto_On_M2 := FALSE;
       "Unlock_Data".Auto_On_M3 := FALSE;
       "Unlock_Data".Auto_On_M4 := FALSE;
       "Unlock_Data".Auto_On_M5 := FALSE;
   END_IF;
END_REGION
END_FUNCTION_BLOCK

FUNCTION_BLOCK "Filtration"   // FB5, LAD
{ S7_Optimized_Access := 'TRUE' }
VERSION : 0.1
   VAR_TEMP   // added for the SCL form of the ladder/FBD networks
      _w1 : Bool;
      _w2 : Bool;
      _w3 : Bool;
      _w4 : Bool;
      _w5 : Bool;
      _w6 : Bool;
      _w7 : Bool;
      _w8 : Bool;
      _w9 : Bool;
      _w10 : Bool;
      _w11 : Bool;
      _w12 : Bool;
      _w13 : Bool;
   END_VAR
BEGIN

REGION Network 1: Выбор режима
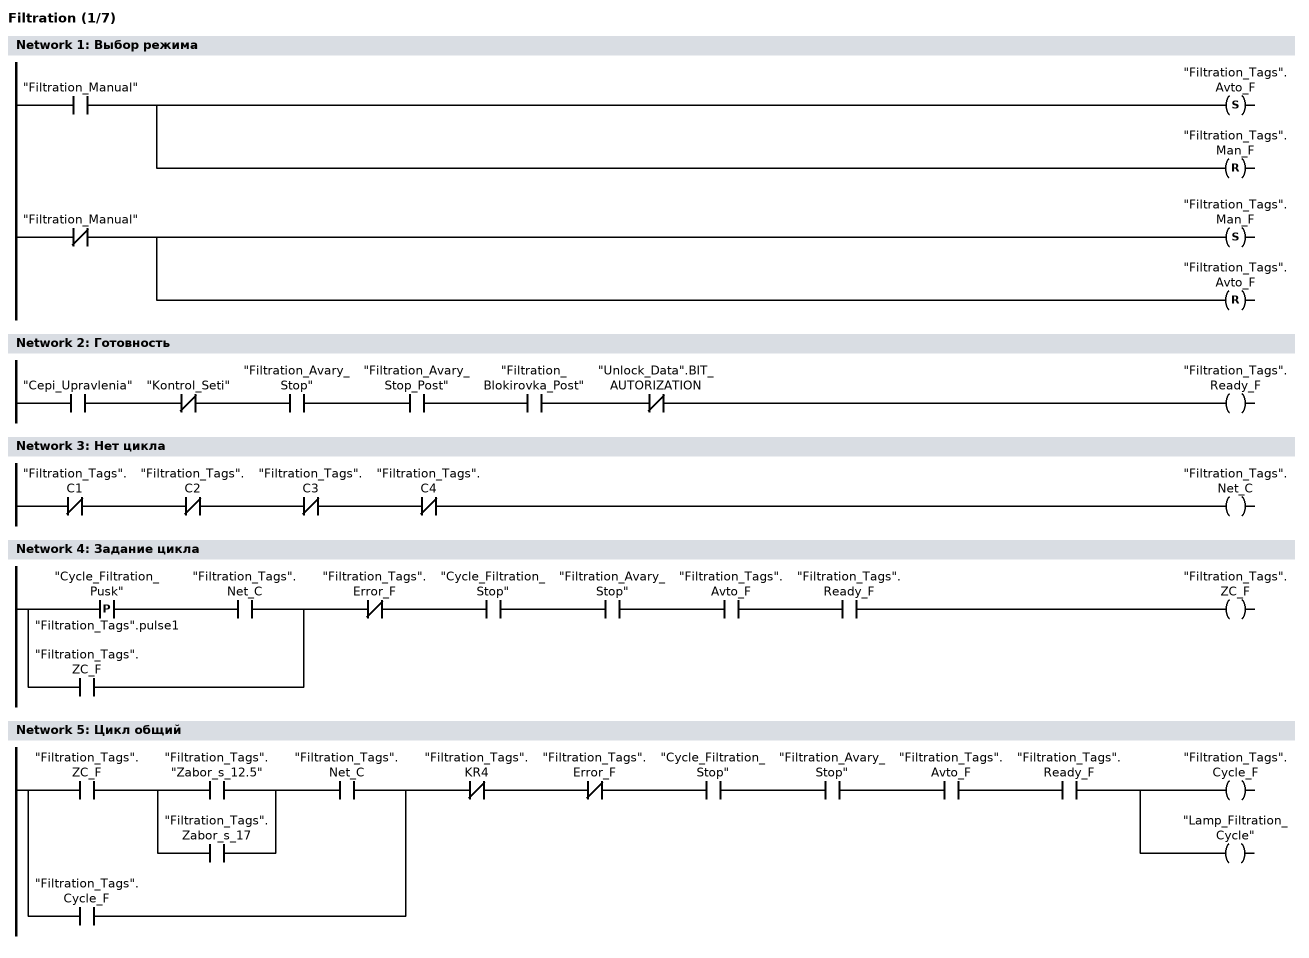
   RUNG wire#powerrail
      Contact( "Filtration_Manual" )
      wire#w1
      S_Coil( "Filtration_Tags".Avto_F )
   END_RUNG
   RUNG wire#w1
      R_Coil( "Filtration_Tags".Man_F )
   END_RUNG
   RUNG wire#powerrail
      I_Contact( "Filtration_Manual" )
      wire#w2
      S_Coil( "Filtration_Tags".Man_F )
   END_RUNG
   RUNG wire#w2
      R_Coil( "Filtration_Tags".Avto_F )
   END_RUNG
   // the same network as SCL:
   IF "Filtration_Manual" THEN
       "Filtration_Tags".Avto_F := TRUE;
       "Filtration_Tags".Man_F := FALSE;
   END_IF;
   IF NOT "Filtration_Manual" THEN
       "Filtration_Tags".Man_F := TRUE;
       "Filtration_Tags".Avto_F := FALSE;
   END_IF;
END_REGION

REGION Network 2: Готовность
   RUNG wire#powerrail
      Contact( "Cepi_Upravlenia" )
      I_Contact( "Kontrol_Seti" )
      Contact( "Filtration_Avary_Stop" )
      Contact( "Filtration_Avary_Stop_Post" )
      Contact( "Filtration_Blokirovka_Post" )
      I_Contact( "Unlock_Data".BIT_AUTORIZATION )
      Coil( "Filtration_Tags".Ready_F )
   END_RUNG
   // the same network as SCL:
   "Filtration_Tags".Ready_F := "Cepi_Upravlenia" AND NOT "Kontrol_Seti" AND "Filtration_Avary_Stop" AND "Filtration_Avary_Stop_Post" AND "Filtration_Blokirovka_Post" AND NOT "Unlock_Data".BIT_AUTORIZATION;
END_REGION

REGION Network 3: Нет цикла
   RUNG wire#powerrail
      I_Contact( "Filtration_Tags".C1 )
      I_Contact( "Filtration_Tags".C2 )
      I_Contact( "Filtration_Tags".C3 )
      I_Contact( "Filtration_Tags".C4 )
      Coil( "Filtration_Tags".Net_C )
   END_RUNG
   // the same network as SCL:
   "Filtration_Tags".Net_C := NOT "Filtration_Tags".C1 AND NOT "Filtration_Tags".C2 AND NOT "Filtration_Tags".C3 AND NOT "Filtration_Tags".C4;
END_REGION

REGION Network 4: Задание цикла
   RUNG wire#powerrail
      P_Contact(operand := "Cycle_Filtration_Pusk", bit := "Filtration_Tags".pulse1)
      Contact( "Filtration_Tags".Net_C )
      wire#w1
      I_Contact( "Filtration_Tags".Error_F )
      Contact( "Cycle_Filtration_Stop" )
      Contact( "Filtration_Avary_Stop" )
      Contact( "Filtration_Tags".Avto_F )
      Contact( "Filtration_Tags".Ready_F )
      Coil( "Filtration_Tags".ZC_F )
   END_RUNG
   RUNG wire#powerrail
      Contact( "Filtration_Tags".ZC_F )
   END_RUNG wire#w1
   // the same network as SCL:
   #_w1 := "Cycle_Filtration_Pusk" AND NOT "Filtration_Tags".pulse1;   // rising edge of "Cycle_Filtration_Pusk"
   "Filtration_Tags".pulse1 := "Cycle_Filtration_Pusk";
   "Filtration_Tags".ZC_F := ((#_w1 AND "Filtration_Tags".Net_C) OR "Filtration_Tags".ZC_F) AND NOT "Filtration_Tags".Error_F AND "Cycle_Filtration_Stop" AND "Filtration_Avary_Stop" AND "Filtration_Tags".Avto_F AND "Filtration_Tags".Ready_F;
END_REGION

REGION Network 5: Цикл общий
   RUNG wire#powerrail
      Contact( "Filtration_Tags".ZC_F )
      wire#w1
      Contact( "Filtration_Tags"."Zabor_s_12.5" )
      wire#w2
      Contact( "Filtration_Tags".Net_C )
      wire#w3
      I_Contact( "Filtration_Tags".KR4 )
      I_Contact( "Filtration_Tags".Error_F )
      Contact( "Cycle_Filtration_Stop" )
      Contact( "Filtration_Avary_Stop" )
      Contact( "Filtration_Tags".Avto_F )
      Contact( "Filtration_Tags".Ready_F )
      wire#w4
      Coil( "Filtration_Tags".Cycle_F )
   END_RUNG
   RUNG wire#w1
      Contact( "Filtration_Tags".Zabor_s_17 )
   END_RUNG wire#w2
   RUNG wire#powerrail
      Contact( "Filtration_Tags".Cycle_F )
   END_RUNG wire#w3
   RUNG wire#w4
      Coil( "Lamp_Filtration_Cycle" )
   END_RUNG
   // the same network as SCL:
   "Filtration_Tags".Cycle_F := (("Filtration_Tags".ZC_F AND ("Filtration_Tags"."Zabor_s_12.5" OR "Filtration_Tags".Zabor_s_17) AND "Filtration_Tags".Net_C) OR "Filtration_Tags".Cycle_F) AND NOT "Filtration_Tags".KR4 AND NOT "Filtration_Tags".Error_F AND "Cycle_Filtration_Stop" AND "Filtration_Avary_Stop" AND "Filtration_Tags".Avto_F AND "Filtration_Tags".Ready_F;
   "Lamp_Filtration_Cycle" := "Filtration_Tags".Cycle_F;
END_REGION

REGION Network 6: Задание циклов 1...4 в автоматическом режиме
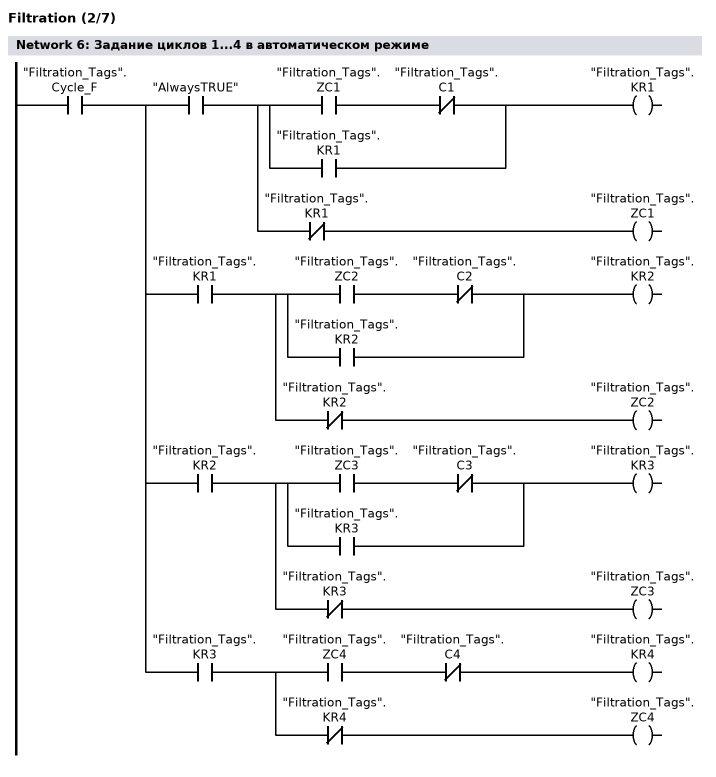
   RUNG wire#powerrail
      Contact( "Filtration_Tags".Cycle_F )
      wire#w1
      Contact( "AlwaysTRUE" )
      wire#w2
      Contact( "Filtration_Tags".ZC1 )
      I_Contact( "Filtration_Tags".C1 )
      wire#w3
      Coil( "Filtration_Tags".KR1 )
   END_RUNG
   RUNG wire#w2
      Contact( "Filtration_Tags".KR1 )
   END_RUNG wire#w3
   RUNG wire#w2
      I_Contact( "Filtration_Tags".KR1 )
      Coil( "Filtration_Tags".ZC1 )
   END_RUNG
   RUNG wire#w1
      Contact( "Filtration_Tags".KR1 )
      wire#w4
      Contact( "Filtration_Tags".ZC2 )
      I_Contact( "Filtration_Tags".C2 )
      wire#w5
      Coil( "Filtration_Tags".KR2 )
   END_RUNG
   RUNG wire#w4
      Contact( "Filtration_Tags".KR2 )
   END_RUNG wire#w5
   RUNG wire#w4
      I_Contact( "Filtration_Tags".KR2 )
      Coil( "Filtration_Tags".ZC2 )
   END_RUNG
   RUNG wire#w1
      Contact( "Filtration_Tags".KR2 )
      wire#w6
      Contact( "Filtration_Tags".ZC3 )
      I_Contact( "Filtration_Tags".C3 )
      wire#w7
      Coil( "Filtration_Tags".KR3 )
   END_RUNG
   RUNG wire#w6
      Contact( "Filtration_Tags".KR3 )
   END_RUNG wire#w7
   RUNG wire#w6
      I_Contact( "Filtration_Tags".KR3 )
      Coil( "Filtration_Tags".ZC3 )
   END_RUNG
   RUNG wire#w1
      Contact( "Filtration_Tags".KR3 )
      wire#w8
      Contact( "Filtration_Tags".ZC4 )
      I_Contact( "Filtration_Tags".C4 )
      Coil( "Filtration_Tags".KR4 )
   END_RUNG
   RUNG wire#w8
      I_Contact( "Filtration_Tags".KR4 )
      Coil( "Filtration_Tags".ZC4 )
   END_RUNG
   // the same network as SCL:
   #_w1 := "Filtration_Tags".Cycle_F AND "AlwaysTRUE";
   "Filtration_Tags".KR1 := #_w1 AND (("Filtration_Tags".ZC1 AND NOT "Filtration_Tags".C1) OR "Filtration_Tags".KR1);
   "Filtration_Tags".ZC1 := #_w1 AND NOT "Filtration_Tags".KR1;
   #_w2 := "Filtration_Tags".Cycle_F AND "Filtration_Tags".KR1;
   "Filtration_Tags".KR2 := #_w2 AND (("Filtration_Tags".ZC2 AND NOT "Filtration_Tags".C2) OR "Filtration_Tags".KR2);
   "Filtration_Tags".ZC2 := #_w2 AND NOT "Filtration_Tags".KR2;
   #_w3 := "Filtration_Tags".Cycle_F AND "Filtration_Tags".KR2;
   "Filtration_Tags".KR3 := #_w3 AND (("Filtration_Tags".ZC3 AND NOT "Filtration_Tags".C3) OR "Filtration_Tags".KR3);
   "Filtration_Tags".ZC3 := #_w3 AND NOT "Filtration_Tags".KR3;
   #_w4 := "Filtration_Tags".Cycle_F AND "Filtration_Tags".KR3;
   "Filtration_Tags".KR4 := #_w4 AND "Filtration_Tags".ZC4 AND NOT "Filtration_Tags".C4;
   "Filtration_Tags".ZC4 := #_w4 AND NOT "Filtration_Tags".KR4;
END_REGION

REGION Network 7: Выбор режима. Режимы включаются с операторской панели и работают только в ручном режиме
